Omron CX-Programmer project 新工程 (CX-Programmer 9.62)

# PLC 新PLC1: CJ2M CPU33
I/O table (CPU CJ2M-CPU33): rack 0 slot 0 CJ1W-ID261; rack 0 slot 1 CJ1W-MD261; rack 0 slot 2 CJ1W-OD261; rack 0 slot 3 CJ1W-SCU21-V1; rack 0 slot 11 CJ2M-EIP21

## Global symbols (name address type ; comment)
0.00 BOOL  ; 扫码阻挡气缸1原位
0.01 BOOL  ; 扫码阻挡气缸1到位
0.02 BOOL  ; 扫码阻挡气缸2原位
0.03 BOOL  ; 扫码阻挡气缸2到位
0.04 BOOL  ; 隔离气缸1原位
0.05 BOOL  ; 隔离气缸1到位
0.06 BOOL  ; 隔离气缸2原位
0.07 BOOL  ; 隔离气缸2到位
0.08 BOOL  ; 进料对射光电
0.09 BOOL  ; 夹爪A1夹紧位
0.10 BOOL  ; 夹爪A1松开位
0.11 BOOL  ; 夹爪A2夹紧位
0.12 BOOL  ; 夹爪A2松开位
0.13 BOOL  ; 夹爪B1夹紧位
0.14 BOOL  ; 夹爪B1松开位
0.15 BOOL  ; 夹爪B2夹紧位
10.00 BOOL  ; 扫码阻挡气缸1缩回
10.01 BOOL  ; 扫码阻挡气缸1伸出
10.02 BOOL  ; 扫码阻挡气缸2缩回
10.03 BOOL  ; 扫码阻挡气缸2伸出
10.04 BOOL  ; 隔离气缸1缩回
10.05 BOOL  ; 隔离气缸1伸出
10.06 BOOL  ; 隔离气缸2缩回
10.07 BOOL  ; 隔离气缸2伸出
10.08 BOOL  ; 上料拉带电机启动
10.09 BOOL  ; 夹爪A1夹紧
10.10 BOOL  ; 夹爪A1松开
10.11 BOOL  ; 夹爪A2夹紧
10.12 BOOL  ; 夹爪A2松开
10.13 BOOL  ; 夹爪B1夹紧
10.14 BOOL  ; 夹爪B1松开
10.15 BOOL  ; 夹爪B2夹紧
11.00 BOOL  ; 夹爪B2松开
11.01 BOOL  ; NG升降气缸1缩回
11.02 BOOL  ; NG升降气缸1伸出
11.03 BOOL  ; NG升降气缸2缩回
11.04 BOOL  ; NG升降气缸2伸出
11.05 BOOL  ; 无杆气缸1缩回
11.06 BOOL  ; 无杆气缸1伸出
11.07 BOOL  ; 无杆气缸2缩回
11.08 BOOL  ; 无杆气缸2伸出
11.09 BOOL  ; 阻挡伸出气缸1缩回
11.10 BOOL  ; 阻挡伸出气缸1伸出
11.11 BOOL  ; 阻挡伸出气缸2缩回
11.12 BOOL  ; 阻挡伸出气缸2伸出
11.13 BOOL  ; 阻挡伸出气缸3缩回
11.14 BOOL  ; 阻挡伸出气缸3伸出
11.15 BOOL  ; 阻挡伸出气缸4缩回
12.00 BOOL  ; 阻挡伸出气缸4伸出
12.01 BOOL  ; 精定位气缸A1缩回
12.02 BOOL  ; 精定位气缸A1伸出
12.03 BOOL  ; 精定位气缸A2缩回
12.04 BOOL  ; 精定位气缸A2伸出
12.05 BOOL  ; 精定位气缸B1缩回
12.06 BOOL  ; 精定位气缸B1伸出
12.07 BOOL  ; 精定位气缸B2缩回
12.08 BOOL  ; 精定位气缸B2伸出
12.09 BOOL  ; 擦拭升降气缸缩回
12.10 BOOL  ; 擦拭升降气缸伸出
12.11 BOOL  ; 压钉气缸缩回
12.12 BOOL  ; 压钉气缸伸出
12.13 BOOL  ; 料盒拨料气缸1缩回
12.14 BOOL  ; 料盒拨料气缸1伸出
12.15 BOOL  ; 料盒拨料气缸2缩回
13.00 BOOL  ; 料盒拨料气缸2伸出
13.01 BOOL  ; 推钉X轴气缸缩回
13.02 BOOL  ; 推钉X轴气缸伸出
13.03 BOOL  ; 推钉Y轴气缸缩回
13.04 BOOL  ; 推钉Y轴气缸伸出
13.05 BOOL  ; 钉位清洁拉带启动
13.06 BOOL  ; 入钉拉带启动
13.07 BOOL  ; 扫码NG收料拉带启动
13.08 BOOL  ; 入钉NG收料拉带启动
13.09 BOOL  ; 供钉振动盘启动
13.10 BOOL  ; 清洁料盘放料电机启动
13.11 BOOL  ; 料盘收料电机
13.12 BOOL  ; 真空阀打开
13.13 BOOL  ; 真空阀关闭
13.14 BOOL  ; 吹气阀打开
13.15 BOOL  ; 吹气阀关闭
1535.01 BOOL  ; ETN21_1TCP Socket No.2 Receving Flag
1535.02 BOOL  ; ETN21_1TCP Socket No.2 Sending Flag
1535.03 BOOL  ; ETN21_1TCP Socket No.2 Closing Flag
1535.13 BOOL  ; ETN21_1TCP Socket No.2 Data Receved Flag
1535.15 BOOL  ; ETN21_1TCP Socket No.2 TCP Connection/TCP Open Flag
1544.10 BOOL  ; ETN21_1Socket2 TCP Active Open Request SW
1544.11 BOOL  ; ETN21_1Socket2 Send Request Switch
1544.12 BOOL  ; ETN21_1Socket2 Receive Request SW
1544.13 BOOL  ; ETN21_1Socket2 Close Request SW
1544.15 BOOL  ; SCU21_1 Port#2忙绿标志
1559.15 BOOL  ; SCU21_2Port#1 Protocol Macro Executing Flag
186.00 BOOL  ; 1#入料扫码启动
1.00 BOOL  ; 夹爪B2松开位
1.01 BOOL  ; NG升降气缸1原位
1.02 BOOL  ; NG升降气缸1到位
1.03 BOOL  ; NG升降气缸2原位
1.04 BOOL  ; NG升降气缸2到位
1.05 BOOL  ; 无杆气缸1原位
1.06 BOOL  ; 无杆气缸1到位
1.07 BOOL  ; 无杆气缸2原位
1.08 BOOL  ; 无杆气缸2到位
1.09 BOOL  ; 阻挡伸出气缸1原位
1.10 BOOL  ; 阻挡伸出气缸1到位
1.11 BOOL  ; 阻挡伸出气缸2原位
1.12 BOOL  ; 阻挡伸出气缸2到位
1.13 BOOL  ; 阻挡伸出气缸3原位
1.14 BOOL  ; 阻挡伸出气缸3到位
1.15 BOOL  ; 阻挡伸出气缸4原位
200.00 BOOL  ; PLC上电
200.01 BOOL  ; 紧急停止
200.02 BOOL  ; 自动启动
200.03 BOOL  ; 自动停止
200.04 BOOL  ; 报警清除
200.05 BOOL  ; 清料停止中
200.06 BOOL  ; 异常报警停止
200.07 BOOL  ; 自动模式擦拭拉带启动
200.08 BOOL  ; 自动模式入钉拉带启动
200.09 BOOL  ; 设备内有电池
200.10 BOOL  ; 机台有错误
200.11 BOOL  ; 报警中
200.12 BOOL  ; 三色灯-绿灯
200.13 BOOL  ; 三色灯-红灯
200.14 BOOL  ; 三色灯-黄灯
200.15 BOOL  ; 三色灯-蜂鸣器
201.00 BOOL  ; 整机在初始位
205.00 BOOL  ; 整机停止中（Lamp）
205.01 BOOL  ; 清料停止中（Lamp）
205.02 BOOL  ; 整机复位（Lamp）
210.01 BOOL  ; PC系统通讯正常标志
210.03 BOOL  ; 安全门标志
210.04 BOOL  ; 供料震盘启动标志
210.05 BOOL  ; 机器人Socket_Tcp连接完成标志
210.06 BOOL  ; 扫码枪Socket_Tcp连接完成标志
221.00 BOOL  ; 整机复位（M）
221.01 BOOL  ; 电池上料机构复位（M）
221.02 BOOL  ; 扫码NG抓取机构复位（M）
221.03 BOOL  ; 电池清洁机构复位
221.04 BOOL  ; 电池入钉机构复位（M）
221.05 BOOL  ; 入钉NG抓取机构复位（M）
221.06 BOOL  ; 扫码入料机构记忆复位（M）
221.08 BOOL  ; 进料拉带扫码工站整机复位（M）
2960.06 BOOL  ; 入钉升降伺服负极限
2960.07 BOOL  ; 入钉伺服正极限
2962.06 BOOL  ; 上料水平伺服负极限
2962.07 BOOL  ; 上料水平伺服正极限
2.00 BOOL  ; 阻挡伸出气缸4到位
2.01 BOOL  ; 精定位气缸A1原位
2.02 BOOL  ; 精定位气缸A1到位
2.03 BOOL  ; 精定位气缸A2原位
2.04 BOOL  ; 精定位气缸A2到位
2.05 BOOL  ; 精定位气缸B1原位
2.06 BOOL  ; 精定位气缸B1到位
2.07 BOOL  ; 精定位气缸B2原位
2.08 BOOL  ; 精定位气缸B2到位
2.09 BOOL  ; 擦拭升降气缸原位
2.10 BOOL  ; 擦拭升降气缸到位
2.11 BOOL  ; 压钉气缸原位
2.12 BOOL  ; 压钉气缸到位
2.13 BOOL  ; 料盒拨料气缸1原位
2.14 BOOL  ; 料盒拨料气缸1到位
2.15 BOOL  ; 料盒拨料气缸2原位
300.00 BOOL  ; 扫码阻挡气缸1缩回[Pls]
300.01 BOOL  ; 扫码阻挡气缸1伸出[Pls]
300.02 BOOL  ; 扫码阻挡气缸2缩回[Pls]
300.03 BOOL  ; 扫码阻挡气缸2伸出[Pls]
300.04 BOOL  ; 隔离气缸1缩回[Pls]
300.05 BOOL  ; 隔离气缸1伸出[Pls]
300.06 BOOL  ; 隔离气缸2缩回[Pls]
300.07 BOOL  ; 隔离气缸2伸出[Pls]
300.08 BOOL  ; 进料拉带电机启动[Pls]
300.09 BOOL  ; 夹爪A1夹紧[Pls]
300.10 BOOL  ; 夹爪A1松开[Pls]
300.11 BOOL  ; 夹爪A2夹紧[Pls]
300.12 BOOL  ; 夹爪A2松开[Pls]
300.13 BOOL  ; 夹爪B1夹紧[Pls]
300.14 BOOL  ; 夹爪B1松开[Pls]
300.15 BOOL  ; 夹爪B2夹紧[Pls]
301.00 BOOL  ; 夹爪B2松开[Pls]
301.01 BOOL  ; NG升降气缸1缩回[Pls]
301.02 BOOL  ; NG升降气缸1伸出[Pls]
301.03 BOOL  ; NG升降气缸2缩回[Pls]
301.04 BOOL  ; NG升降气缸2伸出[Pls]
301.05 BOOL  ; 无杆气缸1缩回[Pls]
301.06 BOOL  ; 无杆气缸1伸出[Pls]
301.07 BOOL  ; 无杆气缸2缩回[Pls]
301.08 BOOL  ; 无杆气缸2伸出[Pls]
301.09 BOOL  ; 阻挡伸出气缸1缩回[Pls]
301.10 BOOL  ; 阻挡伸出气缸1伸出[Pls]
301.11 BOOL  ; 阻挡伸出气缸2缩回[Pls]
301.12 BOOL  ; 阻挡伸出气缸2伸出[Pls]
301.13 BOOL  ; 阻挡伸出气缸3缩回[Pls]
301.14 BOOL  ; 阻挡伸出气缸3伸出[Pls]
301.15 BOOL  ; 阻挡伸出气缸4缩回[Pls]
302.00 BOOL  ; 阻挡伸出气缸4伸出[Pls]
302.01 BOOL  ; 精定位气缸A1缩回[Pls]
302.02 BOOL  ; 精定位气缸A1伸出[Pls]
302.03 BOOL  ; 精定位气缸A2缩回[Pls]
302.04 BOOL  ; 精定位气缸A2伸出[Pls]
302.05 BOOL  ; 精定位气缸B1缩回[Pls]
302.06 BOOL  ; 精定位气缸B1伸出[Pls]
302.07 BOOL  ; 精定位气缸B2缩回[Pls]
302.08 BOOL  ; 精定位气缸B2伸出[Pls]
302.09 BOOL  ; 擦拭升降气缸缩回[Pls]
302.10 BOOL  ; 擦拭升降气缸伸出[Pls]
302.11 BOOL  ; 压钉气缸缩回[Pls]
302.12 BOOL  ; 压钉气缸伸出[Pls]
302.13 BOOL  ; 料盒拨料气缸1缩回[Pls]
302.14 BOOL  ; 料盒拨料气缸1伸出[Pls]
302.15 BOOL  ; 料盒拨料气缸2缩回[Pls]
303.00 BOOL  ; 料盒拨料气缸2伸出[Pls]
303.01 BOOL  ; 推钉X轴气缸缩回[Pls]
303.02 BOOL  ; 推钉X轴气缸伸出[Pls]
303.03 BOOL  ; 推钉Y轴气缸缩回[Pls]
303.04 BOOL  ; 推钉Y轴气缸伸出[Pls]
303.05 BOOL  ; 入钉位拉带启动[Pls]
303.06 BOOL  ; 入钉NG位拉带启动[Pls]
303.07 BOOL  ; 清洁放料拉带启动[Pls]
303.08 BOOL  ; 清洁收料拉带启动[Pls]
303.09 BOOL  ; 供料振动盘启动[Pls]
303.11 BOOL  ; 入钉真空阀打开PLS
303.12 BOOL  ; $?St$Bk?_#[5] / 入钉真空阀打开PLS / $?St$Bk?_#[5]
303.13 BOOL  ; 入钉真空阀关闭PLS
303.14 BOOL  ; 入钉吹气阀打开PLS
303.15 BOOL  ; 入钉吹气阀关闭PLS
3.00 BOOL  ; 料盒拨料气缸2到位
3.01 BOOL  ; 推钉X轴气缸原位
3.02 BOOL  ; 推钉X轴气缸到位
3.03 BOOL  ; 推钉Y轴气缸原位
3.04 BOOL  ; 推钉Y轴气缸到位
3.05 BOOL  ; 扫码位对射光电
3.06 BOOL  ; 分隔电池对射光电
3.07 BOOL  ; 擦拭料带下限满料感应
3.08 BOOL  ; 擦拭料带放料上限光电[0003.08]
3.09 BOOL  ; 擦拭带盘无料料感应
3.10 BOOL  ; 扫码NG位对射光电
3.11 BOOL  ; 擦拭位对射光电
3.12 BOOL  ; 入钉位对射光电
3.13 BOOL  ; 入钉NG位对射光电
3.14 BOOL  ; 扫码NG槽对射前
3.15 BOOL  ; 入钉NG槽对射前
400.00 BOOL  ; 扫码阻挡气缸1缩回[M]
400.01 BOOL  ; 扫码阻挡气缸1伸出[M]
400.02 BOOL  ; 扫码阻挡气缸2缩回[M]
400.03 BOOL  ; 扫码阻挡气缸2伸出[M]
400.04 BOOL  ; 隔离气缸1缩回[M]
400.05 BOOL  ; 隔离气缸1伸出[M]
400.06 BOOL  ; 隔离气缸2缩回[M]
400.07 BOOL  ; 隔离气缸2伸出[M]
400.08 BOOL  ; 进料拉带电机启动[M]
400.09 BOOL  ; 夹爪A1夹紧[M]
400.10 BOOL  ; 夹爪A1松开[M]
400.11 BOOL  ; 夹爪A2夹紧[M]
400.12 BOOL  ; 夹爪A2松开[M]
400.13 BOOL  ; 夹爪B1夹紧[M]
400.14 BOOL  ; 夹爪B1松开[M]
400.15 BOOL  ; 夹爪B2夹紧[M]
401.00 BOOL  ; 夹爪B2松开[M]
401.01 BOOL  ; NG升降气缸1缩回[M]
401.02 BOOL  ; NG升降气缸1伸出[M]
401.03 BOOL  ; NG升降气缸2缩回[M]
401.04 BOOL  ; NG升降气缸2伸出[M]
401.05 BOOL  ; 无杆气缸1缩回[M]
401.06 BOOL  ; 无杆气缸1伸出[M]
401.07 BOOL  ; 无杆气缸2缩回[M]
401.08 BOOL  ; 无杆气缸2伸出[M]
401.09 BOOL  ; 阻挡伸出气缸1缩回[M]
401.10 BOOL  ; 阻挡伸出气缸1伸出[M]
401.11 BOOL  ; 阻挡伸出气缸2缩回[M]
401.12 BOOL  ; 阻挡伸出气缸2伸出[M]
401.13 BOOL  ; 阻挡伸出气缸3缩回[M]
401.14 BOOL  ; 阻挡伸出气缸3伸出[M]
401.15 BOOL  ; 阻挡伸出气缸4缩回[M]
402.00 BOOL  ; 阻挡伸出气缸4伸出[M]
402.01 BOOL  ; 精定位气缸A1缩回[M]
402.02 BOOL  ; 精定位气缸A1伸出[M]
402.03 BOOL  ; 精定位气缸A2缩回[M]
402.04 BOOL  ; 精定位气缸A2伸出[M]
402.05 BOOL  ; 精定位气缸B1缩回[M]
402.06 BOOL  ; 精定位气缸B1伸出[M]
402.07 BOOL  ; 精定位气缸B2缩回[M]
402.08 BOOL  ; 精定位气缸B2伸出[M]
402.09 BOOL  ; 擦拭升降气缸缩回[M]
402.10 BOOL  ; 擦拭升降气缸伸出[M]
402.11 BOOL  ; 压钉气缸缩回[M]
402.12 BOOL  ; 压钉气缸伸出[M]
402.13 BOOL  ; 料盒拨料气缸1缩回[M]
402.14 BOOL  ; 料盒拨料气缸1伸出[M]
402.15 BOOL  ; 料盒拨料气缸2缩回[M]
403.00 BOOL  ; 料盒拨料气缸2伸出[M]
403.01 BOOL  ; 推钉X轴气缸缩回[M]
403.02 BOOL  ; 推钉X轴气缸伸出[M]
403.03 BOOL  ; 推钉Y轴气缸缩回[M]
403.04 BOOL  ; 推钉Y轴气缸伸出[M]
403.05 BOOL  ; $?St$Bk?_#[6] / 钉位清洁拉带启动[M] / $?St$Bk?_#[6]
403.06 BOOL  ; 入钉位拉带启动[M]
403.07 BOOL  ; 扫码NG收料拉带启动(M)
403.08 BOOL  ; 入钉NG收料拉带启动[M]
403.09 BOOL  ; 供钉振动盘启动[M]
403.10 BOOL  ; 清洁料盘放料电机启动（M)
403.11 BOOL  ; 料盘收料电机启动
403.12 BOOL  ; 入钉真空阀打开
403.13 BOOL  ; $?St$Bk?_#[7] / 入钉真空阀关闭[M] / $?St$Bk?_#[7]
403.14 BOOL  ; 入钉吹气阀打开（M)
403.15 BOOL  ; 入钉吹气阀关闭M
406.00 BOOL  ; 扫码按钮HIM
417.00 BOOL  ; 进料拉带扫码测试[M]
4.00 BOOL  ; 入钉伺服使能
4.02 BOOL  ; 给下位机拉带下料信号
4.05 BOOL  ; 启动按钮指示灯
4.06 BOOL  ; 停止按钮指示灯
4.07 BOOL  ; 复位按钮指示灯
4.08 BOOL  ; 三色灯（红）
4.09 BOOL  ; 三色灯（绿）
4.10 BOOL  ; 三色灯（黄）
4.11 BOOL  ; 蜂鸣器
4.12 BOOL  ; $?St$Bk?_#[8] / 入钉刹车线圈 / $?St$Bk?_#[8]
500.00 BOOL  ; 扫码阻挡气缸1缩回条件
500.01 BOOL  ; 扫码阻挡气缸1伸出条件
500.02 BOOL  ; 扫码阻挡气缸2缩回条件
500.03 BOOL  ; 扫码阻挡气缸2伸出条件
500.04 BOOL  ; 隔离气缸1缩回条件
500.05 BOOL  ; 隔离气缸1伸出条件
500.06 BOOL  ; 隔离气缸2缩回条件
500.07 BOOL  ; 隔离气缸2伸出条件
500.08 BOOL  ; 上料拉带电机启动条件
500.09 BOOL  ; 夹爪A1夹紧条件
500.10 BOOL  ; 夹爪A1松开条件
500.11 BOOL  ; 夹爪A2夹紧条件
500.12 BOOL  ; 夹爪A2松开条件
500.13 BOOL  ; 夹爪B1夹紧条件
500.14 BOOL  ; 夹爪B1松开条件
500.15 BOOL  ; 夹爪B2夹紧条件
501.00 BOOL  ; 夹爪B2松开条件
501.01 BOOL  ; NG升降气缸1缩回条件
501.02 BOOL  ; NG升降气缸1伸出条件
501.03 BOOL  ; NG升降气缸2缩回条件
501.04 BOOL  ; NG升降气缸2伸出条件
501.05 BOOL  ; 无杆气缸1缩回条件
501.06 BOOL  ; 无杆气缸1伸出条件
501.07 BOOL  ; 无杆气缸2缩回条件
501.08 BOOL  ; 无杆气缸2伸出条件
501.09 BOOL  ; 阻挡伸出气缸1缩回条件
501.10 BOOL  ; 阻挡伸出气缸1伸出条件
501.11 BOOL  ; 阻挡伸出气缸2缩回条件
501.12 BOOL  ; 阻挡伸出气缸2伸出条件
501.13 BOOL  ; 阻挡伸出气缸3缩回条件
501.14 BOOL  ; 阻挡伸出气缸3伸出条件
501.15 BOOL  ; 阻挡伸出气缸4缩回条件
502.00 BOOL  ; 阻挡伸出气缸4伸出条件
502.01 BOOL  ; 精定位气缸A1缩回条件
502.02 BOOL  ; 精定位气缸A1伸出条件
502.03 BOOL  ; 精定位气缸A2缩回条件
502.04 BOOL  ; 精定位气缸A2伸出条件
502.05 BOOL  ; 精定位气缸B1缩回条件
502.06 BOOL  ; 精定位气缸B1伸出条件
502.07 BOOL  ; 精定位气缸B2缩回条件
502.08 BOOL  ; 精定位气缸B2伸出条件
502.09 BOOL  ; 擦拭升降气缸缩回条件
502.10 BOOL  ; 擦拭升降气缸伸出条件
502.11 BOOL  ; 压钉气缸缩回条件
502.12 BOOL  ; 压钉气缸伸出条件
502.13 BOOL  ; 料盒拨料气缸1缩回条件
502.14 BOOL  ; 料盒拨料气缸1伸出条件
502.15 BOOL  ; 料盒拨料气缸2缩回条件
503.00 BOOL  ; 料盒拨料气缸2伸出条件
503.01 BOOL  ; 推钉X轴气缸缩回条件
503.02 BOOL  ; 推钉X轴气缸伸出条件
503.03 BOOL  ; 推钉Y轴气缸缩回条件
503.04 BOOL  ; 推钉Y轴气缸伸出条件
503.05 BOOL  ; $?St$Bk?_#[9] / 钉位清洁拉带启动条件 / $?St$Bk?_#[9]
503.06 BOOL  ; 入钉NG位拉带启动条件
503.07 BOOL  ; 清洁放料拉带启动条件
503.08 BOOL  ; 清洁收料拉带启动条件
503.09 BOOL  ; 供料振动盘启动条件
503.12 BOOL  ; $?St$Bk?_#[10] / 入钉真空阀条件 / $?St$Bk?_#[10]
503.13 BOOL  ; $?St$Bk?_#[11] / 入钉真空阀关闭条件 / $?St$Bk?_#[11]
503.14 BOOL  ; $?St$Bk?_#[12] / 入钉吹气打开条件 / $?St$Bk?_#[12]
503.15 BOOL  ; 入钉吹气关闭条件
600.00 BOOL  ; 扫码阻挡气缸1缩回[A]
600.01 BOOL  ; 扫码阻挡气缸1伸出[A]
600.02 BOOL  ; 扫码阻挡气缸2缩回[A]
600.03 BOOL  ; 扫码阻挡气缸2伸出[A]
600.04 BOOL  ; 隔离气缸1缩回[A]
600.05 BOOL  ; 隔离气缸1伸出[A]
600.06 BOOL  ; 隔离气缸2缩回[A]
600.07 BOOL  ; 隔离气缸2伸出[A]
600.08 BOOL  ; 进料拉带电机启动[A]
600.09 BOOL  ; 夹爪A1夹紧[A]
600.10 BOOL  ; 夹爪A1松开[A]
600.11 BOOL  ; 夹爪A2夹紧[A]
600.12 BOOL  ; 夹爪A2松开[A]
600.13 BOOL  ; 夹爪B1夹紧[A]
600.14 BOOL  ; 夹爪B1松开[A]
600.15 BOOL  ; 夹爪B2夹紧[A]
601.00 BOOL  ; 夹爪B2松开[A]
601.01 BOOL  ; NG升降气缸1缩回[A]
601.02 BOOL  ; NG升降气缸1伸出[A]
601.03 BOOL  ; NG升降气缸2缩回[A]
601.04 BOOL  ; NG升降气缸2伸出[A]
601.05 BOOL  ; 无杆气缸1缩回[A]
601.06 BOOL  ; 无杆气缸1伸出[A]
601.07 BOOL  ; 无杆气缸2缩回[A]
601.08 BOOL  ; 无杆气缸2伸出[A]
601.09 BOOL  ; 阻挡伸出气缸1缩回[A]
601.10 BOOL  ; 阻挡伸出气缸1伸出[A]
601.11 BOOL  ; 阻挡伸出气缸2缩回[A]
601.12 BOOL  ; 阻挡伸出气缸2伸出[A]
601.13 BOOL  ; 阻挡伸出气缸3缩回[A]
601.14 BOOL  ; 阻挡伸出气缸3伸出[A]
601.15 BOOL  ; 阻挡伸出气缸4缩回[A]
602.00 BOOL  ; 阻挡伸出气缸4伸出[A]
602.01 BOOL  ; 精定位气缸A1缩回[A]
602.02 BOOL  ; 精定位气缸A1伸出[A]
602.03 BOOL  ; 精定位气缸A2缩回[A]
602.04 BOOL  ; 精定位气缸A2伸出[A]
602.05 BOOL  ; 精定位气缸B1缩回[A]
602.06 BOOL  ; 精定位气缸B1伸出[A]
602.07 BOOL  ; 精定位气缸B2缩回[A]
602.08 BOOL  ; 精定位气缸B2伸出[A]
602.09 BOOL  ; 擦拭升降气缸缩回[A]
602.10 BOOL  ; 擦拭升降气缸伸出[A]
602.11 BOOL  ; 压钉气缸缩回[A]
602.12 BOOL  ; 压钉气缸伸出[A]
602.13 BOOL  ; 料盒拨料气缸1缩回[A]
602.14 BOOL  ; 料盒拨料气缸1伸出[A]
602.15 BOOL  ; 料盒拨料气缸2缩回[A]
603.00 BOOL  ; 料盒拨料气缸2伸出[A]
603.01 BOOL  ; 推钉X轴气缸缩回[A]
603.02 BOOL  ; 推钉X轴气缸伸出[A]
603.03 BOOL  ; 推钉Y轴气缸缩回[A]
603.04 BOOL  ; 推钉Y轴气缸伸出[A]
603.05 BOOL  ; $?St$Bk?_#[13] / 钉位清洁拉带启动[A] / $?St$Bk?_#[13]
603.06 BOOL  ; 入钉NG位拉带启动[A]
603.07 BOOL  ; 扫码NG收料拉带启动[A]
603.08 BOOL  ; 入钉NG收料拉带启动[A]
603.09 BOOL  ; 供钉振动盘启动[A]
603.10 BOOL  ; 清洁料盘放料电机启动[A]
603.11 BOOL  ; $?St$Bk?_#[14] / 料盘收料电机启动[M] / $?St$Bk?_#[14]
603.12 BOOL  ; $?St$Bk?_#[15] / 入钉真空阀打开 / $?St$Bk?_#[15]
603.13 BOOL  ; 入钉真空阀关闭
603.14 BOOL  ; $?St$Bk?_#[16] / 入钉吹气打开[A] / $?St$Bk?_#[16]
603.15 BOOL  ; 入钉吹气阀关闭
6.00 BOOL  ; 扫码NG槽对射光电
6.01 BOOL  ; 入钉NG槽对射后
6.02 BOOL  ; 入钉检测区域光纤
6.03 BOOL  ; 入钉伺服就绪
6.04 BOOL  ; 入钉伺服报警
6.05 BOOL  ; 启动按钮
6.06 BOOL  ; 停止按钮
6.07 BOOL  ; 复位按钮
6.08 BOOL  ; 急停按钮
6.09 BOOL  ; 手自动选择
6.10 BOOL  ; 设备总气压
6.11 BOOL  ; 夹爪1柔性报警
6.12 BOOL  ; 夹爪2柔性报警
6.13 BOOL  ; 真空信号
6.14 BOOL  ; 开关电源监测
6.15 BOOL  ; 变频器监测
700 CHANNEL  ; 手动按钮操作字
700.00 BOOL  ; 扫码阻挡气缸1缩回[SW]
700.01 BOOL  ; 扫码阻挡气缸1伸出[SW]
700.02 BOOL  ; 扫码阻挡气缸2缩回[SW]
700.03 BOOL  ; 扫码阻挡气缸2伸出[SW]
700.04 BOOL  ; 隔离气缸1缩回[SW]
700.05 BOOL  ; 隔离气缸1伸出[SW]
700.06 BOOL  ; 隔离气缸2缩回[SW]
700.07 BOOL  ; 隔离气缸2伸出[SW]
700.08 BOOL  ; 进料拉带电机启动[SW]
700.09 BOOL  ; 夹爪A1夹紧[SW]
700.10 BOOL  ; 夹爪A1松开[SW]
700.11 BOOL  ; 夹爪A2夹紧[SW]
700.12 BOOL  ; 夹爪A2松开[SW]
700.13 BOOL  ; 夹爪B1夹紧[SW]
700.14 BOOL  ; 夹爪B1松开[SW]
700.15 BOOL  ; 夹爪B2夹紧[SW]
701.00 BOOL  ; 夹爪B2松开[SW]
701.01 BOOL  ; NG升降气缸1缩回[SW]
701.02 BOOL  ; NG升降气缸1伸出[SW]
701.03 BOOL  ; NG升降气缸2缩回[SW]
701.04 BOOL  ; NG升降气缸2伸出[SW]
701.05 BOOL  ; 无杆气缸1缩回[SW]
701.06 BOOL  ; 无杆气缸1伸出[SW]
701.07 BOOL  ; 无杆气缸2缩回[SW]
701.08 BOOL  ; 无杆气缸2伸出[SW]
701.09 BOOL  ; 阻挡伸出气缸1缩回[SW]
701.10 BOOL  ; 阻挡伸出气缸1伸出[SW]
701.11 BOOL  ; 阻挡伸出气缸2缩回[SW]
701.12 BOOL  ; 阻挡伸出气缸2伸出[SW]
701.13 BOOL  ; 阻挡伸出气缸3缩回[SW]
701.14 BOOL  ; 阻挡伸出气缸3伸出[SW]
701.15 BOOL  ; 阻挡伸出气缸4缩回[SW]
702.00 BOOL  ; 阻挡伸出气缸4伸出[SW]
702.01 BOOL  ; 精定位气缸A1缩回[SW]
702.02 BOOL  ; 精定位气缸A1伸出[SW]
702.03 BOOL  ; 精定位气缸A2缩回[SW]
702.04 BOOL  ; 精定位气缸A2伸出[SW]
702.05 BOOL  ; 精定位气缸B1缩回[SW]
702.06 BOOL  ; 精定位气缸B1伸出[SW]
702.07 BOOL  ; 精定位气缸B2缩回[SW]
702.08 BOOL  ; 精定位气缸B2伸出[SW]
702.09 BOOL  ; 擦拭升降气缸缩回[SW]
702.10 BOOL  ; 擦拭升降气缸伸出[SW]
702.11 BOOL  ; 压钉气缸缩回[SW]
702.12 BOOL  ; 压钉气缸伸出[SW]
702.13 BOOL  ; 料盒拨料气缸1缩回[SW]
702.14 BOOL  ; 料盒拨料气缸1伸出[SW]
702.15 BOOL  ; 料盒拨料气缸2缩回[SW]
703.00 BOOL  ; 料盒拨料气缸2伸出[SW]
703.01 BOOL  ; 推钉X轴气缸缩回[SW]
703.02 BOOL  ; 推钉X轴气缸伸出[SW]
703.03 BOOL  ; 推钉Y轴气缸缩回[SW]
703.04 BOOL  ; 推钉Y轴气缸伸出[SW]
703.05 BOOL  ; 钉位清洁拉带启动[SW]
703.06 BOOL  ; 入钉位拉带启动[SW]
703.07 BOOL  ; 扫码NG收料拉带启动[SW]
703.08 BOOL  ; 入钉NG收料拉带启动[SW]
703.09 BOOL  ; 供钉振动盘启动[SW]
703.10 BOOL  ; 清洁料盘放料电机启动（SW)
703.11 BOOL  ; 料盘收料电机
703.12 BOOL  ; 入钉真空阀打开
703.13 BOOL  ; 入钉真空阀关闭
703.14 BOOL  ; 入钉吹气阀打开
703.15 BOOL  ; 入钉吹气阀关闭
710 CHANNEL  ; 手动按钮操作字
712.00 BOOL  ; 进料拉带电机停止[SW]
712.01 BOOL  ; 钉位清洁拉带停止[SW]
712.02 BOOL  ; 入钉位拉带停止[SW]
712.03 BOOL  ; 扫码NG收料拉带停止[SW]
712.04 BOOL  ; 入钉NG收料拉带停止[SW]
712.05 BOOL  ; 供钉振动盘停止[SW]
712.06 BOOL  ; 清洁料盘放料电机停止（SW)
712.07 BOOL  ; 清洁料盘收料电机停止（SW)
712.08 BOOL  ; $?St$Bk?_#[17] / 入钉真空阀关闭[SW] / $?St$Bk?_#[17]
712.09 BOOL  ; $?St$Bk?_#[18] / 入钉吹气阀关闭[SW] / $?St$Bk?_#[18]
716.00 BOOL  ; 1#入料扫码[SW]
750 CHANNEL  ; 手动按钮操作字
7.00 BOOL  ; NG门磁开关
7.01 BOOL  ; 前门磁开关
7.02 BOOL  ; 后门磁开关
7.03 BOOL  ; 左门磁开关
7.04 BOOL  ; 右门磁开关
7.05 BOOL  ; 区域光纤对射
7.06 BOOL  ; 钉位钉子对射光纤钉位
7.07 BOOL  ; 震盘钉嘴反射光纤
7.08 BOOL  ; 拉带入口对射光电
7.10 BOOL  ; 下位机收料完成信号
7.12 BOOL  ; 1
800.00 BOOL  ; 扫码阻挡气缸1原位标志[0000.00]
800.01 BOOL  ; 扫码阻挡气缸1到位标志[0000.01]
800.02 BOOL  ; 扫码阻挡气缸2原位标志[0000.02]
800.03 BOOL  ; 扫码阻挡气缸2到位标志[0000.03]
800.04 BOOL  ; 隔离气缸1原位标志[0000.04]
800.05 BOOL  ; 隔离气缸1到位标志[0000.05]
800.06 BOOL  ; 隔离气缸2原位标志[0000.06]
800.07 BOOL  ; 隔离气缸2到位标志[0000.07]
800.08 BOOL  ; 进料对射光电满料标志[0000.08]
800.09 BOOL  ; 夹爪A1夹紧位标志[0000.09]
800.10 BOOL  ; 夹爪A1松开位标志[0000.10]
800.11 BOOL  ; 夹爪A2夹紧位标志[0000.11]
800.12 BOOL  ; 夹爪A2松开位标志[0000.12]
800.13 BOOL  ; 夹爪B1夹紧位标志[0000.13]
800.14 BOOL  ; 夹爪B1松开位标志[0000.14]
800.15 BOOL  ; 夹爪B2夹紧位标志[0000.15]
801.00 BOOL  ; 夹爪B2松开位标志[0001.00]
801.01 BOOL  ; NG升降气缸1原位标志[0001.01]
801.02 BOOL  ; NG升降气缸1到位标志[0001.02]
801.03 BOOL  ; NG升降气缸2原位标志[0001.03]
801.04 BOOL  ; NG升降气缸2到位标志[0001.04]
801.05 BOOL  ; 无杆气缸1原位标志[0001.05]
801.06 BOOL  ; 无杆气缸1到位标志[0001.06]
801.07 BOOL  ; 无杆气缸2原位标志[0001.07]
801.08 BOOL  ; 无杆气缸2到位标志[0001.08]
801.09 BOOL  ; 拉带阻挡气缸1原位标志[0001.09]
801.10 BOOL  ; 拉带阻挡气缸1到位标志[0001.10]
801.11 BOOL  ; 拉带阻挡气缸2原位标志[0001.11]
801.12 BOOL  ; 拉带阻挡伸出气缸2到位标志[0001.12]
801.13 BOOL  ; 阻挡伸出气缸3原位标志[0001.13]
801.14 BOOL  ; 阻挡伸出气缸3到位标志[0001.14]
801.15 BOOL  ; 阻挡伸出气缸4原位标志[0001.15]
802.00 BOOL  ; 阻挡伸出气缸4到位标志[0002.00]
802.01 BOOL  ; 精定位气缸A1原位标志[0002.01]
802.02 BOOL  ; 精定位气缸A1到位标志[0002.02]
802.03 BOOL  ; 精定位气缸A2原位标志[0002.03]
802.04 BOOL  ; 精定位气缸A2到位标志[0002.04]
802.05 BOOL  ; 精定位气缸B1原位标志[0002.05]
802.06 BOOL  ; 精定位气缸B1到位标志[0002.06]
802.07 BOOL  ; 精定位气缸B2原位标志[0002.07]
802.08 BOOL  ; 精定位气缸B2到位标志[0002.08]
802.09 BOOL  ; 擦拭升降气缸原位标志[0002.09]
802.10 BOOL  ; 擦拭升降气缸到位标志[0002.10]
802.11 BOOL  ; 压钉气缸原位标志[0002.11]
802.12 BOOL  ; 压钉气缸到位标志[0002.12]
802.13 BOOL  ; 料盒拨料气缸1原位标志[0002.13]
802.14 BOOL  ; 料盒拨料气缸1到位标志[0002.14]
802.15 BOOL  ; 料盒拨料气缸2原位标志[0002.15]
803.00 BOOL  ; 料盒拨料气缸2到位标志[0003.00]
803.01 BOOL  ; 推钉X轴气缸原位标志[0003.01]
803.02 BOOL  ; 推钉X轴气缸到位标志[0003.02]
803.03 BOOL  ; 推钉Y轴气缸原位标志[0003.03]
803.04 BOOL  ; 推钉Y轴气缸到位标志[0003.04]
803.05 BOOL  ; 扫码位对射光电来料标志[0003.05]
803.06 BOOL  ; 分隔电池对射光电有料标志[0003.06]
803.07 BOOL  ; 擦拭料带满标志[0003.07]
803.08 BOOL  ; 擦拭料带上限放料光电标志[0003.08]
803.09 BOOL  ; 擦拭带盘无料感应标志
803.10 BOOL  ; 扫码NG位对射光电有料标志[0003.10]
803.11 BOOL  ; 擦拭位对射光电有料标志[0003.11]
803.12 BOOL  ; 入钉位对射光电有料标志[0003.12]
803.13 BOOL  ; 入钉NG位对射光电有料标志[0003.13]
803.14 BOOL  ; 扫码NG槽对射前光电有料标志[0003.14]
803.15 BOOL  ; 入钉NG槽对射前光电有料标志[0003.15]
804.00 BOOL  ; 扫码NG槽对射光电满料标志[0006.00]
804.01 BOOL  ; 入钉NG槽对射光电满料标志[0006.01]
804.02 BOOL  ; 入钉检测区域光纤
804.03 BOOL  ; 入钉伺服就绪 标志[0006.03]
804.04 BOOL  ; 入钉伺服报警 标志[0006.04]
804.05 BOOL  ; 启动按钮标志[0006.05]
804.06 BOOL  ; 停止按钮标志[0006.06]
804.07 BOOL  ; 复位按钮标志[0006.07]
804.08 BOOL  ; 急停按钮标志[0006.08]
804.09 BOOL  ; 手自动选择标志[0006.09]
804.10 BOOL  ; 设备总气压标志[0006.10]
804.11 BOOL  ; 夹爪1柔性报警标志[0006.11]
804.12 BOOL  ; 夹爪2柔性报警标志[0006.12]
804.13 BOOL  ; 真空信号标志[0006.13]
804.14 BOOL  ; 开关电源监测标志[0006.14]
804.15 BOOL  ; 变频器监测标志[0006.15]
805.00 BOOL  ; NG门磁开关标志[0007.00]
805.01 BOOL  ; 前门磁开关标志[0007.01]
805.02 BOOL  ; 后门磁开关标志[0007.02]
805.03 BOOL  ; 左门磁开关标志[0007.03]
805.04 BOOL  ; 右门磁开关标志[0007.04]
805.05 BOOL  ; 区域光纤对射入钉完成标志[0007.05]
805.06 BOOL  ; 钉位钉子对射光纤来钉标志
805.07 BOOL  ; 震盘钉嘴反射光纤有钉嘴标志[0007.07]
805.08 BOOL  ; 拉带入口对射光电来料标志
900.00 BOOL  ; 扫码阻挡气缸1原位[lamp]
900.01 BOOL  ; 扫码阻挡气缸1到位[lamp]
900.02 BOOL  ; 扫码阻挡气缸2原位[lamp]
900.03 BOOL  ; 扫码阻挡气缸2到位[lamp]
900.04 BOOL  ; 隔离气缸1原位[lamp]
900.05 BOOL  ; 隔离气缸1到位[lamp]
900.06 BOOL  ; 隔离气缸2原位[lamp]
900.07 BOOL  ; 隔离气缸2到位[lamp]
900.08 BOOL  ; 进料拉带电机启动[lamp]
900.09 BOOL  ; 夹爪A1夹紧位[lamp]
900.10 BOOL  ; 夹爪A1松开位[lamp]
900.11 BOOL  ; 夹爪A2夹紧位[lamp]
900.12 BOOL  ; 夹爪A2松开位[lamp]
900.13 BOOL  ; 夹爪B1夹紧位[lamp]
900.14 BOOL  ; 夹爪B1松开位[lamp]
900.15 BOOL  ; 夹爪B2夹紧位[lamp]
901.00 BOOL  ; 夹爪B2松开位[lamp]
901.01 BOOL  ; NG升降气缸1原位[lamp]
901.02 BOOL  ; NG升降气缸1到位[lamp]
901.03 BOOL  ; NG升降气缸2原位[lamp]
901.04 BOOL  ; NG升降气缸2到位[lamp]
901.05 BOOL  ; NG无杆气缸1原位[lamp]
901.06 BOOL  ; NG无杆气缸1到位[lamp]
901.07 BOOL  ; NG无杆气缸2原位[lamp]
901.08 BOOL  ; NG无杆气缸2到位[lamp]
901.09 BOOL  ; 阻挡伸出气缸1原位[lamp]
901.10 BOOL  ; 阻挡伸出气缸1到位[lamp]
901.11 BOOL  ; 阻挡伸出气缸2原位[lamp]
901.12 BOOL  ; 阻挡伸出气缸2到位[lamp]
901.13 BOOL  ; 阻挡伸出气缸3原位[lamp]
901.14 BOOL  ; 阻挡伸出气缸3到位[lamp]
901.15 BOOL  ; 阻挡伸出气缸4原位[lamp]
902.00 BOOL  ; 阻挡伸出气缸4到位[lamp]
902.01 BOOL  ; 精定位气缸A1原位[lamp]
902.02 BOOL  ; 精定位气缸A1到位[lamp]
902.03 BOOL  ; 精定位气缸A2原位[lamp]
902.04 BOOL  ; 精定位气缸A2到位[lamp]
902.05 BOOL  ; 精定位气缸B1原位[lamp]
902.06 BOOL  ; 精定位气缸B1到位[lamp]
902.07 BOOL  ; 精定位气缸B2原位[lamp]
902.08 BOOL  ; 精定位气缸B2到位[lamp]
902.09 BOOL  ; 擦拭升降气缸原位[lamp]
902.10 BOOL  ; 擦拭升降气缸到位[lamp]
902.11 BOOL  ; 压钉气缸原位[lamp]
902.12 BOOL  ; 压钉气缸到位[lamp]
902.13 BOOL  ; 料盒拨料气缸1原位[lamp]
902.14 BOOL  ; 料盒拨料气缸1到位[lamp]
902.15 BOOL  ; 料盒拨料气缸2原位[lamp]
903.00 BOOL  ; 料盒拨料气缸2到位[lamp]
903.01 BOOL  ; 推钉X轴气缸原位[lamp]
903.02 BOOL  ; 推钉X轴气缸到位[lamp]
903.03 BOOL  ; 推钉Y轴气缸原位[lamp]
903.04 BOOL  ; 推钉Y轴气缸到位[lamp]
903.05 BOOL  ; 扫码位对射光电[lamp]
903.06 BOOL  ; 分隔电池对射光电[lamp]
903.07 BOOL  ; 清料带光电1[lamp]
903.08 BOOL  ; 清料带光电2[lamp]
903.09 BOOL  ; 料盘清洁带有料[lamp]
903.10 BOOL  ; 扫码NG位对射光电[lamp]
903.11 BOOL  ; 擦拭位对射光电[lamp]
903.12 BOOL  ; 入钉位对射光电[lamp]
903.13 BOOL  ; 入钉NG位对射光电[lamp]
903.14 BOOL  ; 清洁放料拉带电机启动[lamp]
903.15 BOOL  ; 放料位对射2光电[lamp]
904.00 BOOL  ; 取料位对射1光电[lamp]
904.01 BOOL  ; 取料位对射2光电[lamp]
904.02 BOOL  ; 放料允许信号[lamp]
904.03 BOOL  ; 入钉伺服就绪 [lamp]
904.04 BOOL  ; 入钉伺服报警 [lamp]
904.05 BOOL  ; 启动按钮[lamp]
904.06 BOOL  ; 停止按钮[lamp]
904.07 BOOL  ; 复位按钮[lamp]
904.08 BOOL  ; 急停按钮[lamp]
904.09 BOOL  ; 手自动选择[lamp]
904.10 BOOL  ; 设备总气压[lamp]
904.11 BOOL  ; 夹爪1柔性报警[lamp]
904.12 BOOL  ; 夹爪2柔性报警[lamp]
904.13 BOOL  ; 真空信号[lamp]
904.14 BOOL  ; 开关电源监测[lamp]
904.15 BOOL  ; 变频器监测[lamp]
905.00 BOOL  ; NG门磁开关[lamp]
905.01 BOOL  ; 前门磁开关[lamp]
905.02 BOOL  ; 后门磁开关[lamp]
905.03 BOOL  ; 左门磁开关[lamp]
905.04 BOOL  ; 右门磁开关[lamp]
9.07 BOOL  ; 急停按钮信号
A202.01 BOOL  ; SCU21_1 Port#2 端口允许标志
A202.05 BOOL  ; SCU21_2 Port#1 端口5允许标志
A276 CHANNEL  ; 进料水平伺服当前脉冲
A280.04 BOOL  ; 入钉升降伺服脉冲输出中
A280.05 BOOL  ; 入钉升降伺服无原点标志
A322 CHANNEL  ; 擦拭步进位置脉冲
A324 CHANNEL  ; 入钉步进位置脉冲
A326.04 BOOL  ; 擦拭步进脉冲输出中
A326.05 BOOL  ; 上料水平伺服无原点
A327.04 BOOL  ; 入钉旋转步进脉冲输出中
A540.08 BOOL  ; 入钉升降伺服CW
A540.09 BOOL  ; 入钉升降伺服CCW
A621.02 BOOL  ; 单元重启
C0060 BOOL  ; 上料拉带扫码NG后重扫次数
D10 CHANNEL  ; 入钉升降伺服自动速度   HMI
D100 CHANNEL  ; 入钉升降伺服准入钉位参数设定 (M)
D10000 CHANNEL  ; 控制字
D10001 CHANNEL  ; 扫码位条码开始字（传递）
D1000.00 BOOL  ; 电池上料机构始位
D1000.01 BOOL  ; 扫码阻挡放料条件
D1000.02 BOOL  ; 扫码拉带启动条件
D1000.05 BOOL  ; 上料机构扫码停止标志
D1000.06 BOOL  ; 电池上料机构清料完成
D1000.07 BOOL  ; 电池上料机构异常标志
D1001.00 BOOL  ; 上料机构工站复位
D1001.01 BOOL  ; 扫码阻挡气缸1伸出
D1001.02 BOOL  ; 扫码阻挡气缸2伸出
D1001.03 BOOL  ; 隔离气缸1缩回
D1001.04 BOOL  ; 隔离气缸2缩回
D1001.05 BOOL  ; 隔离气缸1伸出
D1001.06 BOOL  ; 隔离气缸2伸出
D10020 CHANNEL  ; 扫码数据结束字（传递）
D1002.00 BOOL  ; 上料拉带扫码开始运行条件
D1002.01 BOOL  ; 上料拉带扫码步进条件
D1002.15 BOOL  ; 上料拉带扫码步进
D1003 CHANNEL  ; 上料拉带扫码步序号
D1003.00 BOOL  ; 上料拉带扫码自动开始
D1003.01 BOOL  ; 上料拉带扫码数据初始化（步）
D1003.02 BOOL  ; 上料拉带扫码触发
D1003.03 BOOL  ; 上料拉带扫码结果等待
D1003.04 BOOL  ; 上料隔离气缸伸出
D1003.05 BOOL  ; 上料拉带扫码阻挡气缸缩回
D1003.06 BOOL  ; 等待扫码完成电池通过
D1003.07 BOOL  ; 上料拉带扫码阻挡气缸伸出
D1003.08 BOOL  ; 上料隔离气缸缩回
D1003.09 BOOL  ; 等待扫码位来料
D1003.10 BOOL  ; 上料步序循环结束
D1003.11 BOOL  ; 上料拉带停止
D1003.12 BOOL  ; 预留
D1003.13 BOOL  ; 1
D1005.00 BOOL  ; 上料拉带扫码单步运行
D1005.01 BOOL  ; 上料拉带单步/自动运行
D1006.00 BOOL  ; 上料拉带扫码单步/自动循环运行
D1006.10 BOOL  ; 上料拉带扫码工站记忆显示
D1006.13 BOOL  ; 上料工站记忆清除（SW）
D1006.14 BOOL  ; 上料工站复位按钮（SW）
D1006.15 BOOL  ; 上料机构单步（SW）
D1007 CHANNEL  ; 上料扫码步序号
D1007 CHANNEL  ; 进料拉带扫码步序号
D10100 CHANNEL  ; 进料扫码上料位控制字
D10101 CHANNEL  ; 进料拉带上料位条码（传递）
D1010.00 BOOL  ; 扫码NG抓取机构初始位
D1010.01 BOOL  ; 扫码NG抓取机构运行条件
D1010.02 BOOL  ; 扫码NG抓取机构忙绿标志
D1010.03 BOOL  ; 扫码NG抓取机构完成标志
D1010.04 BOOL  ; 清料带1阻挡气缸放料条件
D1010.05 BOOL  ; 扫码NG抓取机构停止标志
D1010.06 BOOL  ; 扫码NG抓取机构清料完成标志
D1010.07 BOOL  ; 扫码NG抓取机构异常标志
D1011.00 BOOL  ; 扫码NG抓取机构复位
D1011.01 BOOL  ; 扫码NG升降气缸缩回
D1011.02 BOOL  ; 扫码NG抓取夹爪松开
D1011.03 BOOL  ; 扫码NG抓取夹爪夹紧
D1011.04 BOOL  ; 扫码NG抓取无杆气缸缩回
D1011.05 BOOL  ; 扫码NG抓取阻挡气缸缩回
D1011.06 BOOL  ; 料盘拨料气缸复位
D1011.07 BOOL  ; 拉带阻挡气缸1缩回复位
D1012.00 BOOL  ; 扫码NG抓取机构开始运行条件
D1012.01 BOOL  ; 扫码NG抓取机构步进条件
D1012.15 BOOL  ; 扫码NG抓取机构步进
D1013 CHANNEL  ; 扫码NG抓取机构步序号
D1013.00 BOOL  ; 扫码NG抓取机构自动开始
D1013.01 BOOL  ; 拉带阻挡气缸1伸出
D1013.02 BOOL  ; 扫码NG抓取无杆气缸伸出
D1013.03 BOOL  ; 扫码NG抓取升降气缸伸出
D1013.04 BOOL  ; 扫码NG抓取夹爪夹紧
D1013.05 BOOL  ; 扫码NG抓取升降气缸缩回
D1013.06 BOOL  ; 拉带阻挡气缸1缩回
D1013.07 BOOL  ; 扫码NG抓取无杆气缸缩回
D1013.08 BOOL  ; 扫码NG放料拨料气缸伸出
D1013.09 BOOL  ; 扫码NG放料拨料气缸缩回
D1013.10 BOOL  ; 扫码NG抓取升降气缸伸出
D1013.11 BOOL  ; 扫码NG抓取夹爪松开
D1013.12 BOOL  ; 扫码NG抓取升降气缸缩回
D1013.13 BOOL  ; 扫码NG放料拨料气缸伸出
D1013.14 BOOL  ; 扫码NG放料拨料气缸缩回
D1013.15 BOOL  ; 扫码NG抓取步序完成
D1015.00 BOOL  ; 扫码NG抓取机构单步运行
D1015.01 BOOL  ; 扫码NG抓取机构单步/自动运行
D1016.00 BOOL  ; 扫码NG抓取机构单步/自动循环运行
D1016.10 BOOL  ; 扫码NG抓取工站记忆显示
D1016.13 BOOL  ; 扫码NG抓取工站记忆清除（SW）
D1016.14 BOOL  ; 扫码NG抓取工站复位按钮（SW）
D1016.15 BOOL  ; 扫码NG抓取工站单步（SW）
D10199 CHANNEL  ; 进料扫码上料位结束字
D102 CHANNEL  ; 入钉升降伺服安全高度位参数设定
D10200 CHANNEL  ; 清洁带阻挡1位控制字
D10201 CHANNEL  ; 清洁带阻挡1位控制字条码（传递）
D10299 CHANNEL  ; 清洁带阻挡1结束字
D10300 CHANNEL  ; 钉位清洁位控制字
D10301 CHANNEL  ; 钉位清洁位控制字条码（传递）
D1030.00 BOOL  ; 电池清洁机构初始位
D1030.01 BOOL  ; 电池清洁机构运行条件C
D1030.02 BOOL  ; 电池清洁机构忙绿标志
D1030.03 BOOL  ; 电池清洁机构完成标志
D1030.05 BOOL  ; 电池清洁机构停止标志
D1030.06 BOOL  ; 电池清洁机构清料完成标志
D1030.07 BOOL  ; 电池清洁机构异常标志
D1030.08 BOOL  ; 清洁机构运行条件A
D1030.09 BOOL  ; 清洁机构运行条件B
D1031.00 BOOL  ; 电池清洁机构复位
D1031.01 BOOL  ; 擦拭升降气缸缩回
D1031.02 BOOL  ; 阻挡气缸1伸出复位
D1031.03 BOOL  ; 阻挡气缸2伸出复位
D1031.04 BOOL  ; 精定位气缸1缩回复位
D1031.05 BOOL  ; 精定位气缸2缩回
D1031.06 BOOL  ; 精定位气缸1伸出复位
D1031.07 BOOL  ; 精定位气缸2伸出复位
D1031.08 BOOL  ; 擦拭步进复位
D1031.09 BOOL  ; 拉带阻挡气缸1复位缩回
D1031.10 BOOL  ; 拉带阻挡气缸2复位缩回
D1032.00 BOOL  ; 电池清洁机构开始运行条件
D1032.01 BOOL  ; 电池清洁机构步进条件
D1032.15 BOOL  ; 1
D1033 CHANNEL  ; 电池清洁机构步序号
D1033.00 BOOL  ; 电池清洁机构自动开始
D1033.01 BOOL  ; 拉带阻挡2气缸伸出
D1033.02 BOOL  ; 清洁拉带运行
D1033.03 BOOL  ; 清洁拉带停止
D1033.04 BOOL  ; 电池清洁机构精定位A2伸出
D1033.05 BOOL  ; 电池清洁机构精定位A1伸出
D1033.06 BOOL  ; 电池清洁机构擦拭升降气缸伸出
D1033.07 BOOL  ; 电池清洁机构擦拭步进启动
D1033.08 BOOL  ; 电池清洁机构擦拭升降气缸缩回
D1033.09 BOOL  ; 电池清洁机构精定位A1缩回
D1033.10 BOOL  ; 电池清洁机构精定位A2缩回
D1033.11 BOOL  ; 拉带阻挡气缸2缩回
D1033.12 BOOL  ; 擦拭完成拉带2启动
D1033.13 BOOL  ; 擦拭完成拉带2停止
D1033.14 BOOL  ; 预留
D1033.15 BOOL  ; 清洁机构步序结束
D1034.15 BOOL  ; 电池清洁机构步进
D1035.00 BOOL  ; 电池清洁机构单步运行
D1035.01 BOOL  ; 电池清洁机构单步/自动循环运行中
D1036.00 BOOL  ; 电池清洁机构单步/自动循环运行
D1036.10 BOOL  ; 钉位清洁工站记忆显示
D1036.13 BOOL  ; 钉位清洁工站记忆清除（SW）
D1036.14 BOOL  ; 钉位清洁工站复位按钮（SW）
D1036.15 BOOL  ; 钉位清洁工站单步（SW）
D1037 CHANNEL  ; 进料拉带扫码步序号
D10399 CHANNEL  ; 钉位清洁位结束字
D104 CHANNEL  ; 入钉升降伺服入钉位参数设定
D10400 CHANNEL  ; 电池入钉位控制字
D10401 CHANNEL  ; 电池入钉位条码（传递）
D1047.00 BOOL  ; 进料拉带扫码工站复位（M）
D1047.01 BOOL  ; 扫码阻挡气缸缩回（复位）
D1047.02 BOOL  ; 扫码阻挡气缸伸出（复位）
D1047.03 BOOL  ; 隔离气缸缩回（复位）
D1047.04 BOOL  ; 隔离气缸伸出（复位）
D10499 CHANNEL  ; 电池入钉位结束字
D1050.00 BOOL  ; 电池入钉机构初始位
D1050.01 BOOL  ; 电池入钉机构运行条件A
D1050.02 BOOL  ; 电池入钉机构忙绿标志
D1050.03 BOOL  ; 电池入钉机构完成标志
D1050.04 BOOL  ; 备钉机构初始位
D1050.05 BOOL  ; 备钉机构运行条件
D1050.06 BOOL  ; 电池入钉机构清料完成标志
D1050.07 BOOL  ; 电池入钉机构异常标志
D1050.08 BOOL  ; 电池入钉机构运行条件B
D1050.10 BOOL  ; 电池清洁机构停止标志
D1050.11 BOOL  ; 电池入钉机构清料完成标志
D1050.12 BOOL  ; 电池入钉机构异常标志
D1050.13 BOOL  ; 备钉钉机构异常标志
D1051.00 BOOL  ; 电池入钉机构复位
D1051.01 BOOL  ; 入钉升降伺服归零
D1051.02 BOOL  ; 入钉升降伺服至安全高度位
D1051.03 BOOL  ; 入钉精定位气缸B1缩回复位
D1051.04 BOOL  ; 入钉精定位气缸B2缩回复位
D1051.05 BOOL  ; 入钉精定位气缸B1伸出复位
D1051.06 BOOL  ; 入钉精定位气缸B2伸出复位
D1051.07 BOOL  ; 入钉压钉气缸缩回复位
D1051.08 BOOL  ; 入钉料盘拨料气缸1缩回复位
D1051.09 BOOL  ; 入钉料盘拨料气缸2缩回复位
D1051.10 BOOL  ; 入钉推钉X轴气缸缩回复位
D1051.11 BOOL  ; 入钉推钉Y轴气缸缩回复位
D1051.12 BOOL  ; 入钉阻挡3缩回复位
D1051.13 BOOL  ; 入钉真空关闭复位
D1051.14 BOOL  ; 入钉吹气关闭复位
D1051.15 BOOL  ; 振动盘关闭复位
D1052.00 BOOL  ; 备钉机构开始运行条件
D1052.01 BOOL  ; 备钉机构步进条件
D1052.02 BOOL  ; 阻挡2伸出复位
D1052.03 BOOL  ; 入钉阻挡4缩回复位
D1052.04 BOOL  ; $?St$Bk?_#[19] / 电池入钉机构开始运行条件 / $?St$Bk?_#[19]
D1052.05 BOOL  ; $?St$Bk?_#[20] / 电池入钉机构步进条件 / $?St$Bk?_#[20]
D1052.14 BOOL  ; 备点机构步进
D1052.15 BOOL  ; 电池入钉机构步进
D1053 CHANNEL  ; 备钉机构步序
D1053.00 BOOL  ; 备钉机构自动步序开始
D1053.01 BOOL  ; 震动盘启动
D1053.02 BOOL  ; 震动盘停止
D1053.03 BOOL  ; 入钉真空打开
D1053.04 BOOL  ; 预留
D1053.05 BOOL  ; 推钉Y轴伸出
D1053.06 BOOL  ; 推钉X轴伸出
D1053.07 BOOL  ; 真空关闭
D1053.08 BOOL  ; 入钉吹气打开
D1053.09 BOOL  ; 入钉吹气关闭
D1053.10 BOOL  ; 推钉X轴缩回
D1053.11 BOOL  ; 推钉Y轴缩回
D1053.12 BOOL  ; 预留
D1053.13 BOOL  ; 备钉机构步序结束
D1053.14 BOOL  ; 1
D1053.15 BOOL  ; 1
D1054 CHANNEL  ; 入钉机构步序
D1054.00 BOOL  ; 入钉机构自动开始
D1054.01 BOOL  ; 入钉阻挡气缸3伸出
D1054.02 BOOL  ; 入钉拉带停止
D1054.03 BOOL  ; 精定位气缸B2夹紧
D1054.04 BOOL  ; 精定位气缸B1夹紧
D1054.05 BOOL  ; 入钉升降伺服至入钉位
D1054.06 BOOL  ; 压钉伸出 启动入钉旋转步进
D1054.07 BOOL  ; 入钉升降伺服至安全高度位
D1054.08 BOOL  ; 压钉气缸缩回
D1054.09 BOOL  ; 监测入钉状况
D1054.10 BOOL  ; 精定位气缸B1松开
D1054.11 BOOL  ; 精定位气缸B2松开
D1054.12 BOOL  ; 入钉OK NG处理
D1054.13 BOOL  ; 入钉阻挡气缸3缩回
D1054.14 BOOL  ; 入钉拉带启动
D1054.15 BOOL  ; 入钉拉带停止
D1055.00 BOOL  ; 入钉阻挡气缸4伸出
D1055.01 BOOL  ; 入钉拉带启动
D1055.02 BOOL  ; 入钉拉带停止
D1055.03 BOOL  ; 入钉阻挡气缸4缩回
D1055.04 BOOL  ; 入钉机构步序结束
D1056.00 BOOL  ; 电池入钉机构单步/自动循环运行
D1056.01 BOOL  ; $?St$Bk?_#[21] / 电池入钉机构单步运行 / $?St$Bk?_#[21]
D1056.02 BOOL  ; $?St$Bk?_#[22] / 电池入钉机构单步/自动循环运行中 / $?St$Bk?_#[22]
D1056.04 BOOL  ; 电池入钉备钉运行
D1056.05 BOOL  ; 电池入钉备钉自动运行
D1056.14 BOOL  ; $?St$Bk?_#[23] / 电池入钉工站复位按钮（SW） / $?St$Bk?_#[23]
D1056.15 BOOL  ; $?St$Bk?_#[24] / 电池入钉工站单步（SW） / $?St$Bk?_#[24]
D1059.00 BOOL  ; 入钉阻挡2伸出复位
D106 CHANNEL  ; 进料水平伺服左爪缓存位参数设定 (M)
D108 CHANNEL  ; 进料水平伺服右爪缓存位参数设定 (M)
D1080.00 BOOL  ; 入钉NG抓取机构初始位
D1080.01 BOOL  ; 入钉NG抓取机构运行条件
D1080.02 BOOL  ; 入钉NG抓取机构忙绿标志
D1080.03 BOOL  ; 入钉NG抓取机构完成标志
D1080.05 BOOL  ; 入钉NG抓取机构停止标志
D1080.06 BOOL  ; 入钉NG抓取机构清料完成标志
D1080.07 BOOL  ; 入钉NG抓取机构异常标志
D1081.00 BOOL  ; 入钉NG抓取机构工站复位
D1081.01 BOOL  ; 入钉NG抓取升降气缸缩回复位
D1081.02 BOOL  ; 入钉NG抓取夹爪松开复位
D1081.03 BOOL  ; 入钉NG抓取夹爪夹紧复位
D1081.04 BOOL  ; 入钉NG抓取无杆气缸缩回复位
D1081.05 BOOL  ; 入钉阻挡气缸4伸出复位
D1081.06 BOOL  ; 入钉阻挡气缸4缩回复位
D1082.00 BOOL  ; 入钉NG抓取机构开始运行条件
D1082.01 BOOL  ; 入钉NG抓取机构步进条件
D1082.15 BOOL  ; 入钉NG抓取机构步进
D1083 CHANNEL  ; 入钉NG抓取机构步序号
D1083.00 BOOL  ; 入钉NG抓取机构自动开始
D1083.01 BOOL  ; 入钉NG抓取条件
D1083.02 BOOL  ; 无杆气缸伸出
D1083.03 BOOL  ; 入钉NG抓取升降气缸伸出
D1083.04 BOOL  ; 入钉NG抓取夹爪夹紧
D1083.05 BOOL  ; 入钉NG抓取升降气缸缩回
D1083.06 BOOL  ; 入钉NG抓取无杆气缸缩回
D1083.07 BOOL  ; 入钉NG放料B拨料气缸伸出
D1083.08 BOOL  ; 入钉NG放料B拨料气缸缩回
D1083.09 BOOL  ; 入钉NG抓取升降气缸伸出
D1083.10 BOOL  ; 入钉NG抓取夹爪松开
D1083.11 BOOL  ; 入钉NG抓取升降气缸缩回
D1083.12 BOOL  ; 入钉NG放料B拨料气缸伸出
D1083.13 BOOL  ; 入钉NG放料B拨料气缸缩回
D1083.14 BOOL  ; 入钉NG抓取步序完成
D1085.00 BOOL  ; 入钉NG抓取机构单步运行
D1085.01 BOOL  ; 入钉NG抓取机构单步/自动运行
D1086.00 BOOL  ; 入钉NG抓取机构单步/自动循环运行
D1086.10 BOOL  ; 入钉NG抓取工站记忆显示
D1086.13 BOOL  ; 入钉NG抓取工站记忆清除（SW）
D1086.14 BOOL  ; 入钉NG抓取工站复位按钮（SW）
D1086.15 BOOL  ; 入钉NG抓取工站单步（SW）
D10.00 BOOL  ; 扫码来料记忆清除HIM
D10.02 BOOL  ; 扫码OK记忆清除HIM
D10.03 BOOL  ; 扫码NG记忆清除HIM
D10.04 BOOL  ; 拉带放料中记忆清除HIM
D10.06 BOOL  ; $?St$Bk?_#[25] / 扫码拉带放料完成 / 记忆清除HIM$?St$Bk?_#[25]
D110 CHANNEL  ; 进料水平伺服NG位参数设定 (M)
D1110.00 BOOL  ; 3#氦检机构初始位
D1110.06 BOOL  ; 3#氦检机构清料完成标志
D1110.07 BOOL  ; 3#氦检机构异常标志
D1140.00 BOOL  ; 上下料机械手初始位
D1140.06 BOOL  ; 上下料机械手清料完成标志
D1140.07 BOOL  ; 上下料机械手异常标志
D118 CHANNEL  ; 进料水平伺服放料位参数设定 (M)
D12 CHANNEL  ; 入钉升降伺服手动速度   HMI
D128 CHANNEL  ; 进料升降伺服待料位参数设定
D136 CHANNEL  ; 入钉旋转步进脉冲参数设定 (M)
D14 CHANNEL  ; 感应器ON延时设定值
D144 CHANNEL  ; 下料水平伺服#2腔体位参数设定 (M)
D146 CHANNEL  ; 擦拭步进擦拭位参数设定 (M)
D14 CHANNEL  ; 感应延时
D16 CHANNEL  ; 感应器延时时间
D16 CHANNEL  ; 延时设定值
D18 CHANNEL  ; 自动运行条件延时时间
D19 CHANNEL  ; 自动运行步间间隔时间
D20.01 BOOL  ; 拉带有OK料记忆清除HIM
D20.02 BOOL  ; 拉带有NG料记忆清除HIM
D20.04 BOOL  ; 扫码NG夹爪记忆清除HIM
D22 CHANNEL  ; 报警长延时
D24 CHANNEL  ; 入钉旋转步进手动速度   HMI
D2501 CHANNEL  ; 扫码阻挡气缸到位延时设定值
D26 CHANNEL  ; 擦拭步进自动速度   HMI
D28 CHANNEL  ; 擦拭步进手动速度   HMI
D30 CHANNEL  ; 入钉旋转步进自动速度   HMI
D3000 CHANNEL  ; 总数
D3002 CHANNEL  ; 良品数
D30027 CHANNEL  ; PA1 Response Code
D3004 CHANNEL  ; 扫码NG不良品数
D3006 CHANNEL  ; 入钉NG不良品数
D3008 CHANNEL  ; 不良品总数
D30128 CHANNEL  ; Socket2 b0-7socket num b8-15 socket option
D30129 CHANNEL  ; Socket2 Local UDP/TCP port num
D30130 CHANNEL  ; Socket2 Remote IP Adds1~2
D30131 CHANNEL  ; Socket2 Remote IP Adds3~4
D30132 CHANNEL  ; Socket2 Remote UDP/TCP port number
D30133 CHANNEL  ; Socket2 num of send/rev bytes
D30134 CHANNEL  ; Socket2 b8-15 Area designation b0-7 leftmost 2 digits
D30135 CHANNEL  ; Socket2 b8-15 right2digits of word b0-7adds bit num=00
D30136 CHANNEL  ; Socket2 Timeout value
D30137 CHANNEL  ; Socket2 Response code
D30.01 BOOL  ; 钉位清洁完成记忆HIM
D30.05 BOOL  ; 钉位清洁记忆清除HIM
D30.07 BOOL  ; $?St$Bk?_#[26] / 钉位清洁完成放料 / 记忆清除HIM$?St$Bk?_#[26]
D4000 CHANNEL  ; 扫码枪发送字符区
D4002.00 BOOL  ; 1扫码接收中
D4002.01 BOOL  ; 1扫码数据接收比较
D4002.02 BOOL  ; 接收完成
D4003 CHANNEL  ; 1扫码字符数
D4004 CHANNEL  ; $?St$Bk?_#[27] / "OK"$?St$Bk?_#[27]
D4010 CHANNEL  ; 扫码枪1接收OKorNG
D402 CHANNEL  ; 轴控预留量
D4050 CHANNEL  ; 替换条码（0D0A）起始位置
D4058 CHANNEL  ; =空
D4060 CHANNEL  ; 截取条码
D40.01 BOOL  ; 电池入钉记忆清除HIM
D40.02 BOOL  ; 入钉OK记忆清除HIM
D40.03 BOOL  ; 入钉NG记忆清除HIM
D40.09 BOOL  ; 管嘴有钉记忆清除HIM
D416 CHANNEL  ; 入钉升降伺服当前脉冲
D426 CHANNEL  ; 进料升降伺服当前脉冲
D446 CHANNEL  ; 入钉旋转步进当前脉冲
D456 CHANNEL  ; 擦拭步进当前脉冲
D50 CHANNEL  ; 总产量
D500 CHANNEL  ; 入钉升降伺服自动状态加速比率
D501 CHANNEL  ; 入钉升降伺服自动状态减速比率
D502 CHANNEL  ; 入钉升降伺服自动状态目标频率（低位）
D504 CHANNEL  ; 入钉升降伺服自动状态脉冲输出量（低位）
D506 CHANNEL  ; 入钉升降伺服自动状态启动频率（低位）
D50.04 BOOL  ; 入钉NG夹爪记忆清除HIM
D5100 CHANNEL  ; 扫码长度
D52 CHANNEL  ; 检测OK产量
D530 CHANNEL  ; 入钉旋转步进自动状态加速比率
D531 CHANNEL  ; 入钉旋转步进自动状态减速比率
D532 CHANNEL  ; 入钉旋转步进自动状态目标频率（低位）
D534 CHANNEL  ; 入钉旋转入钉位自动状态脉冲输出量（低位）
D536 CHANNEL  ; 入钉旋转步进自动状态启动频率（低位）
D54 CHANNEL  ; 检测NG产量
D540 CHANNEL  ; 擦拭步进自动状态加速比率
D541 CHANNEL  ; 擦拭步进自动状态减速比率
D542 CHANNEL  ; 擦拭步进自动状态目标频率（低位）
D544 CHANNEL  ; 擦拭步进自动状态脉冲输出量（低位）
D546 CHANNEL  ; 擦拭步进自动状态启动频率（低位）
D58 CHANNEL  ; 检测总量
D60 CHANNEL  ; 接收条码数据字长度
D600 CHANNEL  ; 入钉升降伺服手动状态加速比率
D601 CHANNEL  ; 入钉升降伺服手动状态减速比率
D602 CHANNEL  ; 入钉升降伺服手动状态目标频率（低位）
D604 CHANNEL  ; 入钉升降伺服手动状态脉冲输出量（低位）
D606 CHANNEL  ; 入钉升降伺服手动状态启动频率（低位）
D62 CHANNEL  ; 1扫码字符实际读取长度
D630 CHANNEL  ; 入钉旋转步进手动状态加速比率
D631 CHANNEL  ; 入钉旋转步进手动状态减速比率
D632 CHANNEL  ; 入钉旋转步进手动状态目标频率（低位）
D634 CHANNEL  ; 入钉深度手动状态脉冲输出量（低位）
D636 CHANNEL  ; 入钉旋转步进手动状态启动频率（低位）
D640 CHANNEL  ; 擦拭步进动状态加速比率
D641 CHANNEL  ; 擦拭步进手动状态减速比率
D642 CHANNEL  ; 擦拭步进手动状态目标频率（低位）
D644 CHANNEL  ; 擦拭步进手动状态脉冲输出量（低位）
D646 CHANNEL  ; 擦拭步进手动状态启动频率（低位）
D66 CHANNEL  ; 设定条码长度
D68 CHANNEL  ; 设定条码字长度
D7897 CHANNEL  ; NG扫码重试次数设置
D7899 CHANNEL  ; PC通信标志
H100.00 BOOL  ; 扫码阻挡气缸1原位屏蔽
H100.01 BOOL  ; 扫码阻挡气缸1到位屏蔽
H100.02 BOOL  ; 扫码阻挡气缸2原位屏蔽
H100.03 BOOL  ; 扫码阻挡气缸2到位屏蔽
H100.04 BOOL  ; 隔离气缸1原位屏蔽
H100.05 BOOL  ; 隔离气缸1到位屏蔽
H100.06 BOOL  ; 隔离气缸2原位屏蔽
H100.07 BOOL  ; 隔离气缸2到位屏蔽
H100.08 BOOL  ; 进料对射光电屏蔽
H100.09 BOOL  ; 夹爪A1夹紧位屏蔽
H100.10 BOOL  ; 夹爪A1松开位屏蔽
H100.11 BOOL  ; 夹爪A2夹紧位屏蔽
H100.12 BOOL  ; 夹爪A2松开位屏蔽
H100.13 BOOL  ; 夹爪B1夹紧位屏蔽
H100.14 BOOL  ; 夹爪B1松开位屏蔽
H100.15 BOOL  ; 夹爪B2夹紧位屏蔽
H101.00 BOOL  ; 夹爪B2松开位屏蔽
H101.01 BOOL  ; NG升降气缸1原位屏蔽
H101.02 BOOL  ; NG升降气缸1到位屏蔽
H101.03 BOOL  ; NG升降气缸2原位屏蔽
H101.04 BOOL  ; NG升降气缸2到位屏蔽
H101.05 BOOL  ; 无杆气缸1原位屏蔽
H101.06 BOOL  ; 无杆气缸1到位屏蔽
H101.07 BOOL  ; 无杆气缸2原位屏蔽
H101.08 BOOL  ; 无杆气缸2到位屏蔽
H101.09 BOOL  ; 阻挡伸出气缸1原位屏蔽
H101.10 BOOL  ; 阻挡伸出气缸1到位屏蔽
H101.11 BOOL  ; 阻挡伸出气缸2原位屏蔽
H101.12 BOOL  ; 阻挡伸出气缸2到位屏蔽
H101.13 BOOL  ; 阻挡伸出气缸3原位屏蔽
H101.14 BOOL  ; 阻挡伸出气缸3到位屏蔽
H101.15 BOOL  ; 阻挡伸出气缸4原位屏蔽
H102.00 BOOL  ; 阻挡伸出气缸4到位屏蔽
H102.01 BOOL  ; 精定位气缸A1原位屏蔽
H102.02 BOOL  ; 精定位气缸A1到位屏蔽
H102.03 BOOL  ; 精定位气缸A2原位屏蔽
H102.04 BOOL  ; 精定位气缸A2到位屏蔽
H102.05 BOOL  ; 精定位气缸B1原位屏蔽
H102.06 BOOL  ; 精定位气缸B1到位屏蔽
H102.07 BOOL  ; 精定位气缸B2原位屏蔽
H102.08 BOOL  ; 精定位气缸B2到位屏蔽
H102.09 BOOL  ; 擦拭升降气缸原位屏蔽
H102.10 BOOL  ; 擦拭升降气缸到位屏蔽
H102.11 BOOL  ; 压钉气缸原位屏蔽
H102.12 BOOL  ; 压钉气缸到位屏蔽
H102.13 BOOL  ; 料盒拨料气缸1原位屏蔽
H102.14 BOOL  ; 料盒拨料气缸1到位屏蔽
H102.15 BOOL  ; 料盒拨料气缸2原位屏蔽
H103.00 BOOL  ; 料盒拨料气缸2到位屏蔽
H103.01 BOOL  ; 推钉X轴气缸原位屏蔽
H103.02 BOOL  ; 推钉X轴气缸到位屏蔽
H103.03 BOOL  ; 推钉Y轴气缸原位屏蔽
H103.04 BOOL  ; 推钉Y轴气缸到位屏蔽
H103.05 BOOL  ; 扫码位对射光电屏蔽
H103.06 BOOL  ; 分隔电池对射光电屏蔽
H103.07 BOOL  ; 光电屏蔽
H103.08 BOOL  ; 光电屏蔽
H103.09 BOOL  ; 擦拭带盘无料感应屏蔽
H103.10 BOOL  ; 扫码NG位对射光电屏蔽
H103.11 BOOL  ; 擦拭位对射光电屏蔽
H103.12 BOOL  ; 入钉位对射光电屏蔽
H103.13 BOOL  ; 入钉NG位对射光电屏蔽
H103.14 BOOL  ; 扫码NG槽对射前光电屏蔽
H103.15 BOOL  ; 入钉NG槽对射前光电屏蔽
H104.00 BOOL  ; 扫码NG槽对射光电屏蔽
H104.01 BOOL  ; 入钉NG槽对射后屏蔽
H104.02 BOOL  ; $?St$Bk?_#[28] / 入钉检测区域光纤屏蔽 / $?St$Bk?_#[28]
H104.03 BOOL  ; 入钉伺服就绪 屏蔽
H104.04 BOOL  ; 入钉伺服报警 屏蔽
H104.05 BOOL  ; 启动按钮屏蔽
H104.06 BOOL  ; 停止按钮屏蔽
H104.07 BOOL  ; 复位按钮屏蔽
H104.08 BOOL  ; 急停按钮屏蔽
H104.09 BOOL  ; 手自动选择屏蔽
H104.10 BOOL  ; 设备总气压屏蔽
H104.11 BOOL  ; 夹爪1柔性报警屏蔽
H104.12 BOOL  ; 夹爪2柔性报警屏蔽
H104.13 BOOL  ; 真空信号屏蔽
H104.14 BOOL  ; 开关电源监测屏蔽
H104.15 BOOL  ; 变频器监测屏蔽
H105.00 BOOL  ; NG门磁开关屏蔽
H105.01 BOOL  ; 前门磁开关屏蔽
H105.02 BOOL  ; 后门磁开关屏蔽
H105.03 BOOL  ; 左门磁开关屏蔽
H105.04 BOOL  ; 右门磁开关屏蔽
H105.05 BOOL  ; $?St$Bk?_#[29] / 区域光纤对射屏蔽 / $?St$Bk?_#[29]
H105.06 BOOL  ; $?St$Bk?_#[30] / 钉位钉子对射光纤屏蔽 / $?St$Bk?_#[30]
H105.07 BOOL  ; 震盘钉嘴反射光纤屏蔽
H105.08 BOOL  ; 拉带入口对射光电屏蔽
H10.00 BOOL  ; 扫码阻挡有料记忆
H10.01 BOOL  ; 扫码完成记忆
H10.02 BOOL  ; 扫码OK记忆
H10.03 BOOL  ; 扫码NG记忆
H10.04 BOOL  ; 上料拉带放料中记忆
H10.05 BOOL  ; 隔离缩回启动拉带
H10.06 BOOL  ; 进料拉带放料完成
H10.08 BOOL  ; 触发扫码NG抓取
H10.10 BOOL  ; 空跑程序
H11.00 BOOL  ; 电脑屏蔽-HMI
H20.00 BOOL  ; 拉带来料记忆
H20.01 BOOL  ; 拉带有扫码OK料记忆
H20.02 BOOL  ; 拉带有扫码NG料记忆
H20.03 BOOL  ; 上料位有扫码NG料记忆
H20.04 BOOL  ; NG抓取夹爪有料记忆
H20.05 BOOL  ; 扫码NG抓取机构忙绿标志
H20.07 BOOL  ; 等待电池清洁处理
H20.10 BOOL  ; 扫码NG抓取机构完成标志
H22.01 BOOL  ; 下料位有料记忆
H25.00 BOOL  ; 进料水平伺服归零完成
H25.01 BOOL  ; 进料升降伺服归零完成
H25.03 BOOL  ; 上料水平伺服归零完成
H25.13 BOOL  ; 断腔体上料伺服归零
H26.01 BOOL  ; 1#腔体有料记忆
H30.00 BOOL  ; 电池清洁完成记忆
H30.01 BOOL  ; 电池清洁完成记忆
H30.05 BOOL  ; 电池清洁机构忙绿标志
H30.07 BOOL  ; 电池擦拭完成放料中
H30.10 BOOL  ; 电池清洁机构完成标志
H31.01 BOOL  ; 2#腔体有料记忆
H36.01 BOOL  ; 3#腔体有料记忆
H3.04 BOOL  ; 扫码屏蔽_1=屏蔽（SW）
H3.05 BOOL  ; 空跑模式
H3.06 BOOL  ; 空跑扫码屏蔽
H40.00 BOOL  ; 入钉升降伺服归零
H40.01 BOOL  ; 电池入钉记忆
H40.02 BOOL  ; 电池入钉OK记忆
H40.03 BOOL  ; 电池入钉NG记忆
H40.04 BOOL  ; 备钉机构忙绿标志
H40.05 BOOL  ; 电池入钉机构忙绿标志
H40.06 BOOL  ; 压钉进行中
H40.07 BOOL  ; 入钉记忆跳步中
H40.08 BOOL  ; 入钉拉带启动
H40.09 BOOL  ; 有钉标志
H40.10 BOOL  ; 电池入钉机构完成标志
H40.11 BOOL  ; 入钉拉带启动
H40.12 BOOL  ; 触发NG机构抓取
H40.13 BOOL  ; 入钉OK电池放料中
H40.14 BOOL  ; 入钉拉带停止标志
H45.01 BOOL  ; 下料夹爪有料记忆
H50.04 BOOL  ; 入钉NG抓取夹爪有料记忆
H50.05 BOOL  ; 入钉NG抓取忙绿标志
H50.10 BOOL  ; 入钉NG抓取机构完成标志
H55.00 BOOL  ; 1#入料扫码完成记忆
H55.02 BOOL  ; 1#入料扫码OK记忆
H55.03 BOOL  ; 1#入料扫码NG记忆
H8.00 BOOL  ; 门磁屏蔽（SW）
H8.02 BOOL  ; 震动盘屏蔽
H8.04 BOOL  ; 扫码屏蔽
H8.06 BOOL  ; 上料拉带重新扫码模式选择（0=使用/1=屏蔽）
H8.08 BOOL  ; 入钉升降伺服回零标志
H8.10 BOOL  ; 空跑程序
T0000 BOOL  ; PLC上电延时100ms
T0001 BOOL  ; 手动模式延时
T0002 BOOL  ; 自动模式延时
T0006 BOOL  ; 复位延时
T0007 BOOL  ; 自动停止完成延时
T0008 BOOL  ; 启动延时
T0009 BOOL  ; 停止延时
T0010 BOOL  ; PLC RUN
T0011 BOOL  ; 左入料扫码延时
T0012 BOOL  ; 扫码位单粒电池启动延时
T0015 BOOL  ; 1扫码接收延时
T0017 BOOL  ; 入钉拉带启动延时
T0018 BOOL  ; 擦拭拉带启动延时
T0019 BOOL  ; 清料停止完成延时
T0021 BOOL  ; 整机在初始位延时
T0022 BOOL  ; 报警发送延时时间
T0030 BOOL  ; 上料扫码数据初始化延时
T0031 BOOL  ; 扫码延时
T0032 BOOL  ; 扫码长度判定延时
T0048 BOOL  ; PC运行标志断开时间
T0049 BOOL  ; PC通信正常持续时间
T0050 BOOL  ; 蜂鸣器延时停止
T0100 BOOL  ; 扫码阻挡气缸1原位报警延时
T0101 BOOL  ; 扫码阻挡气缸1到位报警延时
T0102 BOOL  ; 扫码阻挡气缸2原位报警延时
T0103 BOOL  ; 扫码阻挡气缸2到位报警延时
T0104 BOOL  ; 隔离气缸1原位报警延时
T0105 BOOL  ; 隔离气缸1到位报警延时
T0106 BOOL  ; 隔离气缸2原位报警延时
T0107 BOOL  ; 隔离气缸2到位报警延时
T0108 BOOL  ; 进料对射光电报警延时
T0109 BOOL  ; 夹爪A1夹紧位报警延时
T0110 BOOL  ; 夹爪A1松开位报警延时
T0111 BOOL  ; 夹爪A2夹紧位报警延时
T0112 BOOL  ; 夹爪A2松开位报警延时
T0113 BOOL  ; 夹爪B1夹紧位报警延时
T0114 BOOL  ; 夹爪B1松开位报警延时
T0115 BOOL  ; 夹爪B2夹紧位报警延时
T0116 BOOL  ; 夹爪B2松开位报警延时
T0117 BOOL  ; NG升降气缸1原位报警延时
T0118 BOOL  ; NG升降气缸1到位报警延时
T0119 BOOL  ; NG升降气缸2原位报警延时
T0120 BOOL  ; NG升降气缸2到位报警延时
T0121 BOOL  ; NG无杆气缸1原位报警延时
T0122 BOOL  ; NG无杆气缸1到位报警延时
T0123 BOOL  ; NG无杆气缸2原位报警延时
T0124 BOOL  ; NG无杆气缸2到位报警延时
T0125 BOOL  ; 阻挡伸出气缸1原位报警延时
T0126 BOOL  ; 阻挡伸出气缸1到位报警延时
T0127 BOOL  ; 阻挡伸出气缸2原位报警延时
T0128 BOOL  ; 阻挡伸出气缸2到位报警延时
T0129 BOOL  ; 阻挡伸出气缸3原位报警延时
T0130 BOOL  ; 阻挡伸出气缸3到位报警延时
T0131 BOOL  ; 阻挡伸出气缸4原位报警延时
T0132 BOOL  ; 阻挡伸出气缸4到位报警延时
T0133 BOOL  ; 精定位气缸A1原位报警延时
T0134 BOOL  ; 精定位气缸A1到位报警延时
T0135 BOOL  ; 精定位气缸A2原位报警延时
T0136 BOOL  ; 精定位气缸A2到位报警延时
T0137 BOOL  ; 精定位气缸B1原位报警延时
T0138 BOOL  ; 精定位气缸B1到位报警延时
T0139 BOOL  ; 精定位气缸B2原位报警延时
T0140 BOOL  ; 精定位气缸B2到位报警延时
T0141 BOOL  ; 擦拭升降气缸原位报警延时
T0142 BOOL  ; 擦拭升降气缸到位报警延时
T0143 BOOL  ; 压钉气缸原位报警延时
T0144 BOOL  ; 压钉气缸到位报警延时
T0145 BOOL  ; 料盒拨料气缸1原位报警延时
T0146 BOOL  ; 料盒拨料气缸1到位报警延时
T0147 BOOL  ; 料盒拨料气缸2原位报警延时
T0148 BOOL  ; 料盒拨料气缸2到位报警延时
T0149 BOOL  ; 推钉X轴气缸原位报警延时
T0150 BOOL  ; 推钉X轴气缸到位报警延时
T0151 BOOL  ; 推钉Y轴气缸原位报警延时
T0152 BOOL  ; 推钉Y轴气缸到位报警延时
T0153 BOOL  ; 扫码位对射光电报警延时
T0154 BOOL  ; 分隔电池对射光电报警延时
T0155 BOOL  ; 清洁拉带光电报警延时
T0156 BOOL  ; 入钉嘴对射光电来钉报警延时
T0157 BOOL  ; 料盘清洁带有料报警延时
T0158 BOOL  ; 扫码NG位对射光电报警延时
T0159 BOOL  ; 擦拭位对射光电报警延时
T0160 BOOL  ; 胶钉未射入，钉位对射光电报警延时
T0161 BOOL  ; 入钉NG位对射光电报警延时
T0162 BOOL  ; 扫码NG槽对射前光电报警延时
T0163 BOOL  ; 入钉NG槽对射前光电报警延时
T0164 BOOL  ; 扫码NG槽对射光电满料报警延时
T0165 BOOL  ; 入钉NG槽对射光电报警延时
T0166 BOOL  ; $?St$Bk?_#[31] / 入钉检测区域光纤报警延时 / $?St$Bk?_#[31]
T0167 BOOL  ; 入钉伺服就绪 报警延时
T0168 BOOL  ; 入钉伺服报警 报警延时
T0169 BOOL  ; 启动按钮报警延时
T0170 BOOL  ; 停止按钮报警延时
T0171 BOOL  ; 复位按钮报警延时
T0172 BOOL  ; 急停按钮报警延时
T0173 BOOL  ; 手自动选择报警延时
T0174 BOOL  ; 设备总气压报警延时
T0175 BOOL  ; 夹爪1柔性报警报警延时
T0176 BOOL  ; 夹爪2柔性报警报警延时
T0177 BOOL  ; 真空信号报警延时
T0178 BOOL  ; 开关电源监测报警延时
T0179 BOOL  ; 变频器监测报警延时
T0180 BOOL  ; NG门磁开关报警延时
T0181 BOOL  ; 前门磁开关报警延时
T0182 BOOL  ; 后门磁开关报警延时
T0183 BOOL  ; 左门磁开关报警延时
T0184 BOOL  ; 右门磁开关报警延时
T0185 BOOL  ; 入钉胶管有钉感应报警延时
T0186 BOOL  ; 吹钉入位对射光电报警延时
T0187 BOOL  ; 入钉前胶管有钉感应延时
T0188 BOOL  ; 入钉前胶管有钉记记延时
T0189 BOOL  ; 吹气入钉钉位无感应延时
T0190 BOOL  ; 吹气入钉管嘴内有钉记忆延时
T0192 BOOL  ; 管嘴有钉钉位无感应延时
T0193 BOOL  ; 管嘴内无钉记忆钉位有钉延时
T0200 BOOL  ; 入钉升降伺服准入钉位延时
T0201 BOOL  ; 自动回进料水平伺服左爪OK配对位辅助延时
T0202 BOOL  ; 入钉升降伺服安全高度位延时
T0203 BOOL  ; 入钉升降伺服入钉位延时
T0204 BOOL  ; 自动回进料水平伺服右爪缓存位辅助延时
T0205 BOOL  ; 自动回进料水平伺服缓存位辅助延时
T0209 BOOL  ; 自动回进料水平伺服放料位辅助延时
T0210 BOOL  ; 手动入钉升降伺服准入钉位延时
T0212 BOOL  ; 手动入钉升降伺服安全高度位延时
T0213 BOOL  ; 手动入钉升降伺服入钉位延时
T0215 BOOL  ; 入钉升降伺服归零延时
T0216 BOOL  ; 入钉升降伺服上升延时
T0217 BOOL  ; 入钉升降伺服下降延时
T0250 BOOL  ; 进料水平伺服归零辅助延时
T0251 BOOL  ; 进料水平伺服前进辅助延时
T0278 BOOL  ; 上料水平伺服前进辅助延时
T0279 BOOL  ; 上料水平伺服后退辅助延时
T0280 BOOL  ; 手动回上料料水平伺服待料位辅助延时
T0281 BOOL  ; 手动回上料料水平伺服#1腔体位辅助延时
T0284 BOOL  ; 下料水平伺服前进辅助延时
T0286 BOOL  ; 手动回下料水平伺服#1腔体位辅助延时
T0287 BOOL  ; 手动回下料水平伺服#2腔体位辅助延时
T0336 BOOL  ; 上料提升气缸缩回位延时
T0401 BOOL  ; 入钉真空阀打开延时
T0402 BOOL  ; $?St$Bk?_#[32] / 入钉真空阀关闭延时 / $?St$Bk?_#[32]
T0403 BOOL  ; 入钉吹气阀打开延时
T0404 BOOL  ; 入钉吹气阀关闭延时
T0500 BOOL  ; 扫码阻挡气缸1缩回延时[A]
T0501 BOOL  ; 扫码阻挡气缸1伸出延时[A]
T0502 BOOL  ; 扫码阻挡气缸2缩回延时[A]
T0503 BOOL  ; 扫码阻挡气缸2伸出延时[A]
T0504 BOOL  ; 隔离气缸1缩回延时[A]
T0505 BOOL  ; 隔离气缸1伸出延时[A]
T0506 BOOL  ; 隔离气缸2缩回延时[A]
T0507 BOOL  ; 隔离气缸2伸出延时[A]
T0508 BOOL  ; 进料拉带电机启动延时[A]
T0509 BOOL  ; 夹爪A1夹紧延时[A]
T0510 BOOL  ; 夹爪A1松开延时[A]
T0511 BOOL  ; 夹爪A2夹紧延时[A]
T0512 BOOL  ; 夹爪A2松开延时[A]
T0513 BOOL  ; 夹爪B1夹紧延时[A]
T0514 BOOL  ; 夹爪B1松开延时[A]
T0515 BOOL  ; 夹爪B2夹紧延时[A]
T0516 BOOL  ; 夹爪B2松开延时[A]
T0517 BOOL  ; NG升降气缸1缩回延时[A]
T0518 BOOL  ; NG升降气缸1伸出延时[A]
T0519 BOOL  ; NG升降气缸2缩回延时[A]
T0520 BOOL  ; NG升降气缸2伸出延时[A]
T0521 BOOL  ; 无杆气缸1缩回延时[A]
T0522 BOOL  ; 无杆气缸1伸出延时[A]
T0523 BOOL  ; 无杆气缸2缩回延时[A]
T0524 BOOL  ; 无杆气缸2伸出延时[A]
T0525 BOOL  ; 阻挡伸出气缸1缩回延时[A]
T0526 BOOL  ; 阻挡伸出气缸1伸出延时[A]
T0527 BOOL  ; 阻挡伸出气缸2缩回延时[A]
T0528 BOOL  ; 阻挡伸出气缸2伸出延时[A]
T0529 BOOL  ; 阻挡伸出气缸3缩回延时[A]
T0530 BOOL  ; 阻挡伸出气缸3伸出延时[A]
T0531 BOOL  ; 阻挡伸出气缸4缩回延时[A]
T0532 BOOL  ; 阻挡伸出气缸4伸出延时[A]
T0533 BOOL  ; 精定位气缸A1缩回延时[A]
T0534 BOOL  ; 精定位气缸A1伸出延时[A]
T0535 BOOL  ; 精定位气缸A2缩回延时[A]
T0536 BOOL  ; 精定位气缸A2伸出延时[A]
T0537 BOOL  ; 精定位气缸B1缩回延时[A]
T0538 BOOL  ; 精定位气缸B1伸出延时[A]
T0539 BOOL  ; 精定位气缸B2缩回延时[A]
T0540 BOOL  ; 精定位气缸B2伸出延时[A]
T0541 BOOL  ; 擦拭升降气缸缩回延时[A]
T0542 BOOL  ; 擦拭升降气缸伸出延时[A]
T0543 BOOL  ; 压钉气缸缩回延时[A]
T0544 BOOL  ; 压钉气缸伸出延时[A]
T0545 BOOL  ; 料盒拨料气缸1缩回延时[A]
T0546 BOOL  ; 料盒拨料气缸1伸出延时[A]
T0547 BOOL  ; 料盒拨料气缸2缩回延时[A]
T0548 BOOL  ; 料盒拨料气缸2伸出延时[A]
T0549 BOOL  ; 推钉X轴气缸缩回延时[A]
T0550 BOOL  ; 推钉X轴气缸伸出延时[A]
T0551 BOOL  ; 推钉Y轴气缸缩回延时[A]
T0552 BOOL  ; 推钉Y轴气缸伸出延时[A]
T0553 BOOL  ; $?St$Bk?_#[33] / 钉位清洁拉带启动延时[A] / $?St$Bk?_#[33]
T0554 BOOL  ; 入钉NG位拉带启动延时[A]
T0555 BOOL  ; 清洁放料拉带启动延时[A]
T0556 BOOL  ; 清洁收料拉带启动延时[A]
T0557 BOOL  ; 供料振动盘启动延时[A]
T0558 BOOL  ; 0延时[A]
T0559 BOOL  ; 0延时[A]
T0560 BOOL  ; 0延时[A]
T0561 BOOL  ; $?St$Bk?_#[34] / 入钉真空阀打开延时 / $?St$Bk?_#[34]
T0562 BOOL  ; 0延时[A]
T0563 BOOL  ; $?St$Bk?_#[35] / 入钉真空阀关闭延时 / $?St$Bk?_#[35]
T0564 BOOL  ; 入钉吹气打开延时[A]
T0565 BOOL  ; 入钉吹气打开延时[A]
T0566 BOOL  ; 入钉吹气关闭延时[A]
T0567 BOOL  ; 入钉吹气关闭延时
T0568 BOOL  ; 0延时[A]
T0569 BOOL  ; 启动按钮指示灯延时[A]
T0570 BOOL  ; 停止按钮指示灯延时[A]
T0571 BOOL  ; 复位按钮指示灯延时[A]
T0572 BOOL  ; 三色灯（红）延时[A]
T0573 BOOL  ; 三色灯（绿）延时[A]
T0574 BOOL  ; 三色灯（黄）延时[A]
T0575 BOOL  ; 蜂鸣器延时[A]
T0576 BOOL  ; 入钉刹车线圈延时[A]
T0599 BOOL  ; 阻挡气缸4缩回延时
T1000 BOOL  ; 扫码阻挡气缸1原位感应延时[0000.00]
T1001 BOOL  ; 扫码阻挡气缸1到位感应延时[0000.01]
T1002 BOOL  ; 扫码阻挡气缸2原位感应延时[0000.02]
T1003 BOOL  ; 扫码阻挡气缸2到位感应延时[0000.03]
T1004 BOOL  ; 隔离气缸1原位感应延时[0000.04]
T1005 BOOL  ; 隔离气缸1到位感应延时[0000.05]
T1006 BOOL  ; 隔离气缸2原位感应延时[0000.06]
T1007 BOOL  ; 隔离气缸2到位感应延时[0000.07]
T1008 BOOL  ; 进料对射光电感应延时[0000.08]
T1009 BOOL  ; 夹爪A1夹紧位感应延时[0000.09]
T1010 BOOL  ; 夹爪A1松开位感应延时[0000.10]
T1011 BOOL  ; 夹爪A2夹紧位感应延时[0000.11]
T1012 BOOL  ; 夹爪A2松开位感应延时[0000.12]
T1013 BOOL  ; 夹爪B1夹紧位感应延时[0000.13]
T1014 BOOL  ; 夹爪B1松开位感应延时[0000.14]
T1015 BOOL  ; 夹爪B2夹紧位感应延时[0000.15]
T1016 BOOL  ; 夹爪B2松开位感应延时[0001.00]
T1017 BOOL  ; NG升降气缸1原位感应延时[0001.01]
T1018 BOOL  ; NG升降气缸1到位感应延时[0001.02]
T1019 BOOL  ; NG升降气缸2原位感应延时[0001.03]
T1020 BOOL  ; NG升降气缸2到位感应延时[0001.04]
T1021 BOOL  ; 无杆气缸1原位感应延时[0001.05]
T1022 BOOL  ; 无杆气缸1到位感应延时[0001.06]
T1023 BOOL  ; 无杆气缸2原位感应延时[0001.07]
T1024 BOOL  ; 无杆气缸2到位感应延时[0001.08]
T1025 BOOL  ; 阻挡伸出气缸1原位感应延时[0001.09]
T1026 BOOL  ; 阻挡伸出气缸1到位感应延时[0001.10]
T1027 BOOL  ; 阻挡伸出气缸2原位感应延时[0001.11]
T1028 BOOL  ; 阻挡伸出气缸2到位感应延时[0001.12]
T1029 BOOL  ; 阻挡伸出气缸3原位感应延时[0001.13]
T1030 BOOL  ; 阻挡伸出气缸3到位感应延时[0001.14]
T1031 BOOL  ; 阻挡伸出气缸4原位感应延时[0001.15]
T1032 BOOL  ; 阻挡伸出气缸4到位感应延时[0002.00]
T1033 BOOL  ; 精定位气缸A1原位感应延时[0002.01]
T1034 BOOL  ; 精定位气缸A1到位感应延时[0002.02]
T1035 BOOL  ; 精定位气缸A2原位感应延时[0002.03]
T1036 BOOL  ; 精定位气缸A2到位感应延时[0002.04]
T1037 BOOL  ; 精定位气缸B1原位感应延时[0002.05]
T1038 BOOL  ; 精定位气缸B1到位感应延时[0002.06]
T1039 BOOL  ; 精定位气缸B2原位感应延时[0002.07]
T1040 BOOL  ; 精定位气缸B2到位感应延时[0002.08]
T1041 BOOL  ; 擦拭升降气缸原位感应延时[0002.09]
T1042 BOOL  ; 擦拭升降气缸到位感应延时[0002.10]
T1043 BOOL  ; 压钉气缸原位感应延时[0002.11]
T1044 BOOL  ; 压钉气缸到位感应延时[0002.12]
T1045 BOOL  ; 料盒拨料气缸1原位感应延时[0002.13]
T1046 BOOL  ; 料盒拨料气缸1到位感应延时[0002.14]
T1047 BOOL  ; 料盒拨料气缸2原位感应延时[0002.15]
T1048 BOOL  ; 料盒拨料气缸2到位感应延时[0003.00]
T1049 BOOL  ; 推钉X轴气缸原位感应延时[0003.01]
T1050 BOOL  ; 推钉X轴气缸到位感应延时[0003.02]
T1051 BOOL  ; 推钉Y轴气缸原位感应延时[0003.03]
T1052 BOOL  ; 推钉Y轴气缸到位感应延时[0003.04]
T1053 BOOL  ; 扫码位对射光电感应延时[0003.05]
T1054 BOOL  ; 分隔电池对射光电感应延时[0003.06]
T1055 BOOL  ; 擦拭料带下限满料光电感应延时[0003.07]
T1056 BOOL  ; 擦拭料带上限放料光电感应延时
T1057 BOOL  ; 擦拭带盘无料感应延时[0003.09]
T1058 BOOL  ; 扫码NG位对射光电感应延时[0003.10]
T1059 BOOL  ; 擦拭位对射光电感应延时[0003.11]
T1060 BOOL  ; 入钉位对射光电感应延时[0003.12]
T1061 BOOL  ; 入钉NG位对射光电感应延时[0003.13]
T1062 BOOL  ; 扫码NG槽对射前光电感应延时[0003.14]
T1063 BOOL  ; 入钉NG槽对射前光电感应延时[0003.15]
T1064 BOOL  ; 扫码NG槽对射后光电感应延时[0006.00]
T1065 BOOL  ; 入钉NG槽对射后光电感应延时[0006.01]
T1066 BOOL  ; 放料允许信号感应延时[0006.02]
T1067 BOOL  ; 入钉伺服就绪 感应延时[0006.03]
T1068 BOOL  ; 入钉伺服报警 感应延时[0006.04]
T1069 BOOL  ; 启动按钮感应延时[0006.05]
T1070 BOOL  ; 停止按钮感应延时[0006.06]
T1071 BOOL  ; 复位按钮感应延时[0006.07]
T1072 BOOL  ; 急停按钮感应延时[0006.08]
T1073 BOOL  ; 手自动选择感应延时[0006.09]
T1074 BOOL  ; 设备总气压感应延时[0006.10]
T1075 BOOL  ; 夹爪1柔性报警感应延时[0006.11]
T1076 BOOL  ; 夹爪2柔性报警感应延时[0006.12]
T1077 BOOL  ; 真空信号感应延时[0006.13]
T1078 BOOL  ; 开关电源监测感应延时[0006.14]
T1079 BOOL  ; 变频器监测感应延时[0006.15]
T1080 BOOL  ; NG门磁开关感应延时[0007.00]
T1081 BOOL  ; 前门磁开关感应延时[0007.01]
T1082 BOOL  ; 后门磁开关感应延时[0007.02]
T1083 BOOL  ; 左门磁开关感应延时[0007.03]
T1084 BOOL  ; 右门磁开关感应延时[0007.04]
T1085 BOOL  ; 区域光纤对射感应延时
T1086 BOOL  ; 钉位钉子对射光纤感应延时
T1087 BOOL  ; 震盘钉嘴反射光纤感应延时
T1088 BOOL  ; 拉带入口对射光电延时
T1500 BOOL  ; 上料拉带扫码开始开始运行延时
T1509 BOOL  ; 上料机构工站复位完成延时
T1510 BOOL  ; 扫码NG抓取机构开始运行延时
T1519 BOOL  ; 扫码NG抓取工站复位完成延时
T1520 BOOL  ; 电池清洁机构开始运行条件延时
T1522 BOOL  ; 擦拭步进脉冲空闲延时
T1523 BOOL  ; 擦拭步进自动定位关闭延时
T1524 BOOL  ; 擦拭步进定位延时
T1525 BOOL  ; 擦拭步进前进延时
T1526 BOOL  ; 擦拭步进后退延时
T1527 BOOL  ; 擦拭步进擦拭位延时
T1529 BOOL  ; 电池清洁工站复位完成延时
T1530 BOOL  ; 备钉机构开始运行条件延时
T1531 BOOL  ; 入钉机构开始运行延时
T1532 BOOL  ; 入钉升降伺服脉冲空闲延时
T1534 BOOL  ; 入钉旋转步进脉冲空闲延时
T1535 BOOL  ; 入钉旋转启动延时
T1549 BOOL  ; 电池入钉工站复位完成延时
T1550 BOOL  ; 入钉NG抓取机构开始运行延时
T1569 BOOL  ; 入钉NG抓取机构工站复位完成延时
T1990 BOOL  ; 氦检仪稳定延时（公共）
W0.00 BOOL  ; 启动按钮（SW）
W0.01 BOOL  ; 停止按钮(SW)
W0.02 BOOL  ; 复位按钮（SW）
W0.04 BOOL  ; 整机复位按钮（SW）
W0.05 BOOL  ; 清料停止按钮（SW）
W0.06 BOOL  ; 整机记忆清除（SW）
W0.07 BOOL  ; 记忆清除HIM
W0.08 BOOL  ; 蜂鸣器屏蔽（SW）
W0.09 BOOL  ; 整机记忆清除HIM
W0.10 BOOL  ; 良品清零
W0.11 BOOL  ; 扫码NG清零
W0.12 BOOL  ; 入钉NG清零
W0.13 BOOL  ; 入料屏蔽
W0.15 BOOL  ; 进料拉带扫码测试[SW]
W100.00 BOOL  ; 进料水平伺服上料位置设定按钮  HMI
W100.01 BOOL  ; 进料水平伺服左爪OK配对位置设定按钮  HMI
W101.02 BOOL  ; 上料水平伺服待料位置设定按钮  HMI
W101.07 BOOL  ; 下料水平伺服放料位置设定按钮  HMI
W105.00 BOOL  ; 进料水平伺服归零辅助
W105.01 BOOL  ; 进料水平伺服前进辅助
W105.02 BOOL  ; 进料水平伺服后退辅助
W105.03 BOOL  ; 手动回进料水平伺服取料位辅助
W105.04 BOOL  ; 手动回进料水平伺服左爪OK配对位辅助
W105.12 BOOL  ; 手动回进料水平伺服放料位辅助
W106.11 BOOL  ; 上料水平伺服归零辅助
W106.12 BOOL  ; 上料水平伺服前进辅助
W106.13 BOOL  ; 上料水平伺服后退辅助
W106.14 BOOL  ; 手动回上料水平伺服待料位辅助
W107.05 BOOL  ; 手动回下料水平伺服#2腔体位辅助
W107.06 BOOL  ; 手动回下料水平伺服放料位辅助
W10.00 BOOL  ; 进料水平伺服归零   HMI
W10.01 BOOL  ; 进料水平伺服前进   HMI
W10.03 BOOL  ; 手动回进料水平伺服取料位置  HMI
W110.00 BOOL  ; 自动回进料水平伺服上料位辅助
W110.02 BOOL  ; 自动回进料水平伺服右配对位辅助
W115.00 BOOL  ; 进料水平伺服在取料位
W115.01 BOOL  ; 进料水平伺服在左爪OK配对位
W115.02 BOOL  ; 进料水平伺服在右爪OK配对位
W115.03 BOOL  ; 进料水平伺服在左爪缓存位
W115.04 BOOL  ; 进料水平伺服在右爪缓存位
W115.05 BOOL  ; 进料水平伺服在NG位
W115.09 BOOL  ; 进料水平伺服在放料位
W115.14 BOOL  ; 进料升降伺服在待料位
W116.02 BOOL  ; 上料料水平伺服在待料位
W116.07 BOOL  ; 下料水平伺服在放料位
W117.04 BOOL  ; 进料水平伺服在原点位置
W117.05 BOOL  ; 进料升降伺服在原点位置
W118.00 BOOL  ; 备用
W11.11 BOOL  ; 上料水平伺服归零   HMI
W11.12 BOOL  ; 上料水平伺服前进   HMI
W11.13 BOOL  ; 上料水平伺服后退   HMI
W11.14 BOOL  ; 手动回上料水平伺服待料位置  HMI
W1.00 BOOL  ; 手动模式
W1.01 BOOL  ; 自动模式
W1.10 BOOL  ; 上料位有料模拟
W231.00 BOOL  ; 自动回进料水平伺服上料位
W231.15 BOOL  ; 上料机构手自动运行
W233.00 BOOL  ; 自动回下料水平伺服放料位辅助
W233.15 BOOL  ; 下料机构手自动运行
W320.06 BOOL  ; 擦拭步进前进 HMI
W320.07 BOOL  ; 擦拭步进后退 HMI
W320.08 BOOL  ; 擦拭步进启动 HIM
W321.06 BOOL  ; 擦拭步进前进
W321.07 BOOL  ; 擦拭步进后退
W321.08 BOOL  ; 擦拭步进启动
W325.00 BOOL  ; 擦拭步进自动运行
W325.03 BOOL  ; 擦拭步进在零位
W325.04 BOOL  ; 擦拭步进运行脉冲完成
W326.00 BOOL  ; 擦拭步进在擦拭位
W326.03 BOOL  ; 擦拭步进启动
W330.00 BOOL  ; 入钉升降伺服归零 HMI
W330.01 BOOL  ; 入钉升降伺服下降 HMI
W330.02 BOOL  ; 入钉升降伺服上升 HMI
W330.03 BOOL  ; 入钉升降伺服至准入钉位 HIM
W330.04 BOOL  ; 入钉升降伺服至安全高度位 HIM
W330.05 BOOL  ; 入钉升降伺服至入钉位 HIM
W330.06 BOOL  ; 入钉旋转步进上升 HMI
W330.07 BOOL  ; 入钉旋转步进下降 HMI
W330.08 BOOL  ; 入钉旋转步进启动 HIM
W330.09 BOOL  ; 入钉旋转入钉深度按钮  HMI
W330.10 BOOL  ; 设定入钉升降伺服准入钉位 HIM
W330.11 BOOL  ; 设定入钉升降伺服安全高度位 HIM
W330.12 BOOL  ; 设定入钉升降伺服入钉位 HIM
W331.00 BOOL  ; 入钉升降伺服归零
W331.01 BOOL  ; 入钉升降伺服下降
W331.02 BOOL  ; 入钉升降伺服上升
W331.03 BOOL  ; 入钉升降伺服准入钉位
W331.04 BOOL  ; 入钉升降伺服安全高度位
W331.05 BOOL  ; 入钉升降伺服入钉位
W331.06 BOOL  ; 入钉旋转步进上升
W331.07 BOOL  ; 入钉旋转步进下降
W331.08 BOOL  ; 入钉旋转步进启动
W335.00 BOOL  ; 入钉升降伺服在准入钉位
W335.01 BOOL  ; 入钉升降伺服在安全高度位
W335.02 BOOL  ; 入钉升降伺服在入钉位
W335.03 BOOL  ; 入钉旋转步进在零位
W335.04 BOOL  ; 入钉旋转步进运行脉冲完成
W336.00 BOOL  ; 入钉升降至准入钉位
W336.01 BOOL  ; 入钉升降至安全高度位
W336.02 BOOL  ; 入钉升降至入钉位
W336.03 BOOL  ; 入钉旋转启动
W338.00 BOOL  ; 入钉旋转步进自动运行
W400.00 BOOL  ; [W400.00]扫码阻挡气缸1原位异常,请检查[0000.00]
W400.01 BOOL  ; [W400.01]扫码阻挡气缸1到位异常,请检查[0000.01]
W400.02 BOOL  ; [W400.02]扫码阻挡气缸2原位异常,请检查[0000.02]
W400.03 BOOL  ; [W400.03]扫码阻挡气缸2到位异常,请检查[0000.03]
W400.04 BOOL  ; [W400.04]隔离气缸1原位异常,请检查[0000.04]
W400.05 BOOL  ; [W400.05]隔离气缸1到位异常,请检查[0000.05]
W400.06 BOOL  ; [W400.06]隔离气缸2原位异常,请检查[0000.06]
W400.07 BOOL  ; [W400.07]隔离气缸2到位异常,请检查[0000.07]
W400.08 BOOL  ; [W400.08]进料对射光电满料异常,请检查[0000.08]
W400.09 BOOL  ; [W400.09]夹爪A1夹紧位异常,请检查[0000.09]
W400.10 BOOL  ; [W400.10]夹爪A1松开位异常,请检查[0000.10]
W400.11 BOOL  ; [W400.11]夹爪A2夹紧位异常,请检查[0000.11]
W400.12 BOOL  ; [W400.12]夹爪A2松开位异常,请检查[0000.12]
W400.13 BOOL  ; [W400.13]夹爪B1夹紧位异常,请检查[0000.13]
W400.14 BOOL  ; [W400.14]夹爪B1松开位异常,请检查[0000.14]
W400.15 BOOL  ; [W400.15]夹爪B2夹紧位异常,请检查[0000.15]
W401.00 BOOL  ; [W401.00]夹爪B2松开位异常,请检查[0001.00]
W401.01 BOOL  ; [W401.01]NG升降气缸1原位异常,请检查[0001.01]
W401.02 BOOL  ; [W401.02]NG升降气缸1到位异常,请检查[0001.02]
W401.03 BOOL  ; [W401.03]NG升降气缸2原位异常,请检查[0001.03]
W401.04 BOOL  ; [W401.04]NG升降气缸2到位异常,请检查[0001.04]
W401.05 BOOL  ; [W401.05]NG无杆气缸1原位异常,请检查[0001.05]
W401.06 BOOL  ; [W401.06]NG无杆气缸1到位异常,请检查[0001.06]
W401.07 BOOL  ; [W401.07]NG无杆气缸2原位异常,请检查[0001.07]
W401.08 BOOL  ; [W401.08]NG无杆气缸2到位异常,请检查[0001.08]
W401.09 BOOL  ; [W401.09]阻挡伸出气缸1原位异常,请检查[0001.09]
W401.10 BOOL  ; [W401.10]阻挡伸出气缸1到位异常,请检查[0001.10]
W401.11 BOOL  ; [W401.11]阻挡伸出气缸2原位异常,请检查[0001.11]
W401.12 BOOL  ; [W401.12]阻挡伸出气缸2到位异常,请检查[0001.12]
W401.13 BOOL  ; [W401.13]阻挡伸出气缸3原位异常,请检查[0001.13]
W401.14 BOOL  ; [W401.14]阻挡伸出气缸3到位异常,请检查[0001.14]
W401.15 BOOL  ; [W401.15]阻挡伸出气缸4原位异常,请检查[0001.15]
W402.00 BOOL  ; [W402.00]阻挡伸出气缸4到位异常,请检查[0002.00]
W402.01 BOOL  ; [W402.01]精定位气缸A1原位异常,请检查[0002.01]
W402.02 BOOL  ; [W402.02]精定位气缸A1到位异常,请检查[0002.02]
W402.03 BOOL  ; [W402.03]精定位气缸A2原位异常,请检查[0002.03]
W402.04 BOOL  ; [W402.04]精定位气缸A2到位异常,请检查[0002.04]
W402.05 BOOL  ; [W402.05]精定位气缸B1原位异常,请检查[0002.05]
W402.06 BOOL  ; [W402.06]精定位气缸B1到位异常,请检查[0002.06]
W402.07 BOOL  ; [W402.07]精定位气缸B2原位异常,请检查[0002.07]
W402.08 BOOL  ; [W402.08]精定位气缸B2到位异常,请检查[0002.08]
W402.09 BOOL  ; [W402.09]擦拭升降气缸原位异常,请检查[0002.09]
W402.10 BOOL  ; [W402.10]擦拭升降气缸到位异常,请检查[0002.10]
W402.11 BOOL  ; [W402.11]压钉气缸原位异常,请检查[0002.11]
W402.12 BOOL  ; [W402.12]压钉气缸到位异常,请检查[0002.12]
W402.13 BOOL  ; [W402.13]料盒拨料气缸1原位异常,请检查[0002.13]
W402.14 BOOL  ; [W402.14]料盒拨料气缸1到位异常,请检查[0002.14]
W402.15 BOOL  ; [W402.15]料盒拨料气缸2原位异常,请检查[0002.15]
W403.00 BOOL  ; [W403.00]料盒拨料气缸2到位异常,请检查[0003.00]
W403.01 BOOL  ; [W403.01]推钉X轴气缸原位异常,请检查[0003.01]
W403.02 BOOL  ; [W403.02]推钉X轴气缸到位异常,请检查[0003.02]
W403.03 BOOL  ; [W403.03]推钉Y轴气缸原位异常,请检查[0003.03]
W403.04 BOOL  ; [W403.04]推钉Y轴气缸到位异常,请检查[0003.04]
W403.05 BOOL  ; [W403.05]扫码位对射光电感应异常,请检查[0003.05]
W403.06 BOOL  ; [W403.06]分隔电池对射光电感应异常,请检查[0003.06]
W403.07 BOOL  ; [W403.07]清洁带光电1感应异常,请检查[0003.07]
W403.08 BOOL  ; 请检查[0003.08] / $?St$Bk?_#[36]
W403.09 BOOL  ; 请检查[0003.09] / $?St$Bk?_#[37]
W403.10 BOOL  ; [W403.10]扫码NG位对射光电感应异常,请检查[0003.10]
W403.11 BOOL  ; [W403.11]擦拭位对射光电感应异常,请检查[0003.11]
W403.12 BOOL  ; [W403.12]胶钉未射入，钉位对射光电感应异常,请检查[0007.06]
W403.13 BOOL  ; [W403.13]入钉NG位对射光电异常,请检查[0003.13]
W403.14 BOOL  ; [W403.14]扫码NG槽对射前光电异常,请检查[0003.14]
W403.15 BOOL  ; [W403.15]入钉NG槽对射前光电异常,请检查[0003.15]
W404.00 BOOL  ; [W404.00]扫码NG槽对射光电满料[0006.00]异常,请检查[0006.00]
W404.01 BOOL  ; [W404.01]入钉NG槽对射后光电异常,满料请检查[0006.01]
W404.02 BOOL  ; 请检查[0006.02] / $?St$Bk?_#[38]
W404.03 BOOL  ; [W404.03]入钉伺服就绪异常,请检查[0006.03]
W404.04 BOOL  ; [W404.04]入钉伺服报警异常,请检查[0006.04]
W404.05 BOOL  ; [W404.05]启动按钮异常,请检查[0006.05]
W404.06 BOOL  ; [W404.06]停止按钮异常,请检查[0006.06]
W404.07 BOOL  ; [W404.07]复位按钮异常,请检查[0006.07]
W404.08 BOOL  ; [W404.08]急停按钮异常,请检查[0006.08]
W404.09 BOOL  ; [W404.09]手自动选择异常,请检查[0006.09]
W404.10 BOOL  ; [W404.10]设备总气压异常,请检查[0006.10]
W404.11 BOOL  ; [W404.11]夹爪1柔性报警异常,请检查[0006.11]
W404.12 BOOL  ; [W404.12]夹爪2柔性报警异常,请检查[0006.12]
W404.13 BOOL  ; [W404.13]真空信号异常,请检查[0006.13]
W404.14 BOOL  ; [W404.14]开关电源监测异常,请检查[0006.14]
W404.15 BOOL  ; [W404.15]变频器监测异常,请检查[0006.15]
W405.00 BOOL  ; [W405.00]NG门磁开关异常,请检查[0007.00]
W405.01 BOOL  ; [W405.01]前门磁开关异常,请检查[0007.01]
W405.02 BOOL  ; [W405.02]后门磁开关异常,请检查[0007.02]
W405.03 BOOL  ; [W405.03]左门磁开关异常,请检查[0007.03]
W405.04 BOOL  ; [W405.04]右门磁开关异常,请检查[0007.04]
W405.05 BOOL  ; [W405.05]入钉前入钉胶管有钉异常,请检查[0007.06]
W405.06 BOOL  ; [W405.06]吹钉入胶管钉位感应异常,请检查[0007.06]
W405.07 BOOL  ; [W405.07]扫码NG槽对射光电满料,请检查[0006.00]
W405.08 BOOL  ; [W405.08]入钉NG槽对射光电满料,请检查[0006.01]
W405.09 BOOL  ; ！！
W405.10 BOOL  ; [W405.10]入钉前胶管有钉感应！禁止入钉！
W405.11 BOOL  ; [W405.11]入钉前胶管有钉记忆！清除胶嘴胶钉或记忆！
W405.12 BOOL  ; [W405.12]吹气入钉钉位无胶钉感应！请检查吹气管道！
W405.13 BOOL  ; [W405.13]吹气入钉管嘴内有钉记忆！
W405.14 BOOL  ; [W405.14]管嘴内有钉记忆，钉位无胶钉感应。异常！！
W405.15 BOOL  ; [W405.15]管嘴内无胶钉记忆，钉位有胶钉感应。异常！！
W40.00 BOOL  ; 扫码允许信号
W411.02 BOOL  ; 扫码枪通讯异常[alm]
W41.02 BOOL  ; 进料水平伺服归零
W41.03 BOOL  ; 进料水平伺服回取料位
W4.04 BOOL  ; 扫码枪1 TCP打开2(SW)(HMI)
W4.05 BOOL  ; TCP2关闭
W4.06 BOOL  ; TCP2发送
W51.10 BOOL  ; 腔体上料伺服复位(M)
W5.00 BOOL  ; TCP打开错误
W5.01 BOOL  ; TCP关闭错误
W5.02 BOOL  ; TCP发送错误
W5.03 BOOL  ; TCP接收错误
W65.00 BOOL  ; 上料拉带扫码
W65.01 BOOL  ; 上料拉带扫码开始
W65.02 BOOL  ; 上料拉带扫码失败
W65.03 BOOL  ; 上料拉带扫码成功
W65.05 BOOL  ; 上料拉带重新扫码触发
W9.00 BOOL  ; 故障
W9.01 BOOL  ; 清料标志

## Program Main (cyclic task 0)

### Section Main

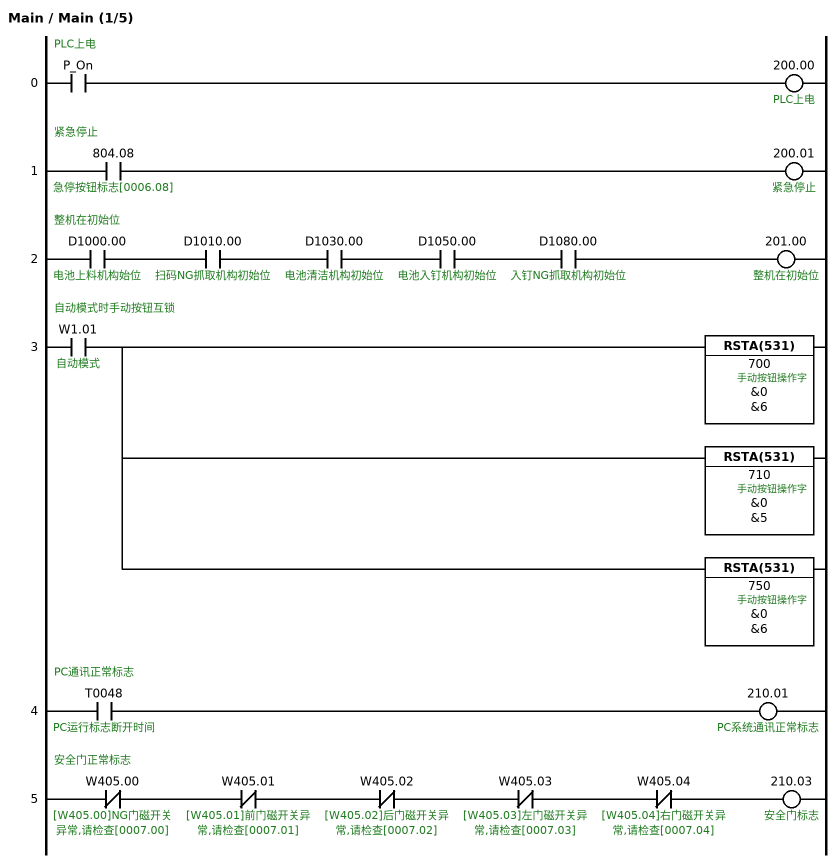
; rung 0: PLC上电
LD P_On
OUT 200.00  ; PLC上电
; rung 1: 紧急停止
LD 804.08  ; 急停按钮标志[0006.08]
OUT 200.01  ; 紧急停止
; rung 2: 整机在初始位
LD D1000.00  ; 电池上料机构始位
AND D1010.00  ; 扫码NG抓取机构初始位
AND D1030.00  ; 电池清洁机构初始位
AND D1050.00  ; 电池入钉机构初始位
AND D1080.00  ; 入钉NG抓取机构初始位
OUT 201.00  ; 整机在初始位
; rung 3: 自动模式时手动按钮互锁
LD W1.01  ; 自动模式
RSTA(531) 700 &0 &6  ; 手动按钮操作字
RSTA(531) 710 &0 &5  ; 手动按钮操作字
RSTA(531) 750 &0 &6  ; 手动按钮操作字
; rung 4: PC通讯正常标志
LD T0048  ; PC运行标志断开时间
OUT 210.01  ; PC系统通讯正常标志
; rung 5: 安全门正常标志
LDNOT W405.00  ; [W405.00]NG门磁开关异常,请检查[0007.00]
ANDNOT W405.01  ; [W405.01]前门磁开关异常,请检查[0007.01]
ANDNOT W405.02  ; [W405.02]后门磁开关异常,请检查[0007.02]
ANDNOT W405.03  ; [W405.03]左门磁开关异常,请检查[0007.03]
ANDNOT W405.04  ; [W405.04]右门磁开关异常,请检查[0007.04]
OUT 210.03  ; 安全门标志

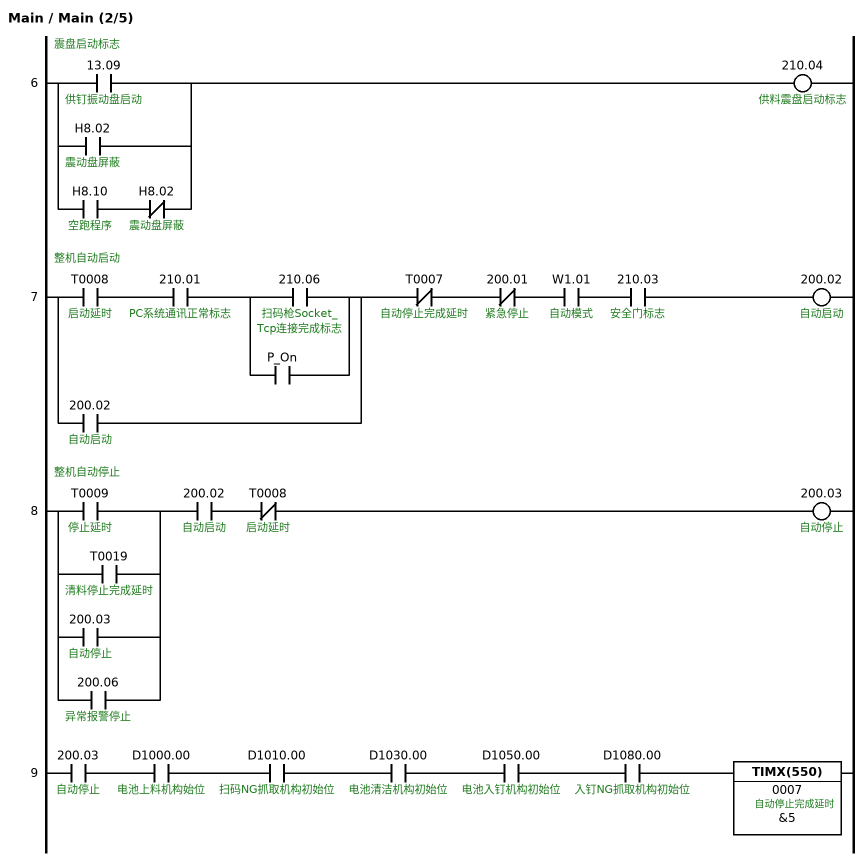
; rung 6: 震盘启动标志
LD 13.09  ; 供钉振动盘启动
OR H8.02  ; 震动盘屏蔽
LD H8.10  ; 空跑程序
ANDNOT H8.02  ; 震动盘屏蔽
ORLD
OUT 210.04  ; 供料震盘启动标志
; rung 7: 整机自动启动
LD T0008  ; 启动延时
AND 210.01  ; PC系统通讯正常标志
LD 210.06  ; 扫码枪Socket_Tcp连接完成标志
OR P_On
ANDLD
OR 200.02  ; 自动启动
ANDNOT T0007  ; 自动停止完成延时
ANDNOT 200.01  ; 紧急停止
AND W1.01  ; 自动模式
AND 210.03  ; 安全门标志
OUT 200.02  ; 自动启动
; rung 8: 整机自动停止
LD T0009  ; 停止延时
OR T0019  ; 清料停止完成延时
OR 200.03  ; 自动停止
OR 200.06  ; 异常报警停止
AND 200.02  ; 自动启动
ANDNOT T0008  ; 启动延时
OUT 200.03  ; 自动停止
; rung 9
LD 200.03  ; 自动停止
AND D1000.00  ; 电池上料机构始位
AND D1010.00  ; 扫码NG抓取机构初始位
AND D1030.00  ; 电池清洁机构初始位
AND D1050.00  ; 电池入钉机构初始位
AND D1080.00  ; 入钉NG抓取机构初始位
TIMX(550) 0007 &5  ; 自动停止完成延时

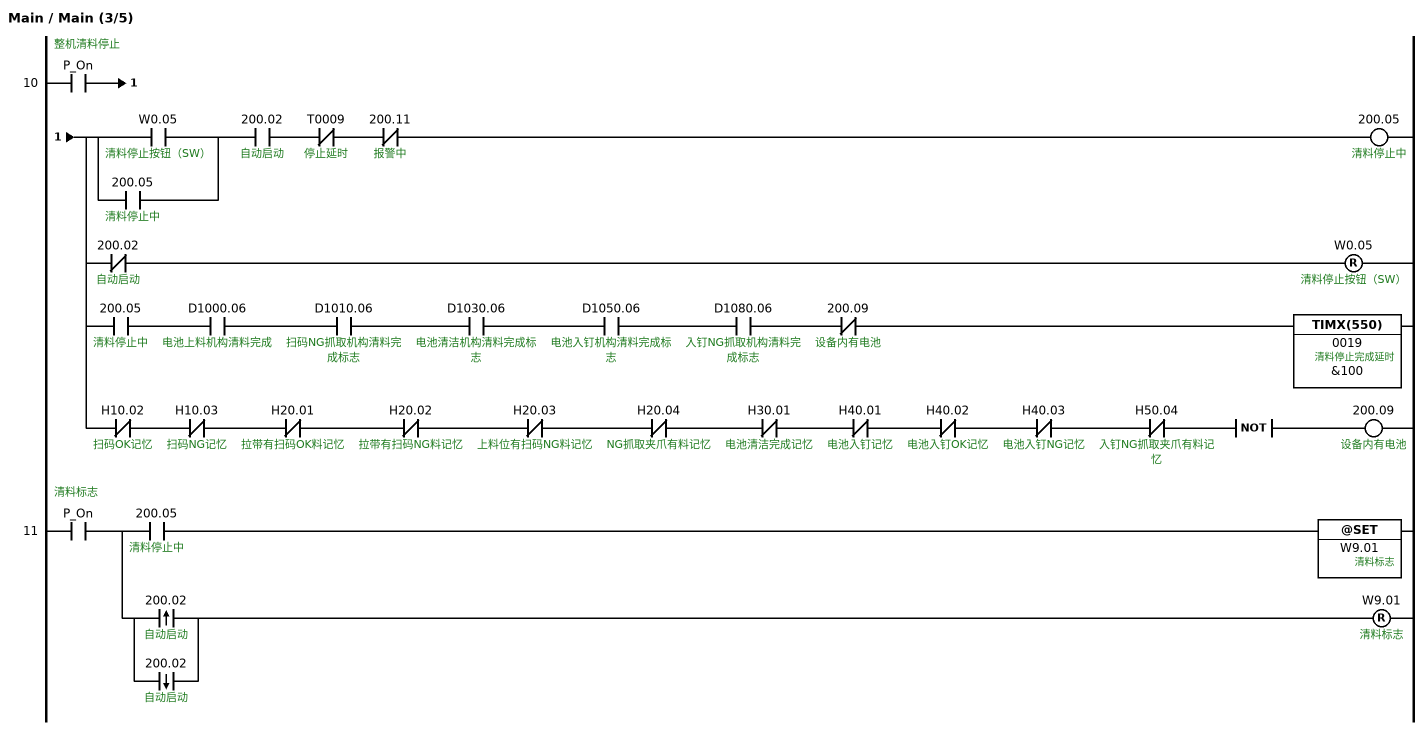
; rung 10: 整机清料停止
LD P_On
OUT TR0
LD W0.05  ; 清料停止按钮（SW）
OR 200.05  ; 清料停止中
ANDLD
AND 200.02  ; 自动启动
ANDNOT T0009  ; 停止延时
ANDNOT 200.11  ; 报警中
OUT 200.05  ; 清料停止中
LD TR0
ANDNOT 200.02  ; 自动启动
RSET W0.05  ; 清料停止按钮（SW）
LD TR0
AND 200.05  ; 清料停止中
AND D1000.06  ; 电池上料机构清料完成
AND D1010.06  ; 扫码NG抓取机构清料完成标志
AND D1030.06  ; 电池清洁机构清料完成标志
AND D1050.06  ; 电池入钉机构清料完成标志
AND D1080.06  ; 入钉NG抓取机构清料完成标志
ANDNOT 200.09  ; 设备内有电池
TIMX(550) 0019 &100  ; 清料停止完成延时
LD TR0
ANDNOT H10.02  ; 扫码OK记忆
ANDNOT H10.03  ; 扫码NG记忆
ANDNOT H20.01  ; 拉带有扫码OK料记忆
ANDNOT H20.02  ; 拉带有扫码NG料记忆
ANDNOT H20.03  ; 上料位有扫码NG料记忆
ANDNOT H20.04  ; NG抓取夹爪有料记忆
ANDNOT H30.01  ; 电池清洁完成记忆
ANDNOT H40.01  ; 电池入钉记忆
ANDNOT H40.02  ; 电池入钉OK记忆
ANDNOT H40.03  ; 电池入钉NG记忆
ANDNOT H50.04  ; 入钉NG抓取夹爪有料记忆
NOT(520)
OUT 200.09  ; 设备内有电池
; rung 11: 清料标志
LD P_On
OUT TR0
AND 200.05  ; 清料停止中
@SET W9.01  ; 清料标志
LD TR0
@LD 200.02  ; 自动启动
%OR 200.02  ; 自动启动
ANDLD
RSET W9.01  ; 清料标志

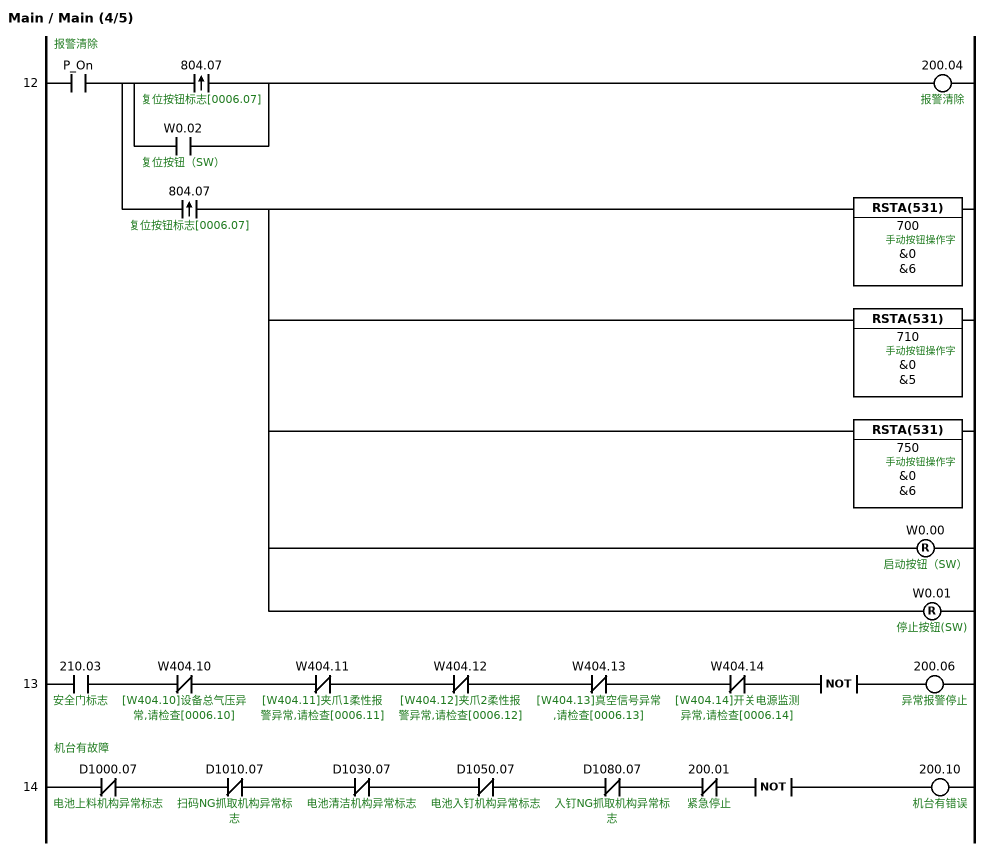
; rung 12: 报警清除
LD P_On
OUT TR0
@LD 804.07  ; 复位按钮标志[0006.07]
OR W0.02  ; 复位按钮（SW）
ANDLD
OUT 200.04  ; 报警清除
LD TR0
@AND 804.07  ; 复位按钮标志[0006.07]
RSTA(531) 700 &0 &6  ; 手动按钮操作字
RSTA(531) 710 &0 &5  ; 手动按钮操作字
RSTA(531) 750 &0 &6  ; 手动按钮操作字
RSET W0.00  ; 启动按钮（SW）
RSET W0.01  ; 停止按钮(SW)
; rung 13
LD 210.03  ; 安全门标志
ANDNOT W404.10  ; [W404.10]设备总气压异常,请检查[0006.10]
ANDNOT W404.11  ; [W404.11]夹爪1柔性报警异常,请检查[0006.11]
ANDNOT W404.12  ; [W404.12]夹爪2柔性报警异常,请检查[0006.12]
ANDNOT W404.13  ; [W404.13]真空信号异常,请检查[0006.13]
ANDNOT W404.14  ; [W404.14]开关电源监测异常,请检查[0006.14]
NOT(520)
OUT 200.06  ; 异常报警停止
; rung 14: 机台有故障
LDNOT D1000.07  ; 电池上料机构异常标志
ANDNOT D1010.07  ; 扫码NG抓取机构异常标志
ANDNOT D1030.07  ; 电池清洁机构异常标志
ANDNOT D1050.07  ; 电池入钉机构异常标志
ANDNOT D1080.07  ; 入钉NG抓取机构异常标志
ANDNOT 200.01  ; 紧急停止
NOT(520)
OUT 200.10  ; 机台有错误

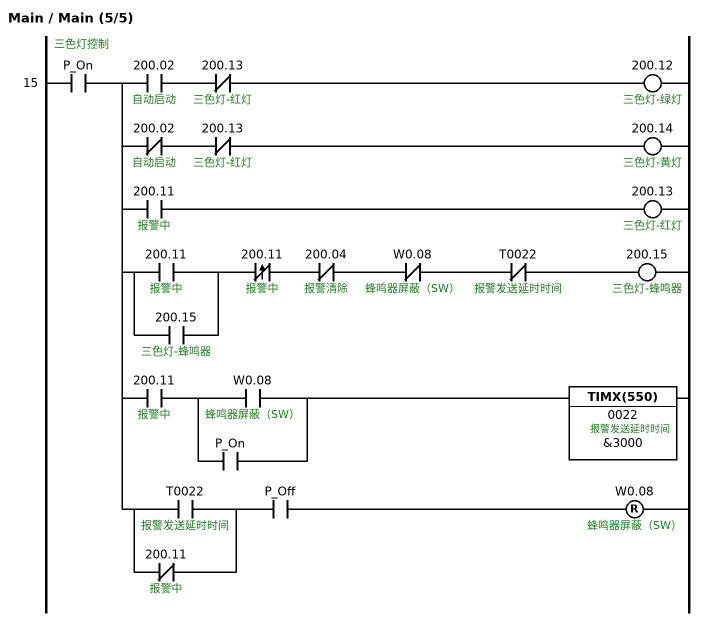
; rung 15: 三色灯控制
LD P_On
OUT TR0
AND 200.02  ; 自动启动
ANDNOT 200.13  ; 三色灯-红灯
OUT 200.12  ; 三色灯-绿灯
LD TR0
ANDNOT 200.02  ; 自动启动
ANDNOT 200.13  ; 三色灯-红灯
OUT 200.14  ; 三色灯-黄灯
LD TR0
AND 200.11  ; 报警中
OUT 200.13  ; 三色灯-红灯
LD TR0
LD 200.11  ; 报警中
OR 200.15  ; 三色灯-蜂鸣器
ANDLD
@ANDNOT 200.11  ; 报警中
ANDNOT 200.04  ; 报警清除
ANDNOT W0.08  ; 蜂鸣器屏蔽（SW）
ANDNOT T0022  ; 报警发送延时时间
OUT 200.15  ; 三色灯-蜂鸣器
LD TR0
AND 200.11  ; 报警中
LD W0.08  ; 蜂鸣器屏蔽（SW）
OR P_On
ANDLD
TIMX(550) 0022 &3000  ; 报警发送延时时间
LD TR0
LD T0022  ; 报警发送延时时间
ORNOT 200.11  ; 报警中
ANDLD
AND P_Off
RSET W0.08  ; 蜂鸣器屏蔽（SW）

### Section 入料扫码通讯

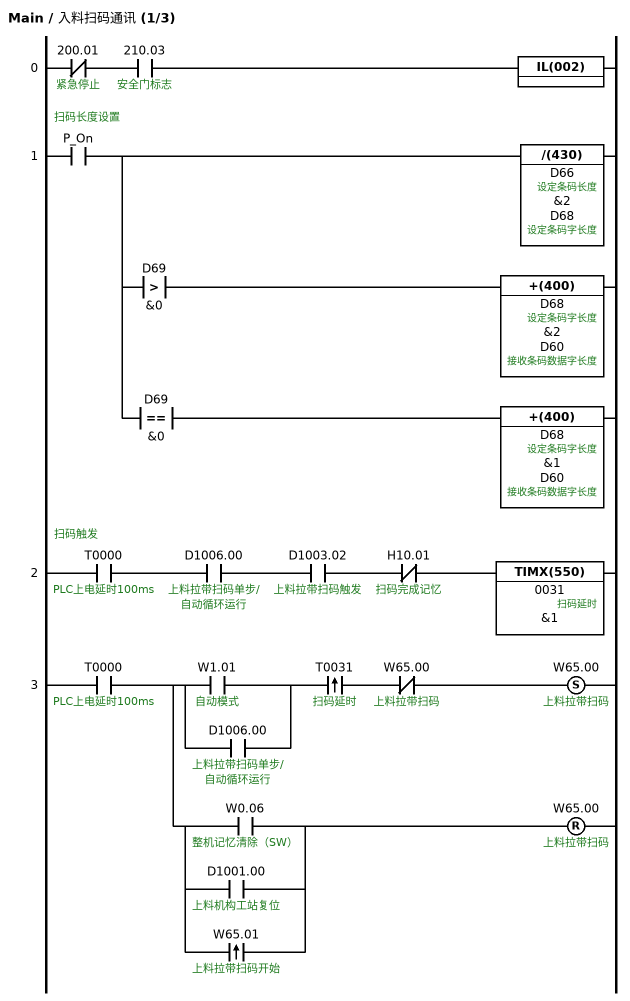
; rung 0
LDNOT 200.01  ; 紧急停止
AND 210.03  ; 安全门标志
IL(002)
; rung 1: 扫码长度设置
LD P_On
OUT TR0
/(430) D66 &2 D68  ; 设定条码长度, 设定条码字长度
AND>(320) D69 &0
+(400) D68 &2 D60  ; 设定条码字长度, 接收条码数据字长度
LD TR0
AND=(300) D69 &0
+(400) D68 &1 D60  ; 设定条码字长度, 接收条码数据字长度
; rung 2: 扫码触发
LD T0000  ; PLC上电延时100ms
AND D1006.00  ; 上料拉带扫码单步/自动循环运行
AND D1003.02  ; 上料拉带扫码触发
ANDNOT H10.01  ; 扫码完成记忆
TIMX(550) 0031 &1  ; 扫码延时
; rung 3
LD T0000  ; PLC上电延时100ms
OUT TR0
LD W1.01  ; 自动模式
OR D1006.00  ; 上料拉带扫码单步/自动循环运行
ANDLD
@AND T0031  ; 扫码延时
ANDNOT W65.00  ; 上料拉带扫码
SET W65.00  ; 上料拉带扫码
LD TR0
LD W0.06  ; 整机记忆清除（SW）
OR D1001.00  ; 上料机构工站复位
@OR W65.01  ; 上料拉带扫码开始
ANDLD
RSET W65.00  ; 上料拉带扫码

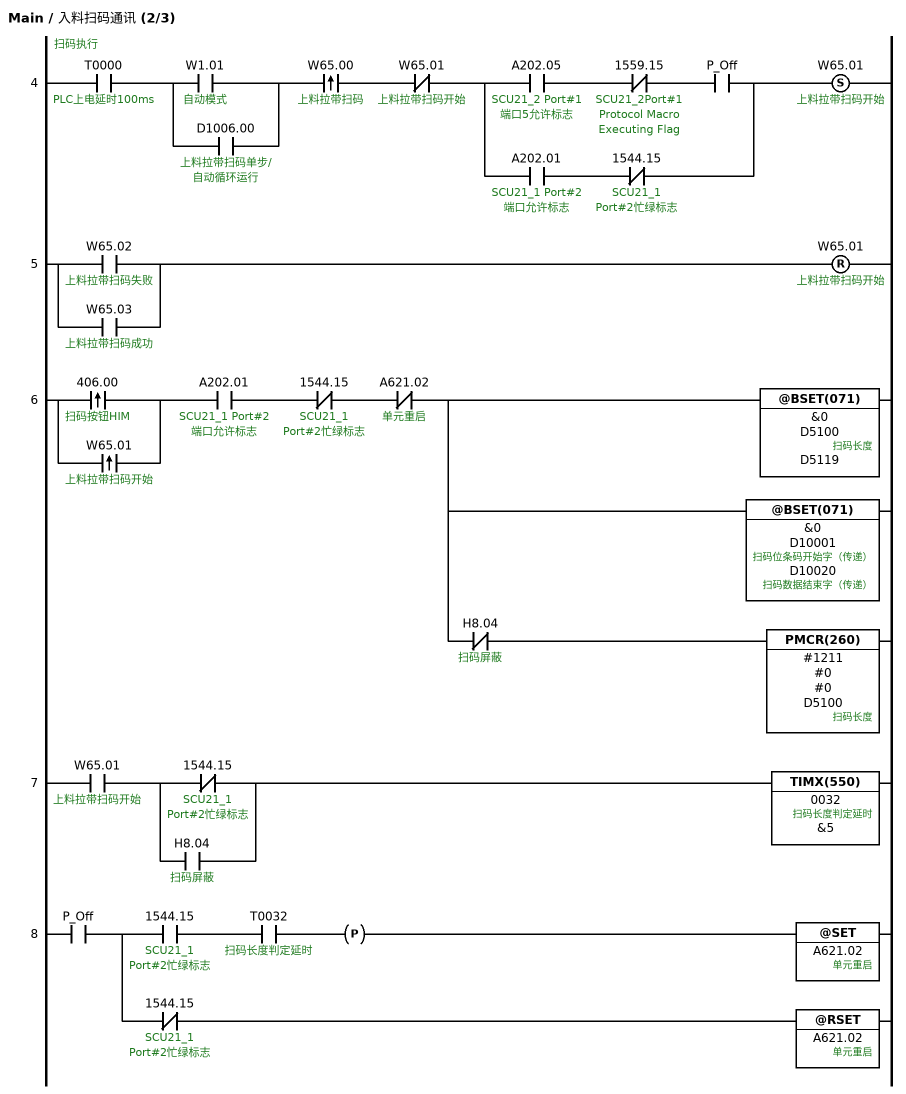
; rung 4: 扫码执行
LD T0000  ; PLC上电延时100ms
LD W1.01  ; 自动模式
OR D1006.00  ; 上料拉带扫码单步/自动循环运行
ANDLD
@AND W65.00  ; 上料拉带扫码
ANDNOT W65.01  ; 上料拉带扫码开始
LD A202.05  ; SCU21_2 Port#1 端口5允许标志
ANDNOT 1559.15  ; SCU21_2Port#1 Protocol Macro Executing Flag
AND P_Off
LD A202.01  ; SCU21_1 Port#2 端口允许标志
ANDNOT 1544.15  ; SCU21_1 Port#2忙绿标志
ORLD
ANDLD
SET W65.01  ; 上料拉带扫码开始
; rung 5
LD W65.02  ; 上料拉带扫码失败
OR W65.03  ; 上料拉带扫码成功
RSET W65.01  ; 上料拉带扫码开始
; rung 6
@LD 406.00  ; 扫码按钮HIM
@OR W65.01  ; 上料拉带扫码开始
AND A202.01  ; SCU21_1 Port#2 端口允许标志
ANDNOT 1544.15  ; SCU21_1 Port#2忙绿标志
ANDNOT A621.02  ; 单元重启
@BSET(071) &0 D5100 D5119  ; 扫码长度
@BSET(071) &0 D10001 D10020  ; 扫码位条码开始字（传递）, 扫码数据结束字（传递）
ANDNOT H8.04  ; 扫码屏蔽
PMCR(260) #1211 #0 #0 D5100  ; 扫码长度
; rung 7
LD W65.01  ; 上料拉带扫码开始
LDNOT 1544.15  ; SCU21_1 Port#2忙绿标志
OR H8.04  ; 扫码屏蔽
ANDLD
TIMX(550) 0032 &5  ; 扫码长度判定延时
; rung 8
LD P_Off
OUT TR0
AND 1544.15  ; SCU21_1 Port#2忙绿标志
AND T0032  ; 扫码长度判定延时
UP(521)
@SET A621.02  ; 单元重启
LD TR0
ANDNOT 1544.15  ; SCU21_1 Port#2忙绿标志
@RSET A621.02  ; 单元重启

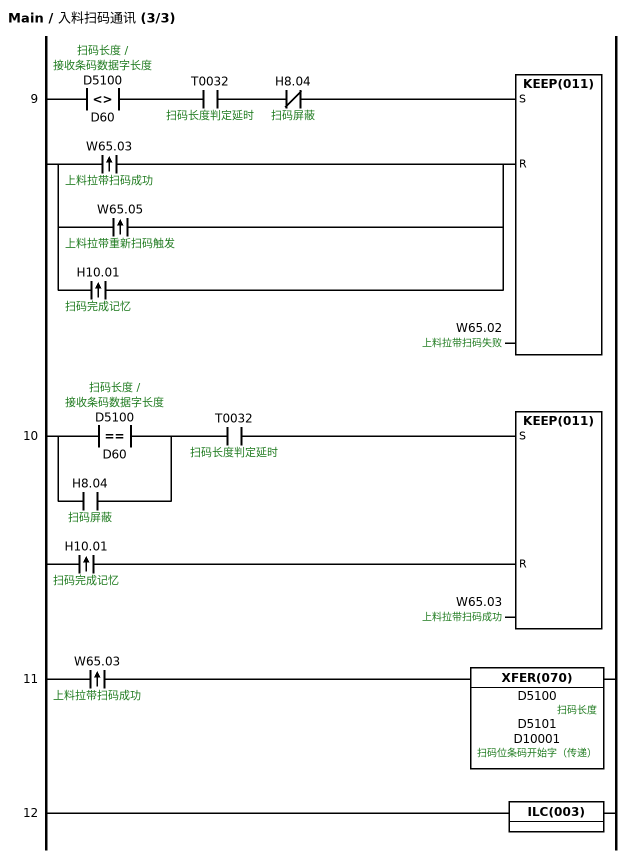
; rung 9
LD<>(305) D5100 D60  ; 扫码长度, 接收条码数据字长度
AND T0032  ; 扫码长度判定延时
ANDNOT H8.04  ; 扫码屏蔽
@LD W65.03  ; 上料拉带扫码成功
@OR W65.05  ; 上料拉带重新扫码触发
@OR H10.01  ; 扫码完成记忆
KEEP(011) W65.02  ; 上料拉带扫码失败
; rung 10
LD=(300) D5100 D60  ; 扫码长度, 接收条码数据字长度
OR H8.04  ; 扫码屏蔽
AND T0032  ; 扫码长度判定延时
@LD H10.01  ; 扫码完成记忆
KEEP(011) W65.03  ; 上料拉带扫码成功
; rung 11
@LD W65.03  ; 上料拉带扫码成功
XFER(070) D5100 D5101 D10001  ; 扫码长度, 扫码位条码开始字（传递）
; rung 12
ILC(003)

### Section 复位

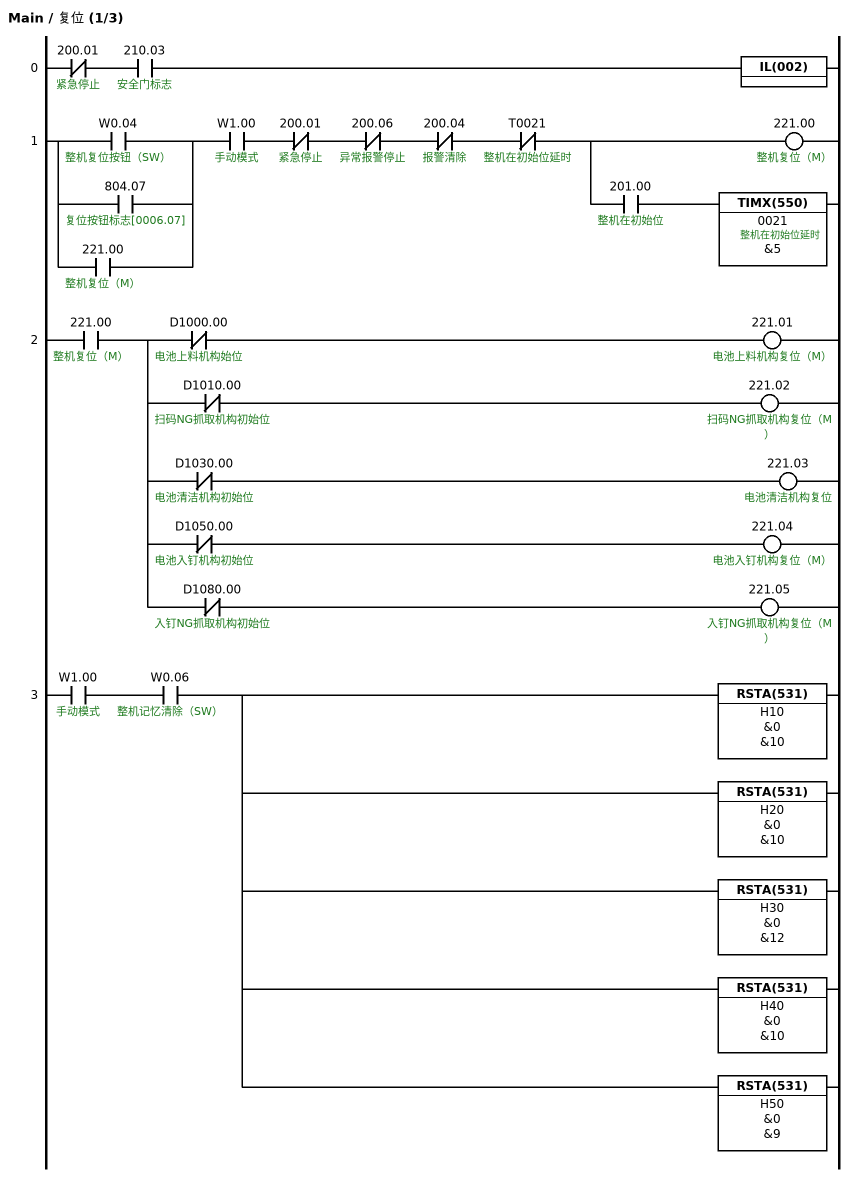
; rung 0
LDNOT 200.01  ; 紧急停止
AND 210.03  ; 安全门标志
IL(002)
; rung 1
LD W0.04  ; 整机复位按钮（SW）
OR 804.07  ; 复位按钮标志[0006.07]
OR 221.00  ; 整机复位（M）
AND W1.00  ; 手动模式
ANDNOT 200.01  ; 紧急停止
ANDNOT 200.06  ; 异常报警停止
ANDNOT 200.04  ; 报警清除
ANDNOT T0021  ; 整机在初始位延时
OUT 221.00  ; 整机复位（M）
AND 201.00  ; 整机在初始位
TIMX(550) 0021 &5  ; 整机在初始位延时
; rung 2
LD 221.00  ; 整机复位（M）
OUT TR0
ANDNOT D1000.00  ; 电池上料机构始位
OUT 221.01  ; 电池上料机构复位（M）
LD TR0
ANDNOT D1010.00  ; 扫码NG抓取机构初始位
OUT 221.02  ; 扫码NG抓取机构复位（M）
LD TR0
ANDNOT D1030.00  ; 电池清洁机构初始位
OUT 221.03  ; 电池清洁机构复位
LD TR0
ANDNOT D1050.00  ; 电池入钉机构初始位
OUT 221.04  ; 电池入钉机构复位（M）
LD TR0
ANDNOT D1080.00  ; 入钉NG抓取机构初始位
OUT 221.05  ; 入钉NG抓取机构复位（M）
; rung 3
LD W1.00  ; 手动模式
AND W0.06  ; 整机记忆清除（SW）
RSTA(531) H10 &0 &10
RSTA(531) H20 &0 &10
RSTA(531) H30 &0 &12
RSTA(531) H40 &0 &10
RSTA(531) H50 &0 &9

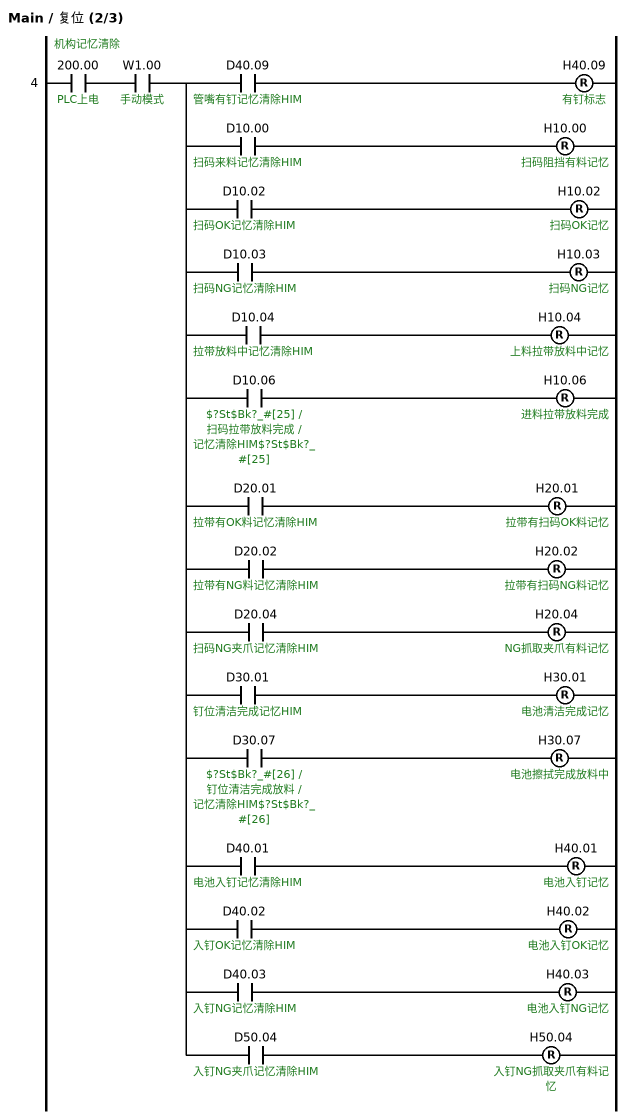
; rung 4: 机构记忆清除
LD 200.00  ; PLC上电
AND W1.00  ; 手动模式
OUT TR0
AND D40.09  ; 管嘴有钉记忆清除HIM
RSET H40.09  ; 有钉标志
LD TR0
AND D10.00  ; 扫码来料记忆清除HIM
RSET H10.00  ; 扫码阻挡有料记忆
LD TR0
AND D10.02  ; 扫码OK记忆清除HIM
RSET H10.02  ; 扫码OK记忆
LD TR0
AND D10.03  ; 扫码NG记忆清除HIM
RSET H10.03  ; 扫码NG记忆
LD TR0
AND D10.04  ; 拉带放料中记忆清除HIM
RSET H10.04  ; 上料拉带放料中记忆
LD TR0
AND D10.06  ; $?St$Bk?_#[25] / 扫码拉带放料完成 / 记忆清除HIM$?St$Bk?_#[25]
RSET H10.06  ; 进料拉带放料完成
LD TR0
AND D20.01  ; 拉带有OK料记忆清除HIM
RSET H20.01  ; 拉带有扫码OK料记忆
LD TR0
AND D20.02  ; 拉带有NG料记忆清除HIM
RSET H20.02  ; 拉带有扫码NG料记忆
LD TR0
AND D20.04  ; 扫码NG夹爪记忆清除HIM
RSET H20.04  ; NG抓取夹爪有料记忆
LD TR0
AND D30.01  ; 钉位清洁完成记忆HIM
RSET H30.01  ; 电池清洁完成记忆
LD TR0
AND D30.07  ; $?St$Bk?_#[26] / 钉位清洁完成放料 / 记忆清除HIM$?St$Bk?_#[26]
RSET H30.07  ; 电池擦拭完成放料中
LD TR0
AND D40.01  ; 电池入钉记忆清除HIM
RSET H40.01  ; 电池入钉记忆
LD TR0
AND D40.02  ; 入钉OK记忆清除HIM
RSET H40.02  ; 电池入钉OK记忆
LD TR0
AND D40.03  ; 入钉NG记忆清除HIM
RSET H40.03  ; 电池入钉NG记忆
LD TR0
AND D50.04  ; 入钉NG夹爪记忆清除HIM
RSET H50.04  ; 入钉NG抓取夹爪有料记忆

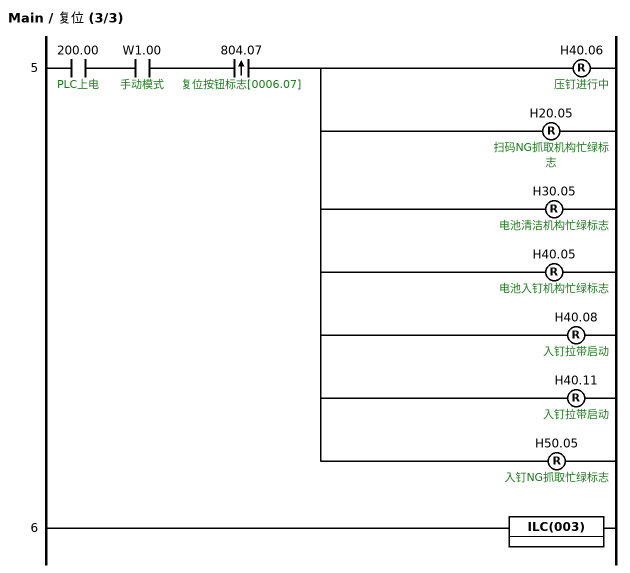
; rung 5
LD 200.00  ; PLC上电
AND W1.00  ; 手动模式
@AND 804.07  ; 复位按钮标志[0006.07]
RSET H40.06  ; 压钉进行中
RSET H20.05  ; 扫码NG抓取机构忙绿标志
RSET H30.05  ; 电池清洁机构忙绿标志
RSET H40.05  ; 电池入钉机构忙绿标志
RSET H40.08  ; 入钉拉带启动
RSET H40.11  ; 入钉拉带启动
RSET H50.05  ; 入钉NG抓取忙绿标志
; rung 6
ILC(003)

### Section 指示灯

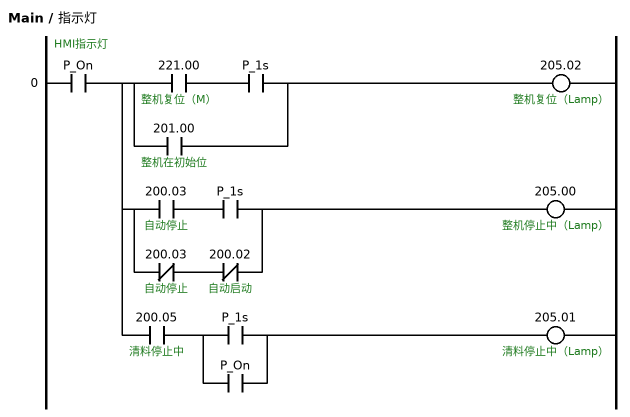
; rung 0: HMI指示灯
LD P_On
OUT TR0
LD 221.00  ; 整机复位（M）
AND P_1s
OR 201.00  ; 整机在初始位
ANDLD
OUT 205.02  ; 整机复位（Lamp）
LD TR0
LD 200.03  ; 自动停止
AND P_1s
LDNOT 200.03  ; 自动停止
ANDNOT 200.02  ; 自动启动
ORLD
ANDLD
OUT 205.00  ; 整机停止中（Lamp）
LD TR0
AND 200.05  ; 清料停止中
LD P_1s
OR P_On
ANDLD
OUT 205.01  ; 清料停止中（Lamp）

### Section 外部输出

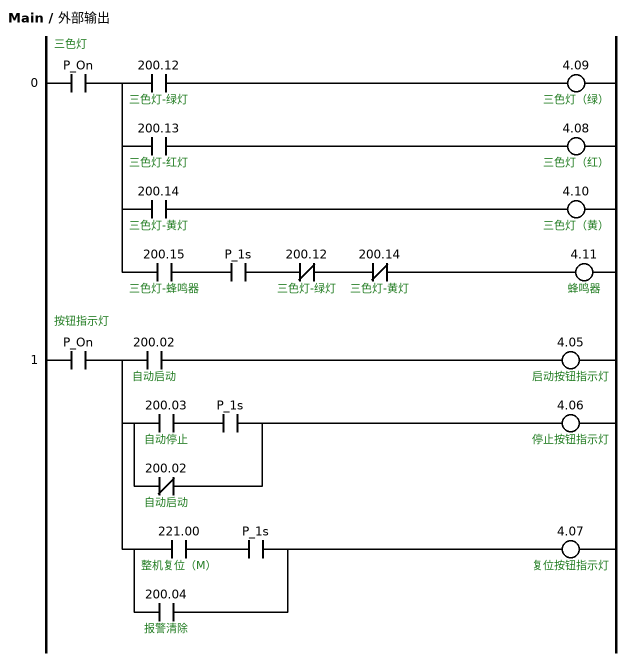
; rung 0: 三色灯
LD P_On
OUT TR0
AND 200.12  ; 三色灯-绿灯
OUT 4.09  ; 三色灯（绿）
LD TR0
AND 200.13  ; 三色灯-红灯
OUT 4.08  ; 三色灯（红）
LD TR0
AND 200.14  ; 三色灯-黄灯
OUT 4.10  ; 三色灯（黄）
LD TR0
AND 200.15  ; 三色灯-蜂鸣器
AND P_1s
ANDNOT 200.12  ; 三色灯-绿灯
ANDNOT 200.14  ; 三色灯-黄灯
OUT 4.11  ; 蜂鸣器
; rung 1: 按钮指示灯
LD P_On
OUT TR0
AND 200.02  ; 自动启动
OUT 4.05  ; 启动按钮指示灯
LD TR0
LD 200.03  ; 自动停止
AND P_1s
ORNOT 200.02  ; 自动启动
ANDLD
OUT 4.06  ; 停止按钮指示灯
LD TR0
LD 221.00  ; 整机复位（M）
AND P_1s
OR 200.04  ; 报警清除
ANDLD
OUT 4.07  ; 复位按钮指示灯

### Section END
; rung 0
END(001)

## Program 电池上料机构 (cyclic task 1)

### Section 主程序

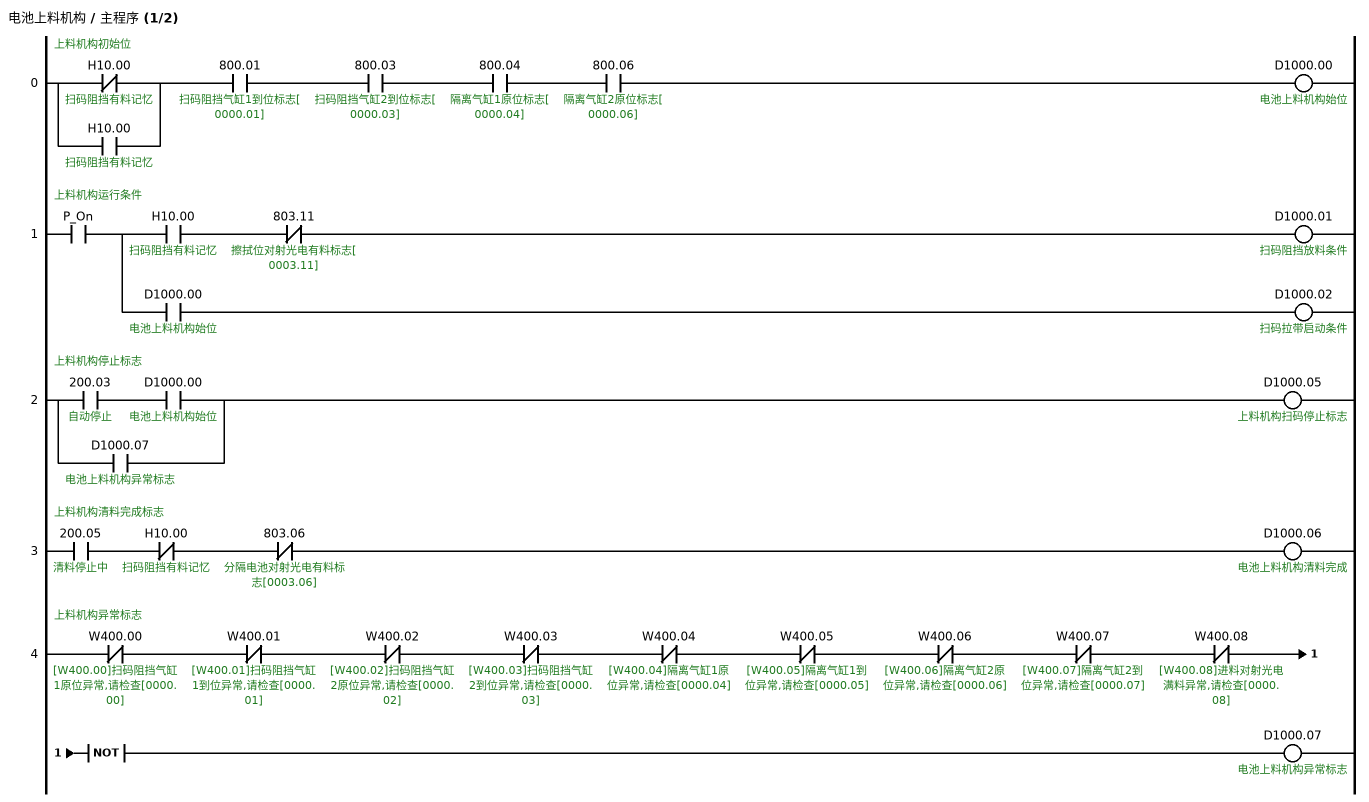
; rung 0: 上料机构初始位
LDNOT H10.00  ; 扫码阻挡有料记忆
OR H10.00  ; 扫码阻挡有料记忆
AND 800.01  ; 扫码阻挡气缸1到位标志[0000.01]
AND 800.03  ; 扫码阻挡气缸2到位标志[0000.03]
AND 800.04  ; 隔离气缸1原位标志[0000.04]
AND 800.06  ; 隔离气缸2原位标志[0000.06]
OUT D1000.00  ; 电池上料机构始位
; rung 1: 上料机构运行条件
LD P_On
OUT TR0
AND H10.00  ; 扫码阻挡有料记忆
ANDNOT 803.11  ; 擦拭位对射光电有料标志[0003.11]
OUT D1000.01  ; 扫码阻挡放料条件
LD TR0
AND D1000.00  ; 电池上料机构始位
OUT D1000.02  ; 扫码拉带启动条件
; rung 2: 上料机构停止标志
LD 200.03  ; 自动停止
AND D1000.00  ; 电池上料机构始位
OR D1000.07  ; 电池上料机构异常标志
OUT D1000.05  ; 上料机构扫码停止标志
; rung 3: 上料机构清料完成标志
LD 200.05  ; 清料停止中
ANDNOT H10.00  ; 扫码阻挡有料记忆
ANDNOT 803.06  ; 分隔电池对射光电有料标志[0003.06]
OUT D1000.06  ; 电池上料机构清料完成
; rung 4: 上料机构异常标志
LDNOT W400.00  ; [W400.00]扫码阻挡气缸1原位异常,请检查[0000.00]
ANDNOT W400.01  ; [W400.01]扫码阻挡气缸1到位异常,请检查[0000.01]
ANDNOT W400.02  ; [W400.02]扫码阻挡气缸2原位异常,请检查[0000.02]
ANDNOT W400.03  ; [W400.03]扫码阻挡气缸2到位异常,请检查[0000.03]
ANDNOT W400.04  ; [W400.04]隔离气缸1原位异常,请检查[0000.04]
ANDNOT W400.05  ; [W400.05]隔离气缸1到位异常,请检查[0000.05]
ANDNOT W400.06  ; [W400.06]隔离气缸2原位异常,请检查[0000.06]
ANDNOT W400.07  ; [W400.07]隔离气缸2到位异常,请检查[0000.07]
ANDNOT W400.08  ; [W400.08]进料对射光电满料异常,请检查[0000.08]
NOT(520)
OUT D1000.07  ; 电池上料机构异常标志

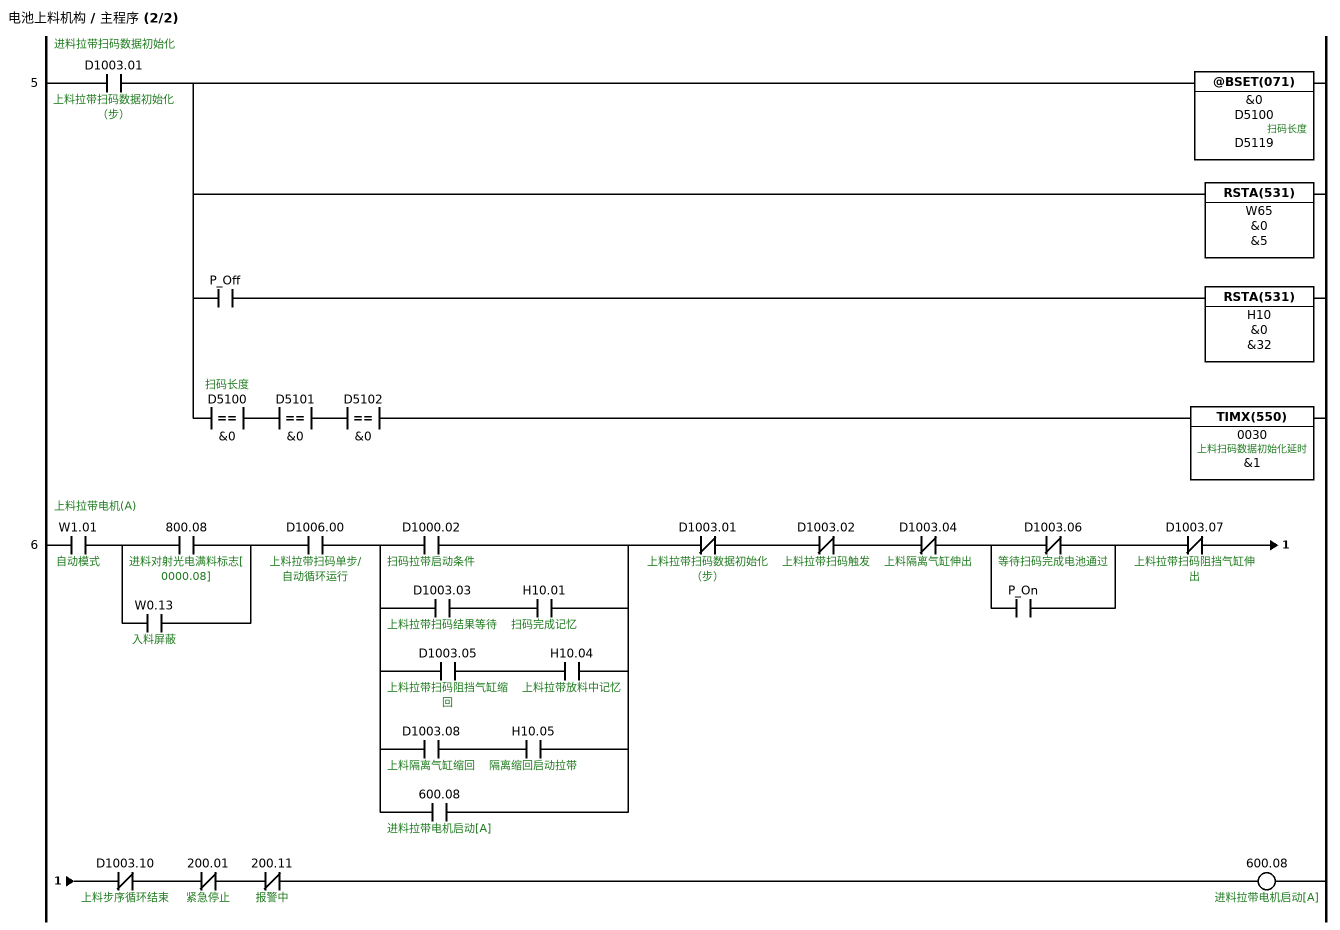
; rung 5: 进料拉带扫码数据初始化
LD D1003.01  ; 上料拉带扫码数据初始化（步）
OUT TR0
@BSET(071) &0 D5100 D5119  ; 扫码长度
RSTA(531) W65 &0 &5
AND P_Off
RSTA(531) H10 &0 &32
LD TR0
AND=(300) D5100 &0  ; 扫码长度
AND=(300) D5101 &0
AND=(300) D5102 &0
TIMX(550) 0030 &1  ; 上料扫码数据初始化延时
; rung 6: 上料拉带电机(A)
LD W1.01  ; 自动模式
LD 800.08  ; 进料对射光电满料标志[0000.08]
OR W0.13  ; 入料屏蔽
ANDLD
AND D1006.00  ; 上料拉带扫码单步/自动循环运行
LD D1000.02  ; 扫码拉带启动条件
LD D1003.03  ; 上料拉带扫码结果等待
AND H10.01  ; 扫码完成记忆
ORLD
LD D1003.05  ; 上料拉带扫码阻挡气缸缩回
AND H10.04  ; 上料拉带放料中记忆
ORLD
LD D1003.08  ; 上料隔离气缸缩回
AND H10.05  ; 隔离缩回启动拉带
ORLD
OR 600.08  ; 进料拉带电机启动[A]
ANDLD
ANDNOT D1003.01  ; 上料拉带扫码数据初始化（步）
ANDNOT D1003.02  ; 上料拉带扫码触发
ANDNOT D1003.04  ; 上料隔离气缸伸出
LDNOT D1003.06  ; 等待扫码完成电池通过
OR P_On
ANDLD
ANDNOT D1003.07  ; 上料拉带扫码阻挡气缸伸出
ANDNOT D1003.10  ; 上料步序循环结束
ANDNOT 200.01  ; 紧急停止
ANDNOT 200.11  ; 报警中
OUT 600.08  ; 进料拉带电机启动[A]

### Section 工站复位

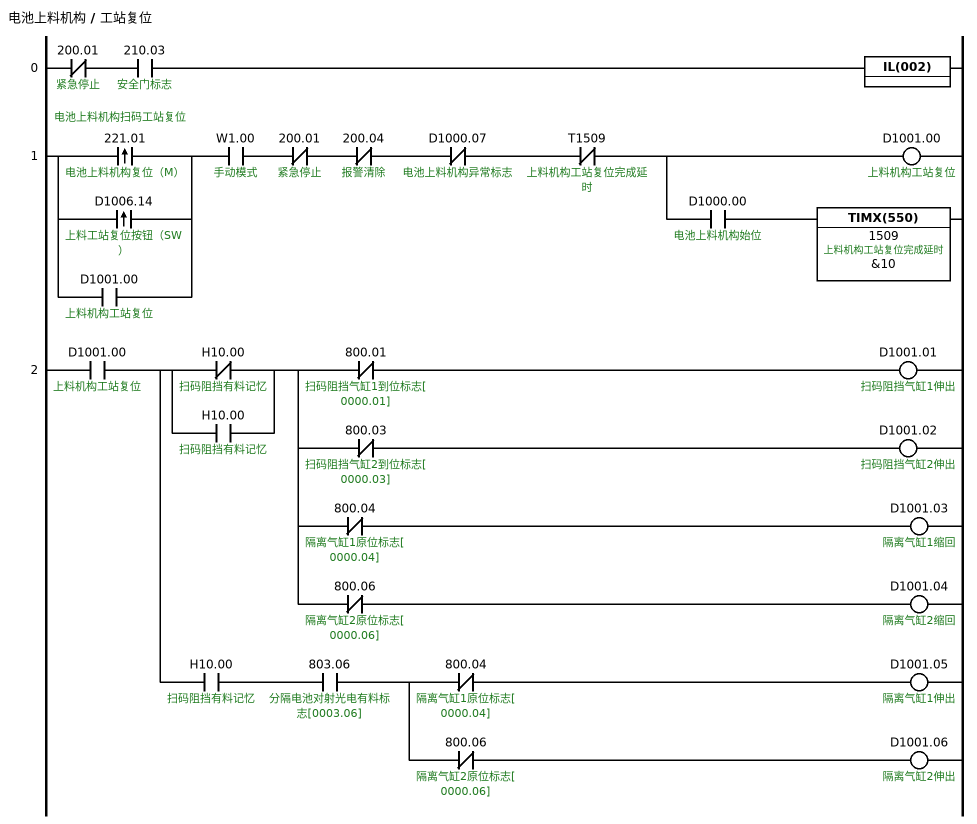
; rung 0
LDNOT 200.01  ; 紧急停止
AND 210.03  ; 安全门标志
IL(002)
; rung 1: 电池上料机构扫码工站复位
@LD 221.01  ; 电池上料机构复位（M）
@OR D1006.14  ; 上料工站复位按钮（SW）
OR D1001.00  ; 上料机构工站复位
AND W1.00  ; 手动模式
ANDNOT 200.01  ; 紧急停止
ANDNOT 200.04  ; 报警清除
ANDNOT D1000.07  ; 电池上料机构异常标志
ANDNOT T1509  ; 上料机构工站复位完成延时
OUT D1001.00  ; 上料机构工站复位
AND D1000.00  ; 电池上料机构始位
TIMX(550) 1509 &10  ; 上料机构工站复位完成延时
; rung 2
LD D1001.00  ; 上料机构工站复位
OUT TR0
LDNOT H10.00  ; 扫码阻挡有料记忆
OR H10.00  ; 扫码阻挡有料记忆
ANDLD
OUT TR1
ANDNOT 800.01  ; 扫码阻挡气缸1到位标志[0000.01]
OUT D1001.01  ; 扫码阻挡气缸1伸出
LD TR1
ANDNOT 800.03  ; 扫码阻挡气缸2到位标志[0000.03]
OUT D1001.02  ; 扫码阻挡气缸2伸出
LD TR1
ANDNOT 800.04  ; 隔离气缸1原位标志[0000.04]
OUT D1001.03  ; 隔离气缸1缩回
LD TR1
ANDNOT 800.06  ; 隔离气缸2原位标志[0000.06]
OUT D1001.04  ; 隔离气缸2缩回
LD TR0
AND H10.00  ; 扫码阻挡有料记忆
AND 803.06  ; 分隔电池对射光电有料标志[0003.06]
OUT TR0
ANDNOT 800.04  ; 隔离气缸1原位标志[0000.04]
OUT D1001.05  ; 隔离气缸1伸出
LD TR0
ANDNOT 800.06  ; 隔离气缸2原位标志[0000.06]
OUT D1001.06  ; 隔离气缸2伸出

### Section 手动程序

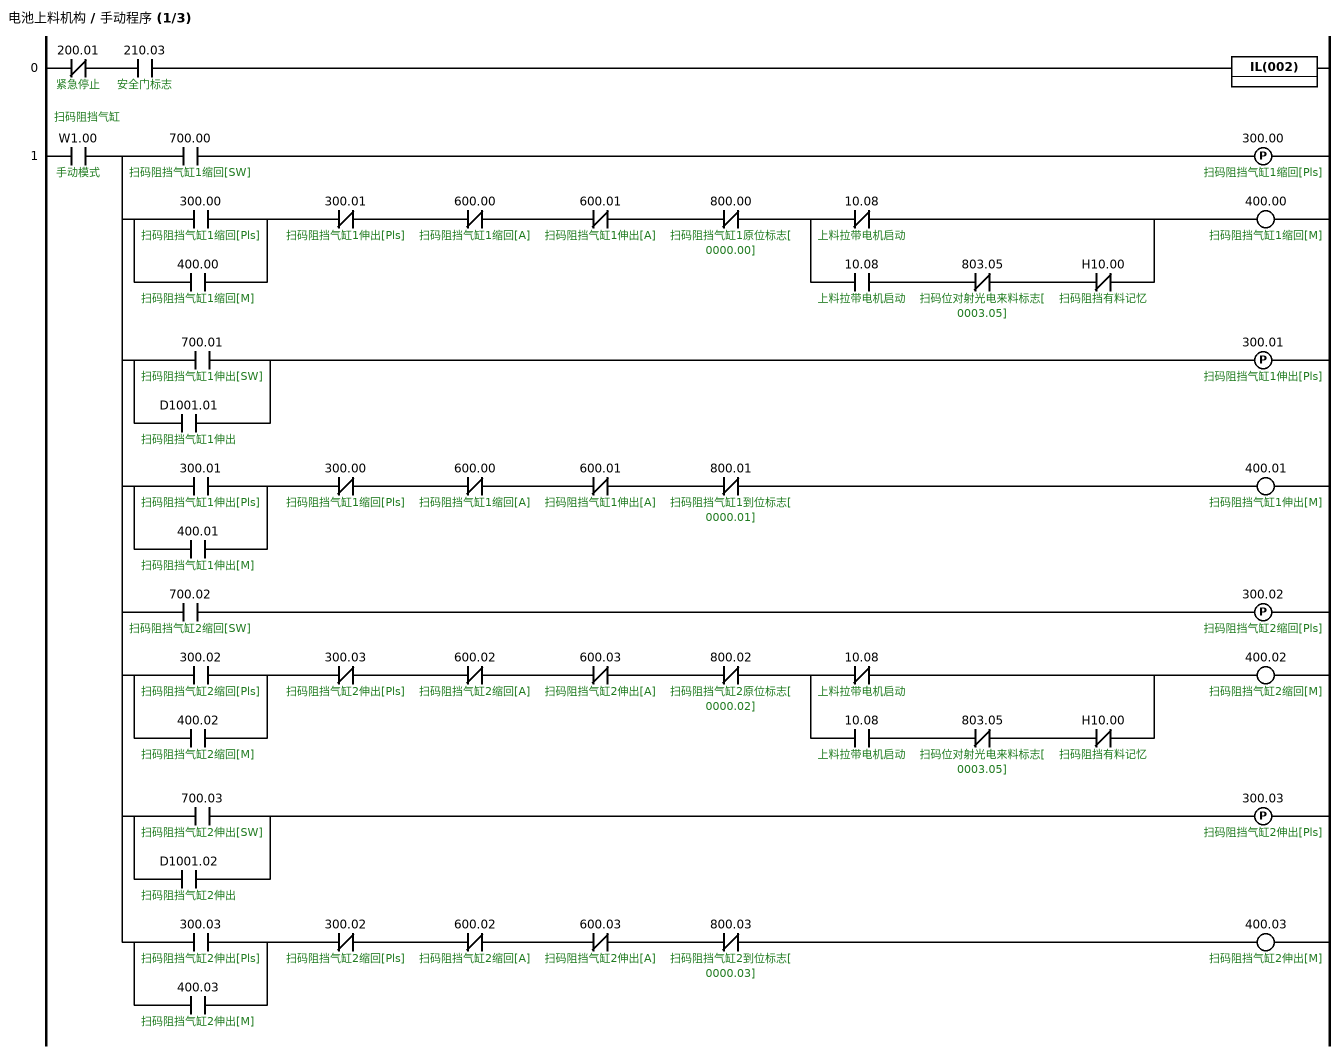
; rung 0
LDNOT 200.01  ; 紧急停止
AND 210.03  ; 安全门标志
IL(002)
; rung 1: 扫码阻挡气缸
LD W1.00  ; 手动模式
OUT TR0
AND 700.00  ; 扫码阻挡气缸1缩回[SW]
DIFU(013) 300.00  ; 扫码阻挡气缸1缩回[Pls]
LD TR0
LD 300.00  ; 扫码阻挡气缸1缩回[Pls]
OR 400.00  ; 扫码阻挡气缸1缩回[M]
ANDLD
ANDNOT 300.01  ; 扫码阻挡气缸1伸出[Pls]
ANDNOT 600.00  ; 扫码阻挡气缸1缩回[A]
ANDNOT 600.01  ; 扫码阻挡气缸1伸出[A]
ANDNOT 800.00  ; 扫码阻挡气缸1原位标志[0000.00]
LDNOT 10.08  ; 上料拉带电机启动
LD 10.08  ; 上料拉带电机启动
ANDNOT 803.05  ; 扫码位对射光电来料标志[0003.05]
ANDNOT H10.00  ; 扫码阻挡有料记忆
ORLD
ANDLD
OUT 400.00  ; 扫码阻挡气缸1缩回[M]
LD TR0
LD 700.01  ; 扫码阻挡气缸1伸出[SW]
OR D1001.01  ; 扫码阻挡气缸1伸出
ANDLD
DIFU(013) 300.01  ; 扫码阻挡气缸1伸出[Pls]
LD TR0
LD 300.01  ; 扫码阻挡气缸1伸出[Pls]
OR 400.01  ; 扫码阻挡气缸1伸出[M]
ANDLD
ANDNOT 300.00  ; 扫码阻挡气缸1缩回[Pls]
ANDNOT 600.00  ; 扫码阻挡气缸1缩回[A]
ANDNOT 600.01  ; 扫码阻挡气缸1伸出[A]
ANDNOT 800.01  ; 扫码阻挡气缸1到位标志[0000.01]
OUT 400.01  ; 扫码阻挡气缸1伸出[M]
LD TR0
AND 700.02  ; 扫码阻挡气缸2缩回[SW]
DIFU(013) 300.02  ; 扫码阻挡气缸2缩回[Pls]
LD TR0
LD 300.02  ; 扫码阻挡气缸2缩回[Pls]
OR 400.02  ; 扫码阻挡气缸2缩回[M]
ANDLD
ANDNOT 300.03  ; 扫码阻挡气缸2伸出[Pls]
ANDNOT 600.02  ; 扫码阻挡气缸2缩回[A]
ANDNOT 600.03  ; 扫码阻挡气缸2伸出[A]
ANDNOT 800.02  ; 扫码阻挡气缸2原位标志[0000.02]
LDNOT 10.08  ; 上料拉带电机启动
LD 10.08  ; 上料拉带电机启动
ANDNOT 803.05  ; 扫码位对射光电来料标志[0003.05]
ANDNOT H10.00  ; 扫码阻挡有料记忆
ORLD
ANDLD
OUT 400.02  ; 扫码阻挡气缸2缩回[M]
LD TR0
LD 700.03  ; 扫码阻挡气缸2伸出[SW]
OR D1001.02  ; 扫码阻挡气缸2伸出
ANDLD
DIFU(013) 300.03  ; 扫码阻挡气缸2伸出[Pls]
LD TR0
LD 300.03  ; 扫码阻挡气缸2伸出[Pls]
OR 400.03  ; 扫码阻挡气缸2伸出[M]
ANDLD
ANDNOT 300.02  ; 扫码阻挡气缸2缩回[Pls]
ANDNOT 600.02  ; 扫码阻挡气缸2缩回[A]
ANDNOT 600.03  ; 扫码阻挡气缸2伸出[A]
ANDNOT 800.03  ; 扫码阻挡气缸2到位标志[0000.03]
OUT 400.03  ; 扫码阻挡气缸2伸出[M]

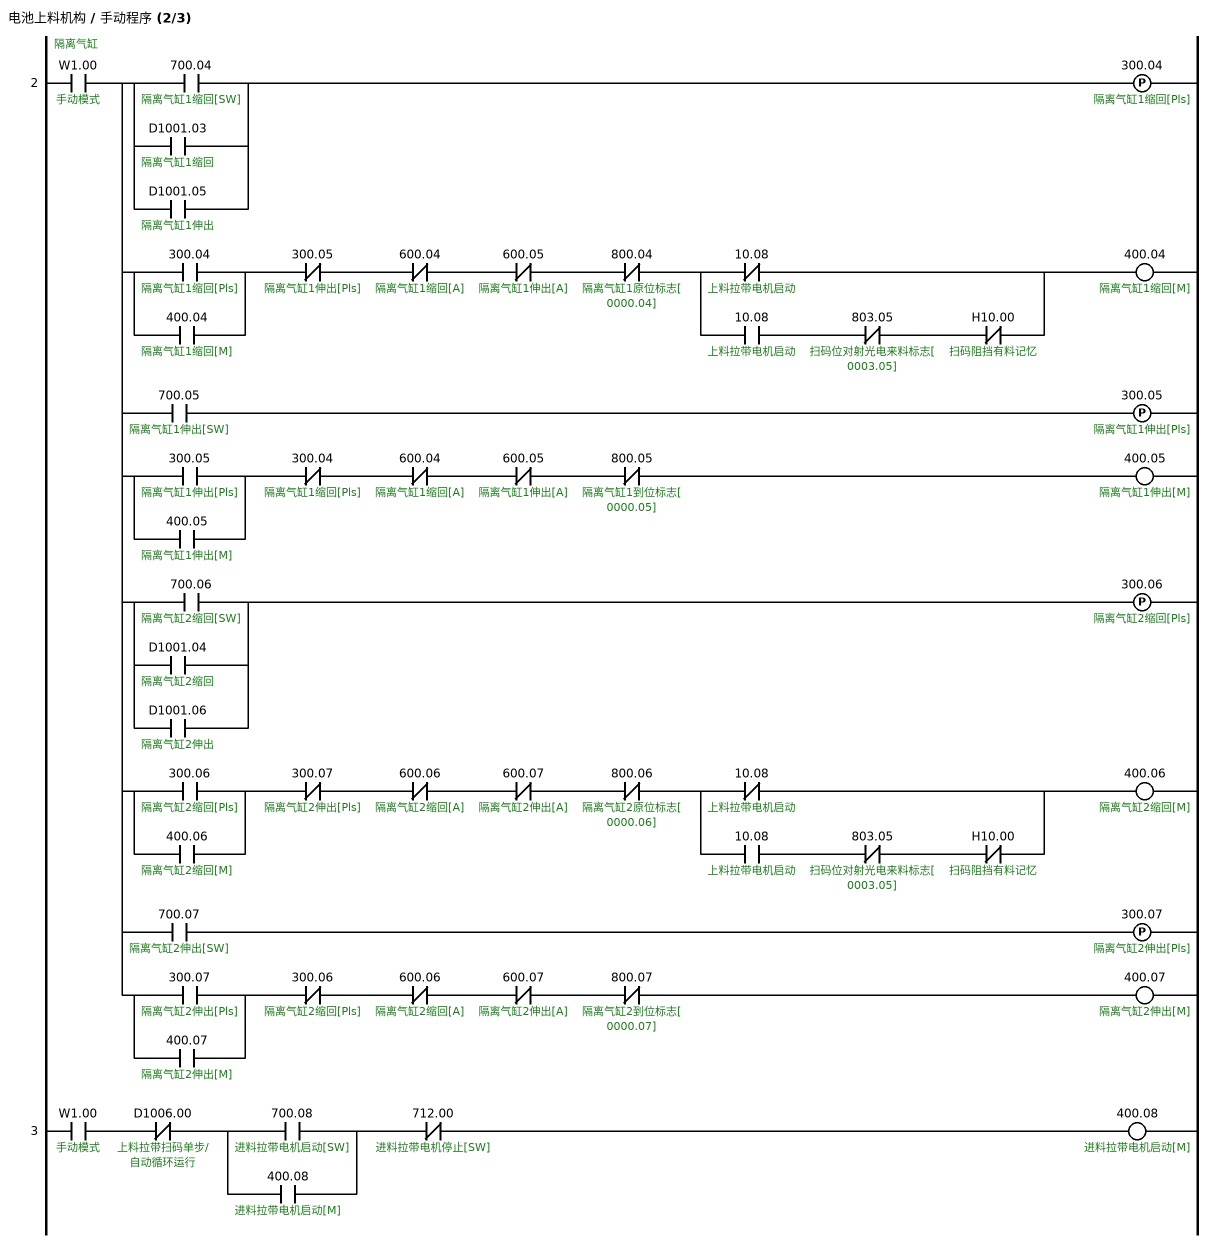
; rung 2: 隔离气缸
LD W1.00  ; 手动模式
OUT TR0
LD 700.04  ; 隔离气缸1缩回[SW]
OR D1001.03  ; 隔离气缸1缩回
OR D1001.05  ; 隔离气缸1伸出
ANDLD
DIFU(013) 300.04  ; 隔离气缸1缩回[Pls]
LD TR0
LD 300.04  ; 隔离气缸1缩回[Pls]
OR 400.04  ; 隔离气缸1缩回[M]
ANDLD
ANDNOT 300.05  ; 隔离气缸1伸出[Pls]
ANDNOT 600.04  ; 隔离气缸1缩回[A]
ANDNOT 600.05  ; 隔离气缸1伸出[A]
ANDNOT 800.04  ; 隔离气缸1原位标志[0000.04]
LDNOT 10.08  ; 上料拉带电机启动
LD 10.08  ; 上料拉带电机启动
ANDNOT 803.05  ; 扫码位对射光电来料标志[0003.05]
ANDNOT H10.00  ; 扫码阻挡有料记忆
ORLD
ANDLD
OUT 400.04  ; 隔离气缸1缩回[M]
LD TR0
AND 700.05  ; 隔离气缸1伸出[SW]
DIFU(013) 300.05  ; 隔离气缸1伸出[Pls]
LD TR0
LD 300.05  ; 隔离气缸1伸出[Pls]
OR 400.05  ; 隔离气缸1伸出[M]
ANDLD
ANDNOT 300.04  ; 隔离气缸1缩回[Pls]
ANDNOT 600.04  ; 隔离气缸1缩回[A]
ANDNOT 600.05  ; 隔离气缸1伸出[A]
ANDNOT 800.05  ; 隔离气缸1到位标志[0000.05]
OUT 400.05  ; 隔离气缸1伸出[M]
LD TR0
LD 700.06  ; 隔离气缸2缩回[SW]
OR D1001.04  ; 隔离气缸2缩回
OR D1001.06  ; 隔离气缸2伸出
ANDLD
DIFU(013) 300.06  ; 隔离气缸2缩回[Pls]
LD TR0
LD 300.06  ; 隔离气缸2缩回[Pls]
OR 400.06  ; 隔离气缸2缩回[M]
ANDLD
ANDNOT 300.07  ; 隔离气缸2伸出[Pls]
ANDNOT 600.06  ; 隔离气缸2缩回[A]
ANDNOT 600.07  ; 隔离气缸2伸出[A]
ANDNOT 800.06  ; 隔离气缸2原位标志[0000.06]
LDNOT 10.08  ; 上料拉带电机启动
LD 10.08  ; 上料拉带电机启动
ANDNOT 803.05  ; 扫码位对射光电来料标志[0003.05]
ANDNOT H10.00  ; 扫码阻挡有料记忆
ORLD
ANDLD
OUT 400.06  ; 隔离气缸2缩回[M]
LD TR0
AND 700.07  ; 隔离气缸2伸出[SW]
DIFU(013) 300.07  ; 隔离气缸2伸出[Pls]
LD TR0
LD 300.07  ; 隔离气缸2伸出[Pls]
OR 400.07  ; 隔离气缸2伸出[M]
ANDLD
ANDNOT 300.06  ; 隔离气缸2缩回[Pls]
ANDNOT 600.06  ; 隔离气缸2缩回[A]
ANDNOT 600.07  ; 隔离气缸2伸出[A]
ANDNOT 800.07  ; 隔离气缸2到位标志[0000.07]
OUT 400.07  ; 隔离气缸2伸出[M]
; rung 3
LD W1.00  ; 手动模式
ANDNOT D1006.00  ; 上料拉带扫码单步/自动循环运行
LD 700.08  ; 进料拉带电机启动[SW]
OR 400.08  ; 进料拉带电机启动[M]
ANDLD
ANDNOT 712.00  ; 进料拉带电机停止[SW]
OUT 400.08  ; 进料拉带电机启动[M]

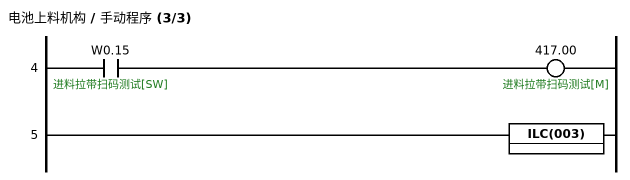
; rung 4
LD W0.15  ; 进料拉带扫码测试[SW]
OUT 417.00  ; 进料拉带扫码测试[M]
; rung 5
ILC(003)

### Section 自动程序

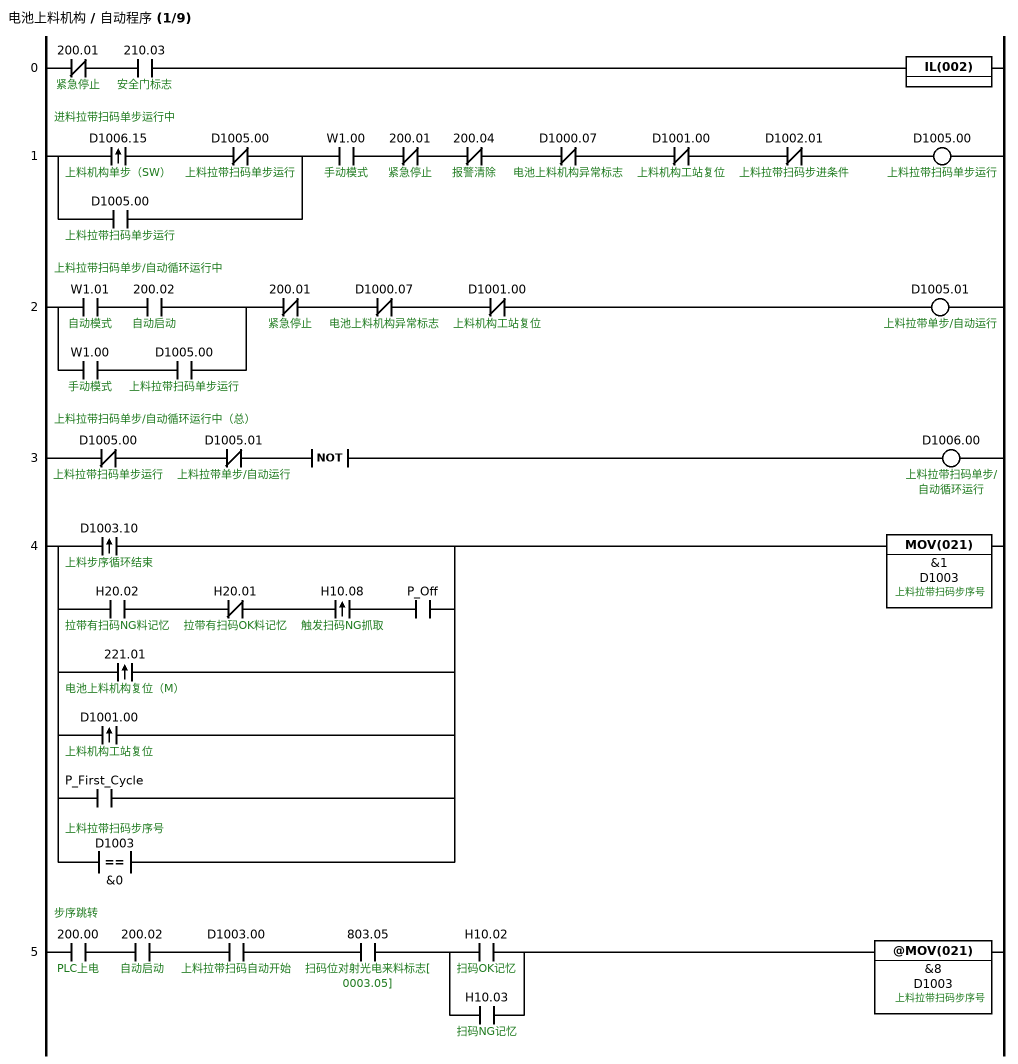
; rung 0
LDNOT 200.01  ; 紧急停止
AND 210.03  ; 安全门标志
IL(002)
; rung 1: 进料拉带扫码单步运行中
@LD D1006.15  ; 上料机构单步（SW）
ANDNOT D1005.00  ; 上料拉带扫码单步运行
OR D1005.00  ; 上料拉带扫码单步运行
AND W1.00  ; 手动模式
ANDNOT 200.01  ; 紧急停止
ANDNOT 200.04  ; 报警清除
ANDNOT D1000.07  ; 电池上料机构异常标志
ANDNOT D1001.00  ; 上料机构工站复位
ANDNOT D1002.01  ; 上料拉带扫码步进条件
OUT D1005.00  ; 上料拉带扫码单步运行
; rung 2: 上料拉带扫码单步/自动循环运行中
LD W1.01  ; 自动模式
AND 200.02  ; 自动启动
LD W1.00  ; 手动模式
AND D1005.00  ; 上料拉带扫码单步运行
ORLD
ANDNOT 200.01  ; 紧急停止
ANDNOT D1000.07  ; 电池上料机构异常标志
ANDNOT D1001.00  ; 上料机构工站复位
OUT D1005.01  ; 上料拉带单步/自动运行
; rung 3: 上料拉带扫码单步/自动循环运行中（总）
LDNOT D1005.00  ; 上料拉带扫码单步运行
ANDNOT D1005.01  ; 上料拉带单步/自动运行
NOT(520)
OUT D1006.00  ; 上料拉带扫码单步/自动循环运行
; rung 4
@LD D1003.10  ; 上料步序循环结束
LD H20.02  ; 拉带有扫码NG料记忆
ANDNOT H20.01  ; 拉带有扫码OK料记忆
@AND H10.08  ; 触发扫码NG抓取
AND P_Off
ORLD
@OR 221.01  ; 电池上料机构复位（M）
@OR D1001.00  ; 上料机构工站复位
OR P_First_Cycle
OR=(300) D1003 &0  ; 上料拉带扫码步序号
MOV(021) &1 D1003  ; 上料拉带扫码步序号
; rung 5: 步序跳转
LD 200.00  ; PLC上电
AND 200.02  ; 自动启动
AND D1003.00  ; 上料拉带扫码自动开始
AND 803.05  ; 扫码位对射光电来料标志[0003.05]
LD H10.02  ; 扫码OK记忆
OR H10.03  ; 扫码NG记忆
ANDLD
@MOV(021) &8 D1003  ; 上料拉带扫码步序号

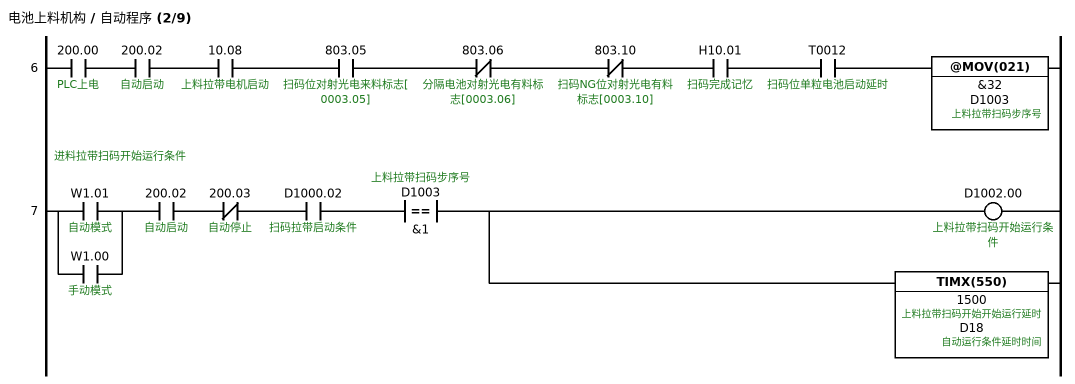
; rung 6
LD 200.00  ; PLC上电
AND 200.02  ; 自动启动
AND 10.08  ; 上料拉带电机启动
AND 803.05  ; 扫码位对射光电来料标志[0003.05]
ANDNOT 803.06  ; 分隔电池对射光电有料标志[0003.06]
ANDNOT 803.10  ; 扫码NG位对射光电有料标志[0003.10]
AND H10.01  ; 扫码完成记忆
AND T0012  ; 扫码位单粒电池启动延时
@MOV(021) &32 D1003  ; 上料拉带扫码步序号
; rung 7: 进料拉带扫码开始运行条件
LD W1.01  ; 自动模式
OR W1.00  ; 手动模式
AND 200.02  ; 自动启动
ANDNOT 200.03  ; 自动停止
AND D1000.02  ; 扫码拉带启动条件
AND=(300) D1003 &1  ; 上料拉带扫码步序号
OUT D1002.00  ; 上料拉带扫码开始运行条件
TIMX(550) 1500 D18  ; 自动运行条件延时时间, 上料拉带扫码开始开始运行延时

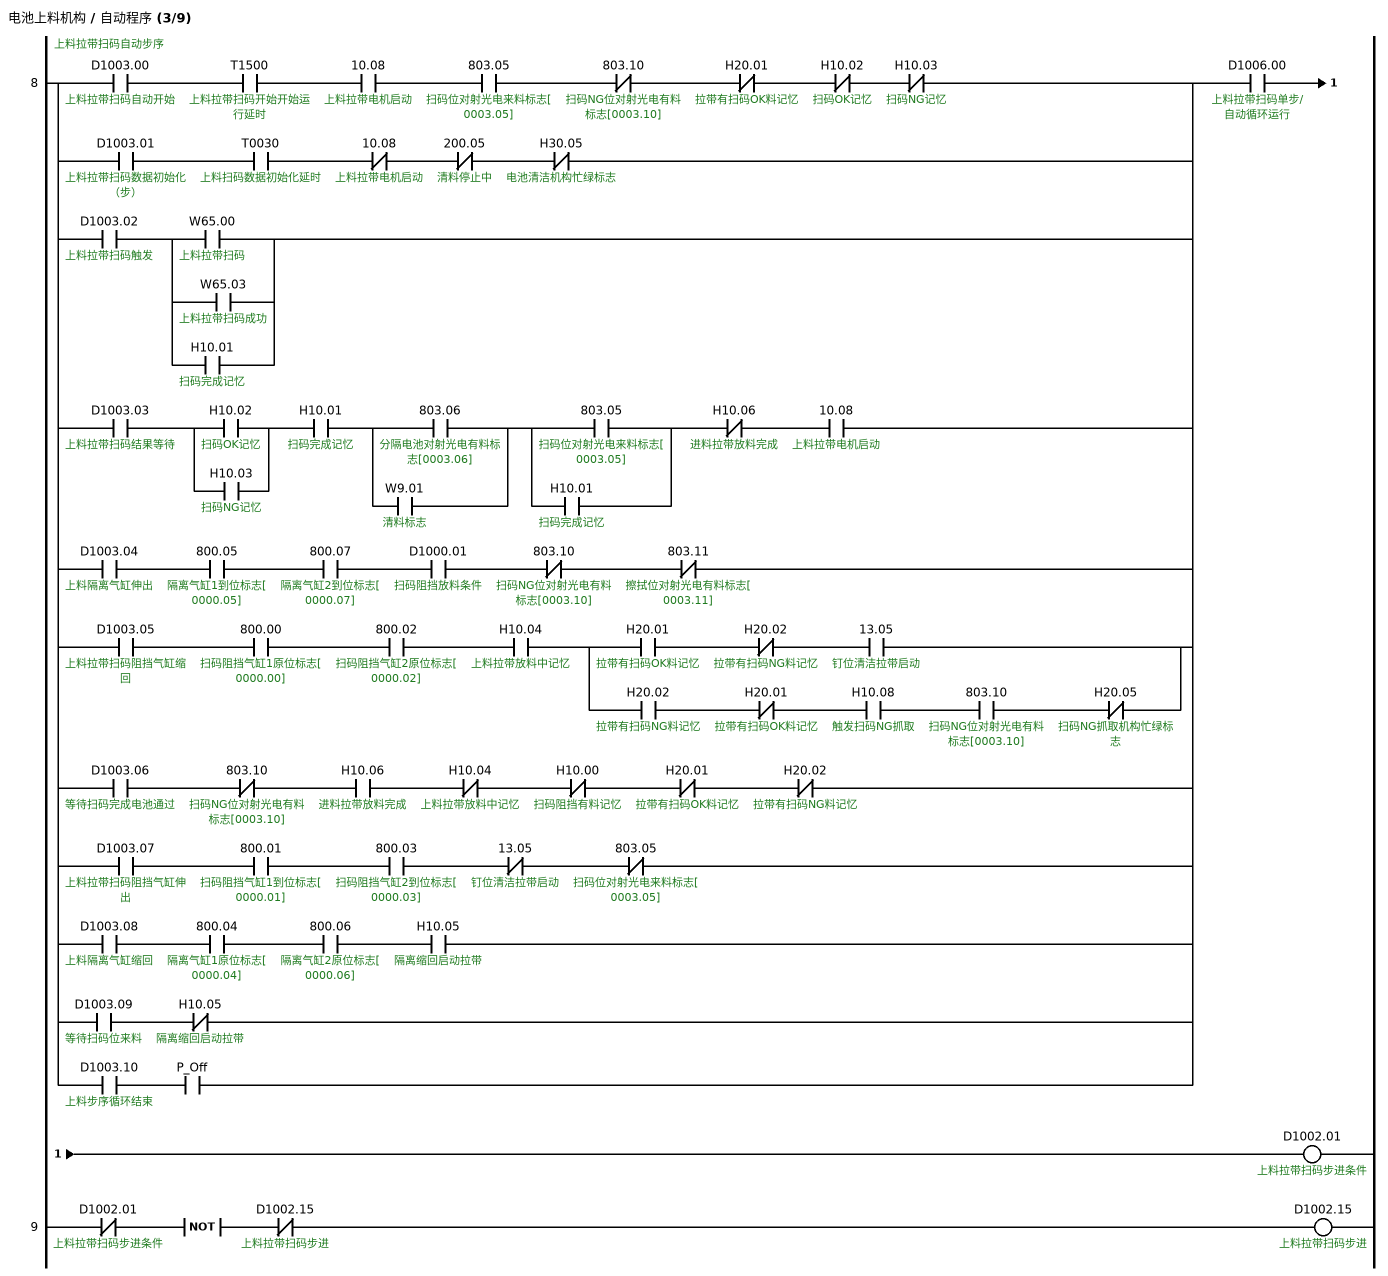
; rung 8: 上料拉带扫码自动步序
LD D1003.00  ; 上料拉带扫码自动开始
AND T1500  ; 上料拉带扫码开始开始运行延时
AND 10.08  ; 上料拉带电机启动
AND 803.05  ; 扫码位对射光电来料标志[0003.05]
ANDNOT 803.10  ; 扫码NG位对射光电有料标志[0003.10]
ANDNOT H20.01  ; 拉带有扫码OK料记忆
ANDNOT H10.02  ; 扫码OK记忆
ANDNOT H10.03  ; 扫码NG记忆
LD D1003.01  ; 上料拉带扫码数据初始化（步）
AND T0030  ; 上料扫码数据初始化延时
ANDNOT 10.08  ; 上料拉带电机启动
ANDNOT 200.05  ; 清料停止中
ANDNOT H30.05  ; 电池清洁机构忙绿标志
ORLD
LD D1003.02  ; 上料拉带扫码触发
LD W65.00  ; 上料拉带扫码
OR W65.03  ; 上料拉带扫码成功
OR H10.01  ; 扫码完成记忆
ANDLD
ORLD
LD D1003.03  ; 上料拉带扫码结果等待
LD H10.02  ; 扫码OK记忆
OR H10.03  ; 扫码NG记忆
ANDLD
AND H10.01  ; 扫码完成记忆
LD 803.06  ; 分隔电池对射光电有料标志[0003.06]
OR W9.01  ; 清料标志
ANDLD
LD 803.05  ; 扫码位对射光电来料标志[0003.05]
OR H10.01  ; 扫码完成记忆
ANDLD
ANDNOT H10.06  ; 进料拉带放料完成
AND 10.08  ; 上料拉带电机启动
ORLD
LD D1003.04  ; 上料隔离气缸伸出
AND 800.05  ; 隔离气缸1到位标志[0000.05]
AND 800.07  ; 隔离气缸2到位标志[0000.07]
AND D1000.01  ; 扫码阻挡放料条件
ANDNOT 803.10  ; 扫码NG位对射光电有料标志[0003.10]
ANDNOT 803.11  ; 擦拭位对射光电有料标志[0003.11]
ORLD
LD D1003.05  ; 上料拉带扫码阻挡气缸缩回
AND 800.00  ; 扫码阻挡气缸1原位标志[0000.00]
AND 800.02  ; 扫码阻挡气缸2原位标志[0000.02]
AND H10.04  ; 上料拉带放料中记忆
LD H20.01  ; 拉带有扫码OK料记忆
ANDNOT H20.02  ; 拉带有扫码NG料记忆
AND 13.05  ; 钉位清洁拉带启动
LD H20.02  ; 拉带有扫码NG料记忆
ANDNOT H20.01  ; 拉带有扫码OK料记忆
AND H10.08  ; 触发扫码NG抓取
AND 803.10  ; 扫码NG位对射光电有料标志[0003.10]
ANDNOT H20.05  ; 扫码NG抓取机构忙绿标志
ORLD
ANDLD
ORLD
LD D1003.06  ; 等待扫码完成电池通过
ANDNOT 803.10  ; 扫码NG位对射光电有料标志[0003.10]
AND H10.06  ; 进料拉带放料完成
ANDNOT H10.04  ; 上料拉带放料中记忆
ANDNOT H10.00  ; 扫码阻挡有料记忆
ANDNOT H20.01  ; 拉带有扫码OK料记忆
ANDNOT H20.02  ; 拉带有扫码NG料记忆
ORLD
LD D1003.07  ; 上料拉带扫码阻挡气缸伸出
AND 800.01  ; 扫码阻挡气缸1到位标志[0000.01]
AND 800.03  ; 扫码阻挡气缸2到位标志[0000.03]
ANDNOT 13.05  ; 钉位清洁拉带启动
ANDNOT 803.05  ; 扫码位对射光电来料标志[0003.05]
ORLD
LD D1003.08  ; 上料隔离气缸缩回
AND 800.04  ; 隔离气缸1原位标志[0000.04]
AND 800.06  ; 隔离气缸2原位标志[0000.06]
AND H10.05  ; 隔离缩回启动拉带
ORLD
LD D1003.09  ; 等待扫码位来料
ANDNOT H10.05  ; 隔离缩回启动拉带
ORLD
LD D1003.10  ; 上料步序循环结束
AND P_Off
ORLD
AND D1006.00  ; 上料拉带扫码单步/自动循环运行
OUT D1002.01  ; 上料拉带扫码步进条件
; rung 9
LDNOT D1002.01  ; 上料拉带扫码步进条件
NOT(520)
ANDNOT D1002.15  ; 上料拉带扫码步进
OUT D1002.15  ; 上料拉带扫码步进

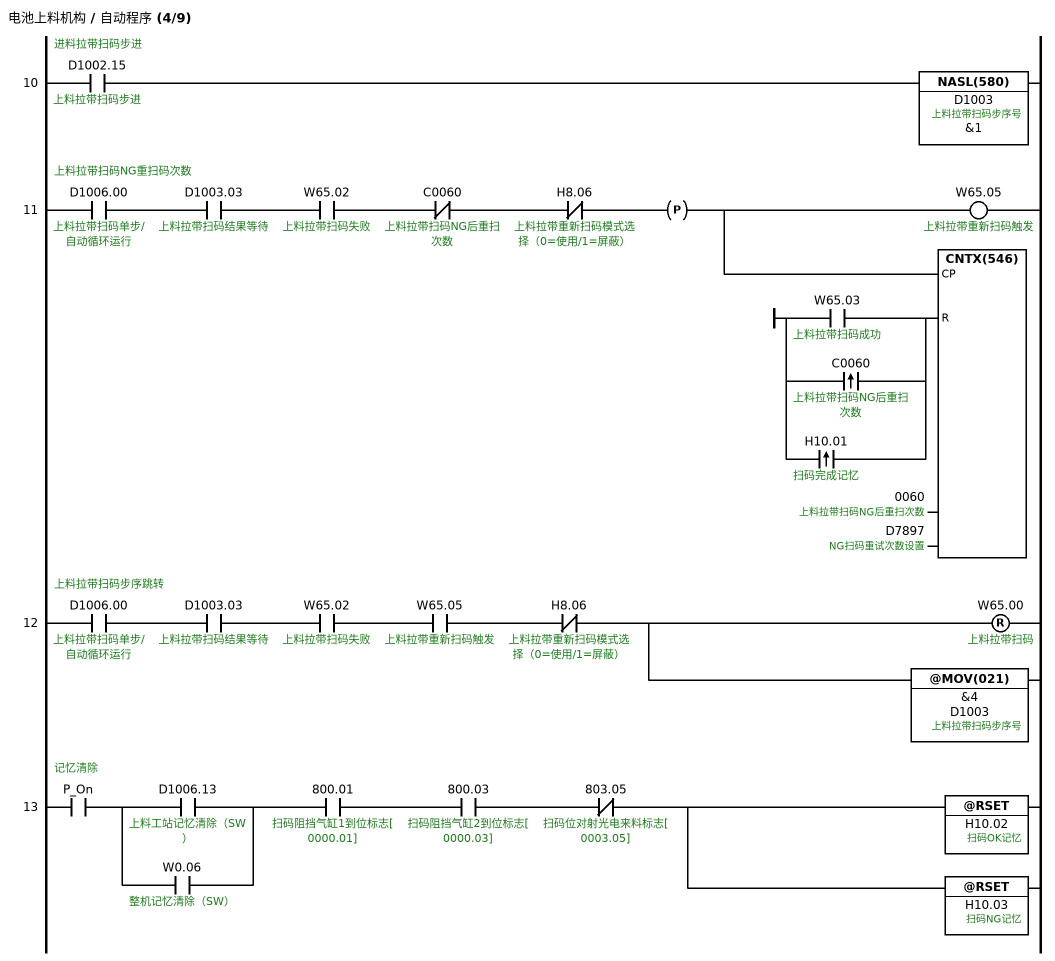
; rung 10: 进料拉带扫码步进
LD D1002.15  ; 上料拉带扫码步进
NASL(580) D1003 &1  ; 上料拉带扫码步序号
; rung 11: 上料拉带扫码NG重扫码次数
LD D1006.00  ; 上料拉带扫码单步/自动循环运行
AND D1003.03  ; 上料拉带扫码结果等待
AND W65.02  ; 上料拉带扫码失败
ANDNOT C0060  ; 上料拉带扫码NG后重扫次数
ANDNOT H8.06  ; 上料拉带重新扫码模式选择（0=使用/1=屏蔽）
UP(521)
OUT W65.05  ; 上料拉带重新扫码触发
LD W65.03  ; 上料拉带扫码成功
@OR C0060  ; 上料拉带扫码NG后重扫次数
@OR H10.01  ; 扫码完成记忆
CNTX(546) 0060 D7897  ; NG扫码重试次数设置, 上料拉带扫码NG后重扫次数
; rung 12: 上料拉带扫码步序跳转
LD D1006.00  ; 上料拉带扫码单步/自动循环运行
AND D1003.03  ; 上料拉带扫码结果等待
AND W65.02  ; 上料拉带扫码失败
AND W65.05  ; 上料拉带重新扫码触发
ANDNOT H8.06  ; 上料拉带重新扫码模式选择（0=使用/1=屏蔽）
RSET W65.00  ; 上料拉带扫码
@MOV(021) &4 D1003  ; 上料拉带扫码步序号
; rung 13: 记忆清除
LD P_On
LD D1006.13  ; 上料工站记忆清除（SW）
OR W0.06  ; 整机记忆清除（SW）
ANDLD
AND 800.01  ; 扫码阻挡气缸1到位标志[0000.01]
AND 800.03  ; 扫码阻挡气缸2到位标志[0000.03]
ANDNOT 803.05  ; 扫码位对射光电来料标志[0003.05]
@RSET H10.02  ; 扫码OK记忆
@RSET H10.03  ; 扫码NG记忆

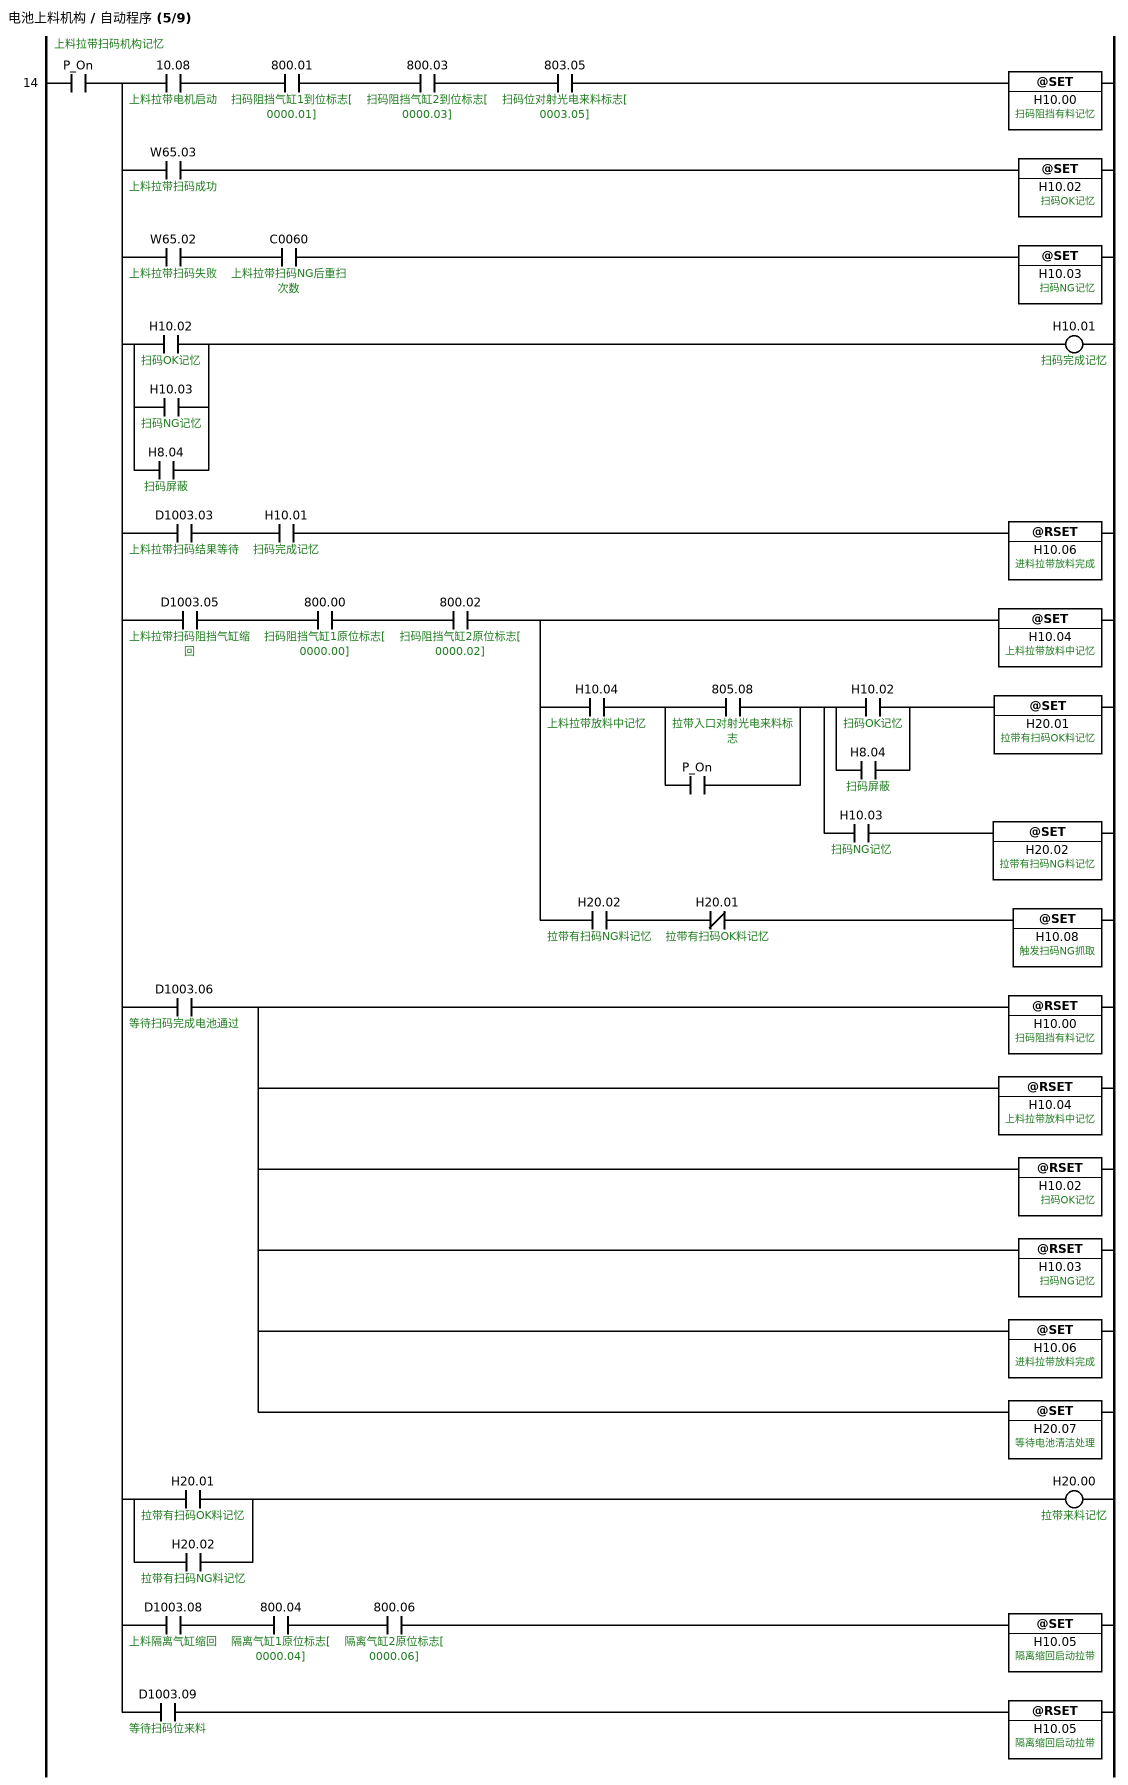
; rung 14: 上料拉带扫码机构记忆
LD P_On
OUT TR0
AND 10.08  ; 上料拉带电机启动
AND 800.01  ; 扫码阻挡气缸1到位标志[0000.01]
AND 800.03  ; 扫码阻挡气缸2到位标志[0000.03]
AND 803.05  ; 扫码位对射光电来料标志[0003.05]
@SET H10.00  ; 扫码阻挡有料记忆
LD TR0
AND W65.03  ; 上料拉带扫码成功
@SET H10.02  ; 扫码OK记忆
LD TR0
AND W65.02  ; 上料拉带扫码失败
AND C0060  ; 上料拉带扫码NG后重扫次数
@SET H10.03  ; 扫码NG记忆
LD TR0
LD H10.02  ; 扫码OK记忆
OR H10.03  ; 扫码NG记忆
OR H8.04  ; 扫码屏蔽
ANDLD
OUT H10.01  ; 扫码完成记忆
LD TR0
AND D1003.03  ; 上料拉带扫码结果等待
AND H10.01  ; 扫码完成记忆
@RSET H10.06  ; 进料拉带放料完成
LD TR0
AND D1003.05  ; 上料拉带扫码阻挡气缸缩回
AND 800.00  ; 扫码阻挡气缸1原位标志[0000.00]
AND 800.02  ; 扫码阻挡气缸2原位标志[0000.02]
OUT TR1
@SET H10.04  ; 上料拉带放料中记忆
AND H10.04  ; 上料拉带放料中记忆
LD 805.08  ; 拉带入口对射光电来料标志
OR P_On
ANDLD
OUT TR2
LD H10.02  ; 扫码OK记忆
OR H8.04  ; 扫码屏蔽
ANDLD
@SET H20.01  ; 拉带有扫码OK料记忆
LD TR2
AND H10.03  ; 扫码NG记忆
@SET H20.02  ; 拉带有扫码NG料记忆
LD TR1
AND H20.02  ; 拉带有扫码NG料记忆
ANDNOT H20.01  ; 拉带有扫码OK料记忆
@SET H10.08  ; 触发扫码NG抓取
LD TR0
AND D1003.06  ; 等待扫码完成电池通过
@RSET H10.00  ; 扫码阻挡有料记忆
@RSET H10.04  ; 上料拉带放料中记忆
@RSET H10.02  ; 扫码OK记忆
@RSET H10.03  ; 扫码NG记忆
@SET H10.06  ; 进料拉带放料完成
@SET H20.07  ; 等待电池清洁处理
LD TR0
LD H20.01  ; 拉带有扫码OK料记忆
OR H20.02  ; 拉带有扫码NG料记忆
ANDLD
OUT H20.00  ; 拉带来料记忆
LD TR0
AND D1003.08  ; 上料隔离气缸缩回
AND 800.04  ; 隔离气缸1原位标志[0000.04]
AND 800.06  ; 隔离气缸2原位标志[0000.06]
@SET H10.05  ; 隔离缩回启动拉带
LD TR0
AND D1003.09  ; 等待扫码位来料
@RSET H10.05  ; 隔离缩回启动拉带

